// NETWORK 11
DS_HMI.b1001_02_AutoPreparationCompletedFlag := (DS_HMI.b1000_02_AutoPreparationOnOffPB AND bInternalInput_b000_05_ThermalOilTempCtrlReadySignal AND bInternalInput_b000_08_TopDistillatorTempCtrlReadySignal OR DS_HMI.b1001_02_AutoPreparationCompletedFlag) AND DS_HMI.b1000_00_AutoModeOnOffPB AND DS_HMI.b1000_03_AutoModeStartStopPB;

// NETWORK 12
DS_HMI.b1001_10_AutoProgressFlag := DS_HMI.b1001_02_AutoPreparationCompletedFlag;
END_ACTION

ACTION AutoHCTopUp_LD:
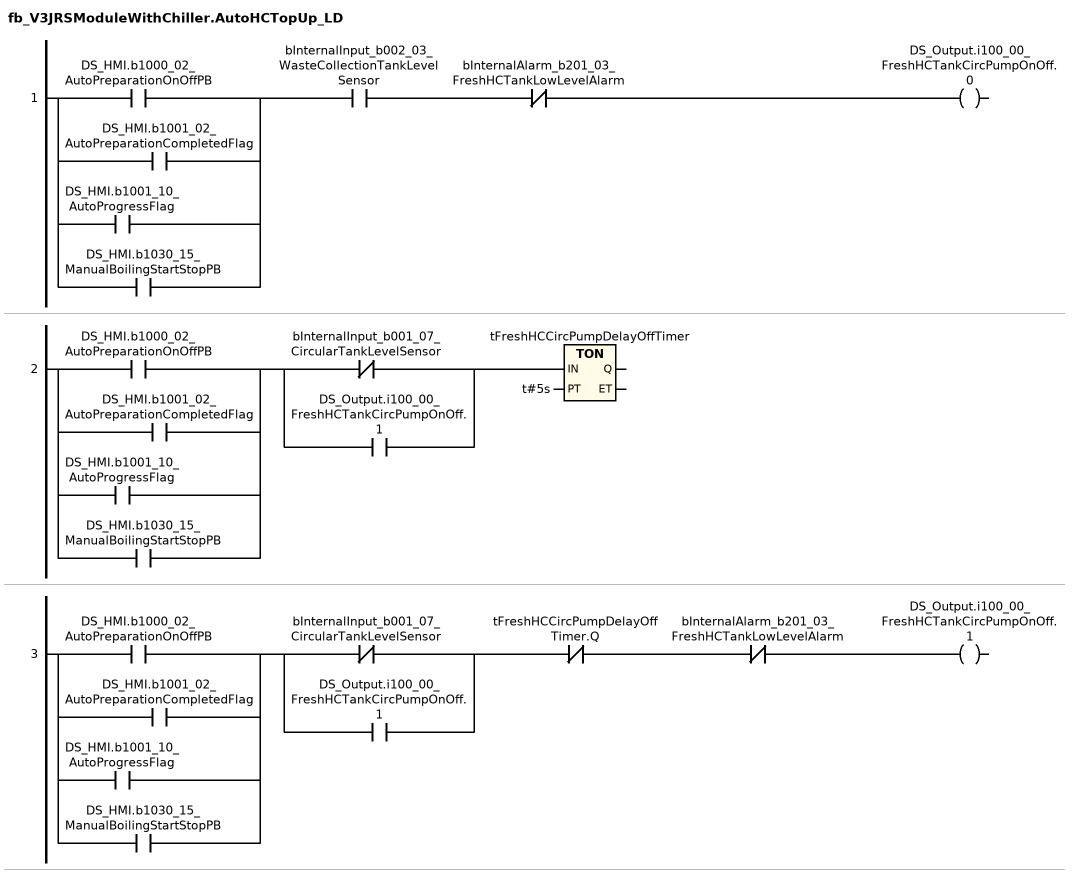
// NETWORK 1
DS_Output.i100_00_FreshHCTankCircPumpOnOff.0 := (DS_HMI.b1000_02_AutoPreparationOnOffPB OR DS_HMI.b1001_02_AutoPreparationCompletedFlag OR DS_HMI.b1001_10_AutoProgressFlag OR DS_HMI.b1030_15_ManualBoilingStartStopPB) AND bInternalInput_b002_03_WasteCollectionTankLevelSensor AND NOT bInternalAlarm_b201_03_FreshHCTankLowLevelAlarm;

// NETWORK 2
tFreshHCCircPumpDelayOffTimer(IN := (DS_HMI.b1000_02_AutoPreparationOnOffPB OR DS_HMI.b1001_02_AutoPreparationCompletedFlag OR DS_HMI.b1001_10_AutoProgressFlag OR DS_HMI.b1030_15_ManualBoilingStartStopPB) AND (NOT bInternalInput_b001_07_CircularTankLevelSensor OR DS_Output.i100_00_FreshHCTankCircPumpOnOff.1), PT := t#5s); // TON

// NETWORK 3
DS_Output.i100_00_FreshHCTankCircPumpOnOff.1 := ((DS_HMI.b1000_02_AutoPreparationOnOffPB OR DS_HMI.b1001_02_AutoPreparationCompletedFlag OR DS_HMI.b1001_10_AutoProgressFlag OR DS_HMI.b1030_15_ManualBoilingStartStopPB) AND (NOT bInternalInput_b001_07_CircularTankLevelSensor OR DS_Output.i100_00_FreshHCTankCircPumpOnOff.1)) AND NOT tFreshHCCircPumpDelayOffTimer.Q AND NOT bInternalAlarm_b201_03_FreshHCTankLowLevelAlarm;
END_ACTION

ACTION BuzzerCtrl_ST:
IF ARiBuzzerOut[1] <>0
AND ARiBuzzerOut[2] <> 0
AND ARiBuzzerOut[3] <> 0
AND ARiBuzzerOut[4] <> 0
THEN
DS_Output.i100_04_Buzzer.0 := TRUE;
ELSE
DS_Output.i100_04_Buzzer.0 := FALSE;
END_IF
END_ACTION

ACTION ChillerCtrl_LD:
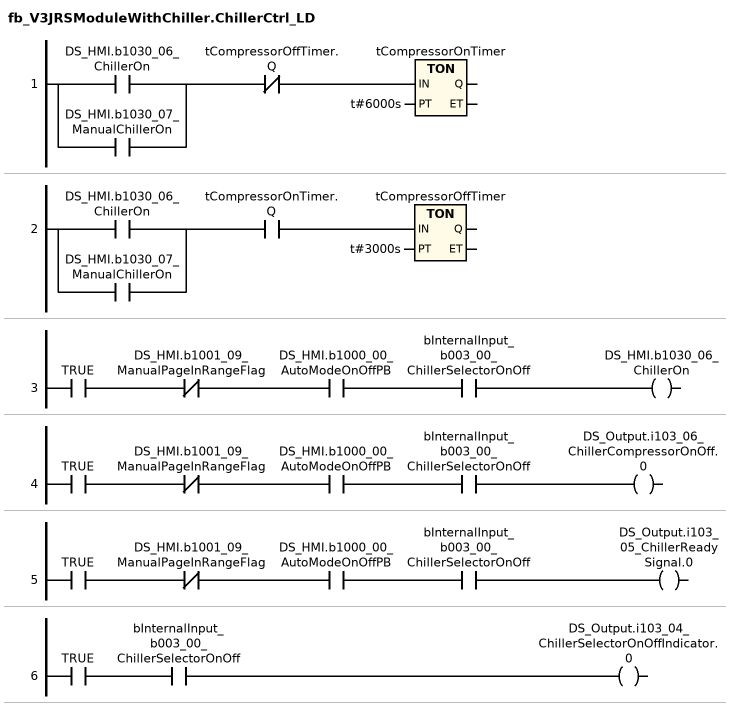
// NETWORK 1
tCompressorOnTimer(IN := (DS_HMI.b1030_06_ChillerOn OR DS_HMI.b1030_07_ManualChillerOn) AND NOT tCompressorOffTimer.Q, PT := t#6000s); // TON

// NETWORK 2
tCompressorOffTimer(IN := (DS_HMI.b1030_06_ChillerOn OR DS_HMI.b1030_07_ManualChillerOn) AND tCompressorOnTimer.Q, PT := t#3000s); // TON

// NETWORK 3
DS_HMI.b1030_06_ChillerOn := TRUE AND NOT DS_HMI.b1001_09_ManualPageInRangeFlag AND DS_HMI.b1000_00_AutoModeOnOffPB AND bInternalInput_b003_00_ChillerSelectorOnOff;

// NETWORK 4
DS_Output.i103_06_ChillerCompressorOnOff.0 := TRUE AND NOT DS_HMI.b1001_09_ManualPageInRangeFlag AND DS_HMI.b1000_00_AutoModeOnOffPB AND bInternalInput_b003_00_ChillerSelectorOnOff;

// NETWORK 5
DS_Output.i103_05_ChillerReadySignal.0 := TRUE AND NOT DS_HMI.b1001_09_ManualPageInRangeFlag AND DS_HMI.b1000_00_AutoModeOnOffPB AND bInternalInput_b003_00_ChillerSelectorOnOff;

// NETWORK 6
DS_Output.i103_04_ChillerSelectorOnOffIndicator.0 := TRUE AND bInternalInput_b003_00_ChillerSelectorOnOff;
END_ACTION

ACTION FixOutput_LD:
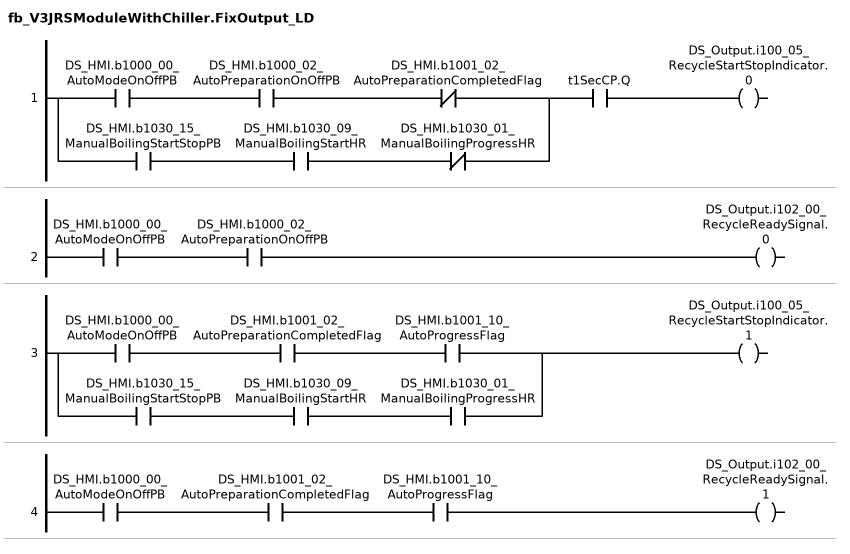
// NETWORK 1
DS_Output.i100_05_RecycleStartStopIndicator.0 := (DS_HMI.b1000_00_AutoModeOnOffPB AND DS_HMI.b1000_02_AutoPreparationOnOffPB AND NOT DS_HMI.b1001_02_AutoPreparationCompletedFlag OR DS_HMI.b1030_15_ManualBoilingStartStopPB AND DS_HMI.b1030_09_ManualBoilingStartHR AND NOT DS_HMI.b1030_01_ManualBoilingProgressHR) AND t1SecCP.Q;

// NETWORK 2
DS_Output.i102_00_RecycleReadySignal.0 := DS_HMI.b1000_00_AutoModeOnOffPB AND DS_HMI.b1000_02_AutoPreparationOnOffPB;

// NETWORK 3
DS_Output.i100_05_RecycleStartStopIndicator.1 := DS_HMI.b1000_00_AutoModeOnOffPB AND DS_HMI.b1001_02_AutoPreparationCompletedFlag AND DS_HMI.b1001_10_AutoProgressFlag OR DS_HMI.b1030_15_ManualBoilingStartStopPB AND DS_HMI.b1030_09_ManualBoilingStartHR AND DS_HMI.b1030_01_ManualBoilingProgressHR;

// NETWORK 4
DS_Output.i102_00_RecycleReadySignal.1 := DS_HMI.b1000_00_AutoModeOnOffPB AND DS_HMI.b1001_02_AutoPreparationCompletedFlag AND DS_HMI.b1001_10_AutoProgressFlag;
END_ACTION

ACTION HighLowLimitCtrl_ST:
(*Low Limit Ctrl*)
IF DS_HMI.iD490_ManualBoilCycleSV < 1 THEN
DS_HMI.iD490_ManualBoilCycleSV := 1;
END_IF

IF DS_HMI.iD200_AutoBoilProcessTimeSV_Min < 30 THEN
DS_HMI.iD200_AutoBoilProcessTimeSV_Min := 30;
END_IF

IF DS_HMI.iD201_AutoBoilDownTimeSV_Min < 5 THEN
DS_HMI.iD201_AutoBoilDownTimeSV_Min := 5;
END_IF

IF DS_HMI.iD202_AutoBoilDistillatorDrainTimeSV_Sec < 5 THEN
DS_HMI.iD202_AutoBoilDistillatorDrainTimeSV_Sec := 5;
END_IF

IF DS_HMI.iD203_AutoBoilSludgeDrainTimeSV_Sec < 5 THEN
DS_HMI.iD203_AutoBoilSludgeDrainTimeSV_Sec := 5;
END_IF

IF DS_HMI.iD210_ManualBoilDownTimeSV_Min < 5 THEN
DS_HMI.iD210_ManualBoilDownTimeSV_Min := 5;
END_IF

IF DS_HMI.iD211_ManualBoilSludgeCoolingTimeSV_Min < 1 THEN
DS_HMI.iD211_ManualBoilSludgeCoolingTimeSV_Min := 1;
END_IF

IF DS_HMI.iD212_ManualBoilSludgeDrainSV_Sec < 5 THEN
DS_HMI.iD212_ManualBoilSludgeDrainSV_Sec := 5;
END_IF




(*High LImit Ctrl*)
IF DS_HMI.iD490_ManualBoilCycleSV > 99 THEN
DS_HMI.iD490_ManualBoilCycleSV := 99;
END_IF

IF DS_HMI.iD200_AutoBoilProcessTimeSV_Min > 9999 THEN
DS_HMI.iD200_AutoBoilProcessTimeSV_Min := 9999;
END_IF

IF DS_HMI.iD201_AutoBoilDownTimeSV_Min > 9999 THEN
DS_HMI.iD201_AutoBoilDownTimeSV_Min := 9999;
END_IF

IF DS_HMI.iD202_AutoBoilDistillatorDrainTimeSV_Sec > 300 THEN
DS_HMI.iD202_AutoBoilDistillatorDrainTimeSV_Sec := 300;
END_IF

IF DS_HMI.iD203_AutoBoilSludgeDrainTimeSV_Sec > 300 THEN
DS_HMI.iD203_AutoBoilSludgeDrainTimeSV_Sec := 300;
END_IF

IF DS_HMI.iD210_ManualBoilDownTimeSV_Min > 99 THEN
DS_HMI.iD210_ManualBoilDownTimeSV_Min := 99;
END_IF

IF DS_HMI.iD211_ManualBoilSludgeCoolingTimeSV_Min > 9999 THEN
DS_HMI.iD211_ManualBoilSludgeCoolingTimeSV_Min := 9999;
END_IF

IF DS_HMI.iD212_ManualBoilSludgeDrainSV_Sec > 300 THEN
DS_HMI.iD212_ManualBoilSludgeDrainSV_Sec := 300;
END_IF
END_ACTION

ACTION JRSMachineServiceCtrl_LD:
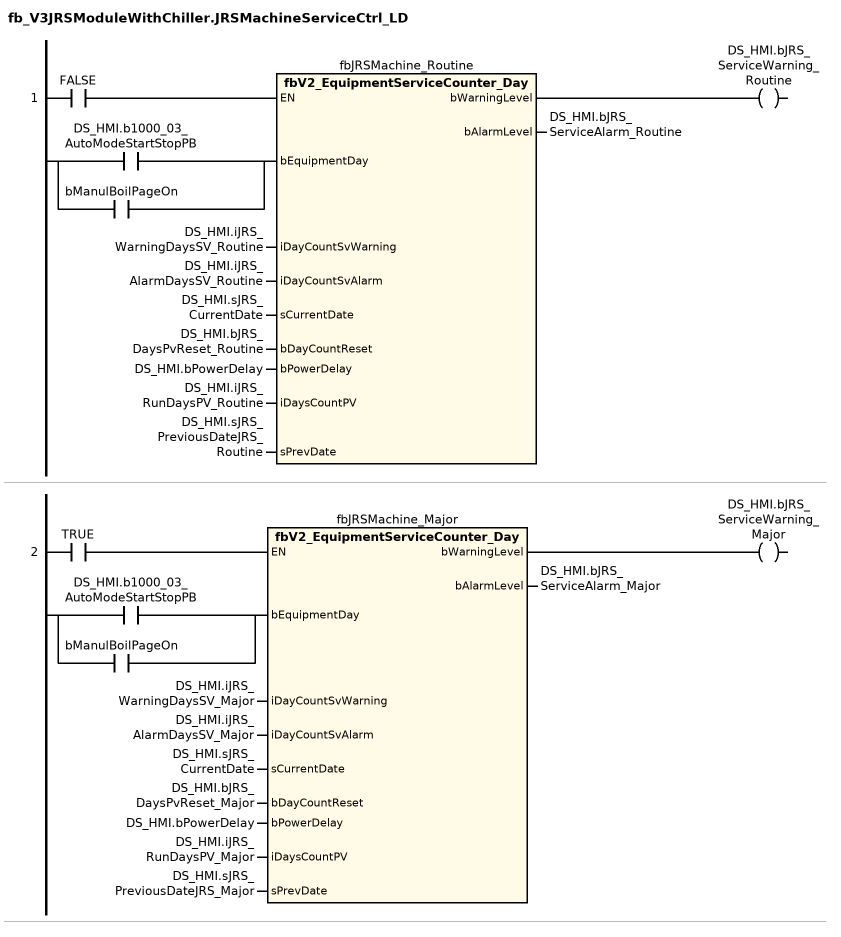
// NETWORK 1
IF FALSE THEN
    fbJRSMachine_Routine(
        bEquipmentDay := DS_HMI.b1000_03_AutoModeStartStopPB OR bManulBoilPageOn,
        iDayCountSvWarning := DS_HMI.iJRS_WarningDaysSV_Routine,
        iDayCountSvAlarm := DS_HMI.iJRS_AlarmDaysSV_Routine,
        sCurrentDate := DS_HMI.sJRS_CurrentDate,
        bDayCountReset := DS_HMI.bJRS_DaysPvReset_Routine,
        bPowerDelay := DS_HMI.bPowerDelay,
        iDaysCountPV := DS_HMI.iJRS_RunDaysPV_Routine,
        sPrevDate := DS_HMI.sJRS_PreviousDateJRS_Routine,
        bAlarmLevel => DS_HMI.bJRS_ServiceAlarm_Routine); // fbV2_EquipmentServiceCounter_Day
END_IF
DS_HMI.bJRS_ServiceWarning_Routine := fbJRSMachine_Routine.bWarningLevel;

// NETWORK 2
fbJRSMachine_Major(
    bEquipmentDay := DS_HMI.b1000_03_AutoModeStartStopPB OR bManulBoilPageOn,
    iDayCountSvWarning := DS_HMI.iJRS_WarningDaysSV_Major,
    iDayCountSvAlarm := DS_HMI.iJRS_AlarmDaysSV_Major,
    sCurrentDate := DS_HMI.sJRS_CurrentDate,
    bDayCountReset := DS_HMI.bJRS_DaysPvReset_Major,
    bPowerDelay := DS_HMI.bPowerDelay,
    iDaysCountPV := DS_HMI.iJRS_RunDaysPV_Major,
    sPrevDate := DS_HMI.sJRS_PreviousDateJRS_Major,
    bAlarmLevel => DS_HMI.bJRS_ServiceAlarm_Major); // fbV2_EquipmentServiceCounter_Day
DS_HMI.bJRS_ServiceWarning_Major := fbJRSMachine_Major.bWarningLevel;
END_ACTION

ACTION ManualBoilingCtrl_LD:
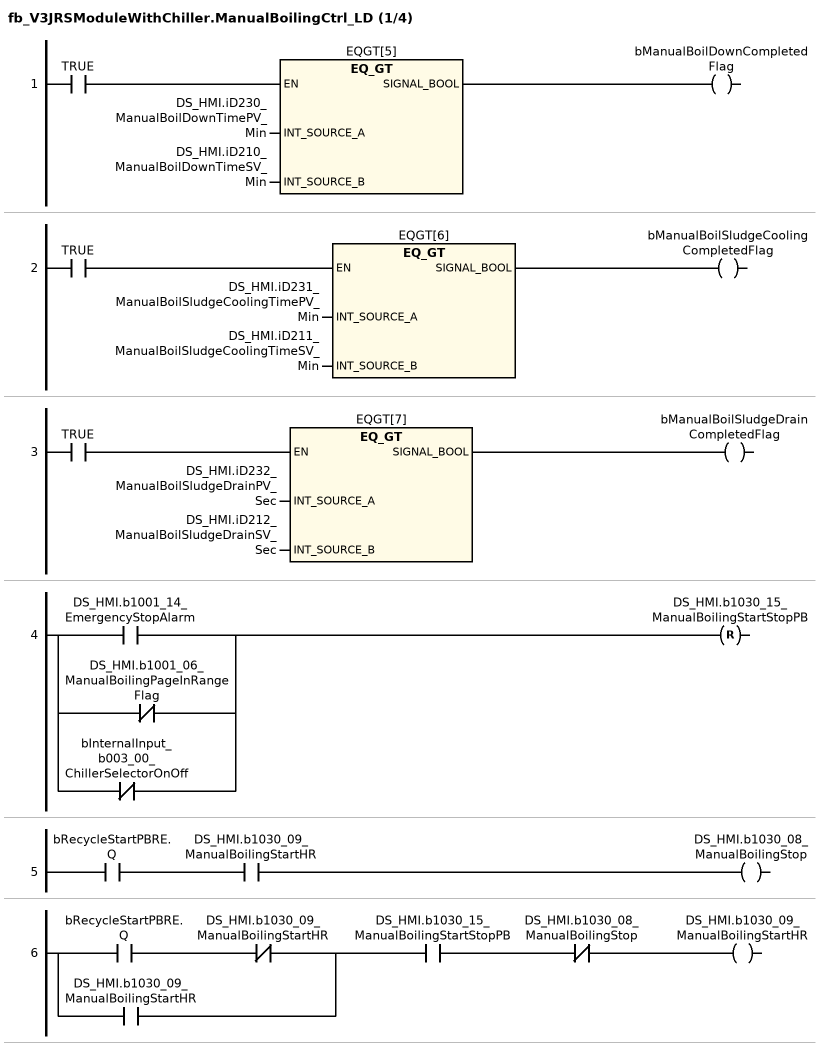
// NETWORK 1
EQGT[5](INT_SOURCE_A := DS_HMI.iD230_ManualBoilDownTimePV_Min, INT_SOURCE_B := DS_HMI.iD210_ManualBoilDownTimeSV_Min); // EQ_GT
bManualBoilDownCompletedFlag := EQGT[5].SIGNAL_BOOL;

// NETWORK 2
EQGT[6](INT_SOURCE_A := DS_HMI.iD231_ManualBoilSludgeCoolingTimePV_Min, INT_SOURCE_B := DS_HMI.iD211_ManualBoilSludgeCoolingTimeSV_Min); // EQ_GT
bManualBoilSludgeCoolingCompletedFlag := EQGT[6].SIGNAL_BOOL;

// NETWORK 3
EQGT[7](INT_SOURCE_A := DS_HMI.iD232_ManualBoilSludgeDrainPV_Sec, INT_SOURCE_B := DS_HMI.iD212_ManualBoilSludgeDrainSV_Sec); // EQ_GT
bManualBoilSludgeDrainCompletedFlag := EQGT[7].SIGNAL_BOOL;

// NETWORK 4
DS_HMI.b1030_15_ManualBoilingStartStopPB R= DS_HMI.b1001_14_EmergencyStopAlarm OR NOT DS_HMI.b1001_06_ManualBoilingPageInRangeFlag OR NOT bInternalInput_b003_00_ChillerSelectorOnOff;

// NETWORK 5
DS_HMI.b1030_08_ManualBoilingStop := bRecycleStartPBRE.Q AND DS_HMI.b1030_09_ManualBoilingStartHR;

// NETWORK 6
DS_HMI.b1030_09_ManualBoilingStartHR := (bRecycleStartPBRE.Q AND NOT DS_HMI.b1030_09_ManualBoilingStartHR OR DS_HMI.b1030_09_ManualBoilingStartHR) AND DS_HMI.b1030_15_ManualBoilingStartStopPB AND NOT DS_HMI.b1030_08_ManualBoilingStop;

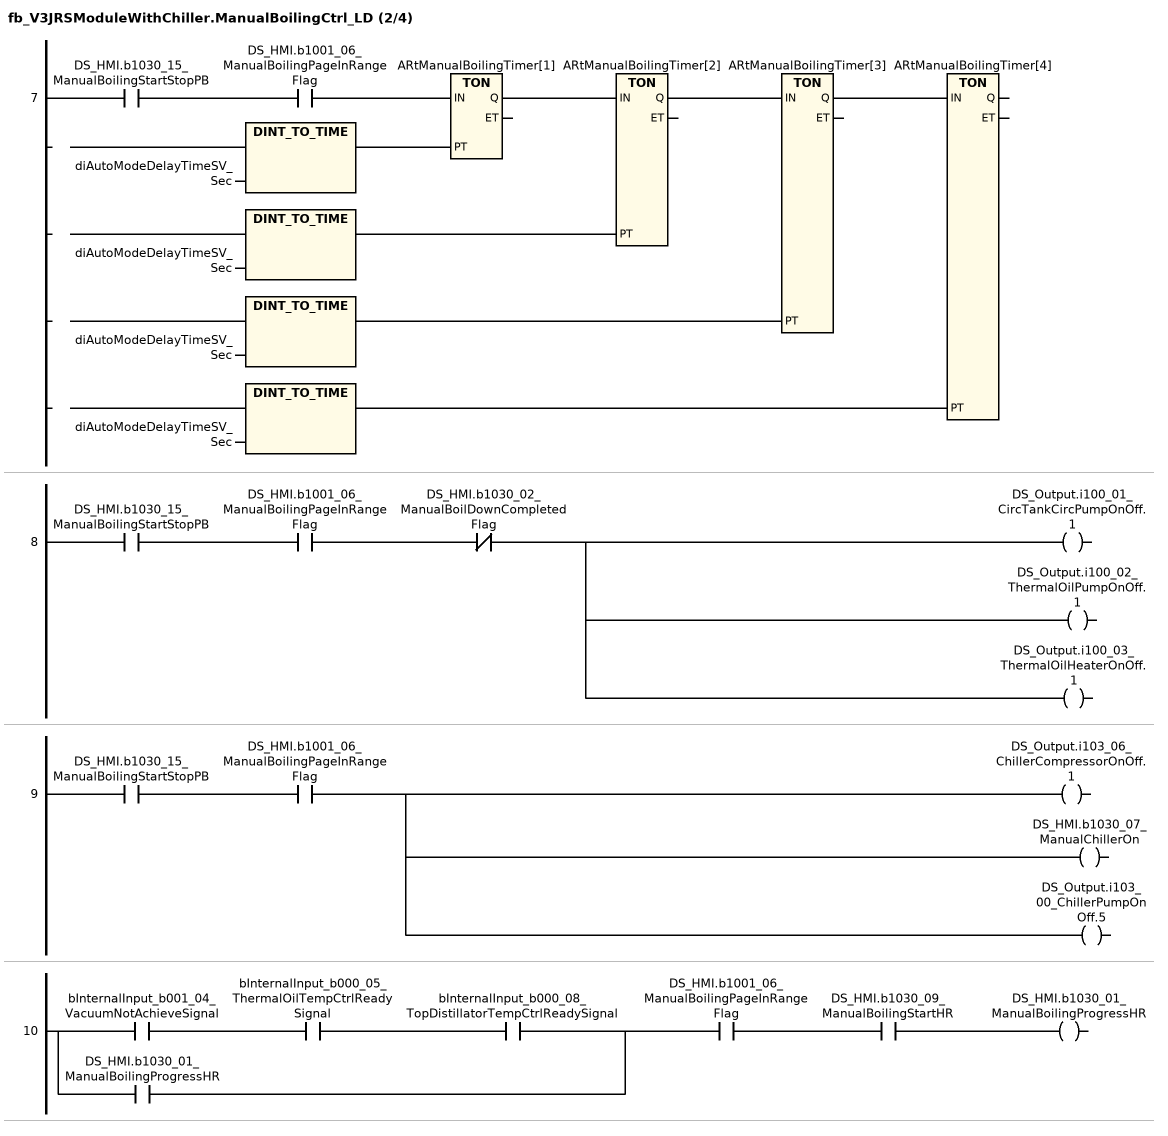
// NETWORK 7
ARtManualBoilingTimer[1](IN := DS_HMI.b1030_15_ManualBoilingStartStopPB AND DS_HMI.b1001_06_ManualBoilingPageInRangeFlag, PT := DINT_TO_TIME(diAutoModeDelayTimeSV_Sec)); // TON
ARtManualBoilingTimer[2](IN := ARtManualBoilingTimer[1].Q, PT := DINT_TO_TIME(diAutoModeDelayTimeSV_Sec)); // TON
ARtManualBoilingTimer[3](IN := ARtManualBoilingTimer[2].Q, PT := DINT_TO_TIME(diAutoModeDelayTimeSV_Sec)); // TON
ARtManualBoilingTimer[4](IN := ARtManualBoilingTimer[3].Q, PT := DINT_TO_TIME(diAutoModeDelayTimeSV_Sec)); // TON

// NETWORK 8
_w5 := DS_HMI.b1030_15_ManualBoilingStartStopPB AND DS_HMI.b1001_06_ManualBoilingPageInRangeFlag AND NOT DS_HMI.b1030_02_ManualBoilDownCompletedFlag;
DS_Output.i100_01_CircTankCircPumpOnOff.1 := _w5;
DS_Output.i100_02_ThermalOilPumpOnOff.1 := _w5;
DS_Output.i100_03_ThermalOilHeaterOnOff.1 := _w5;

// NETWORK 9
_w6 := DS_HMI.b1030_15_ManualBoilingStartStopPB AND DS_HMI.b1001_06_ManualBoilingPageInRangeFlag;
DS_Output.i103_06_ChillerCompressorOnOff.1 := _w6;
DS_HMI.b1030_07_ManualChillerOn := _w6;
DS_Output.i103_00_ChillerPumpOnOff.5 := _w6;

// NETWORK 10
DS_HMI.b1030_01_ManualBoilingProgressHR := (bInternalInput_b001_04_VacuumNotAchieveSignal AND bInternalInput_b000_05_ThermalOilTempCtrlReadySignal AND bInternalInput_b000_08_TopDistillatorTempCtrlReadySignal OR DS_HMI.b1030_01_ManualBoilingProgressHR) AND DS_HMI.b1001_06_ManualBoilingPageInRangeFlag AND DS_HMI.b1030_09_ManualBoilingStartHR;

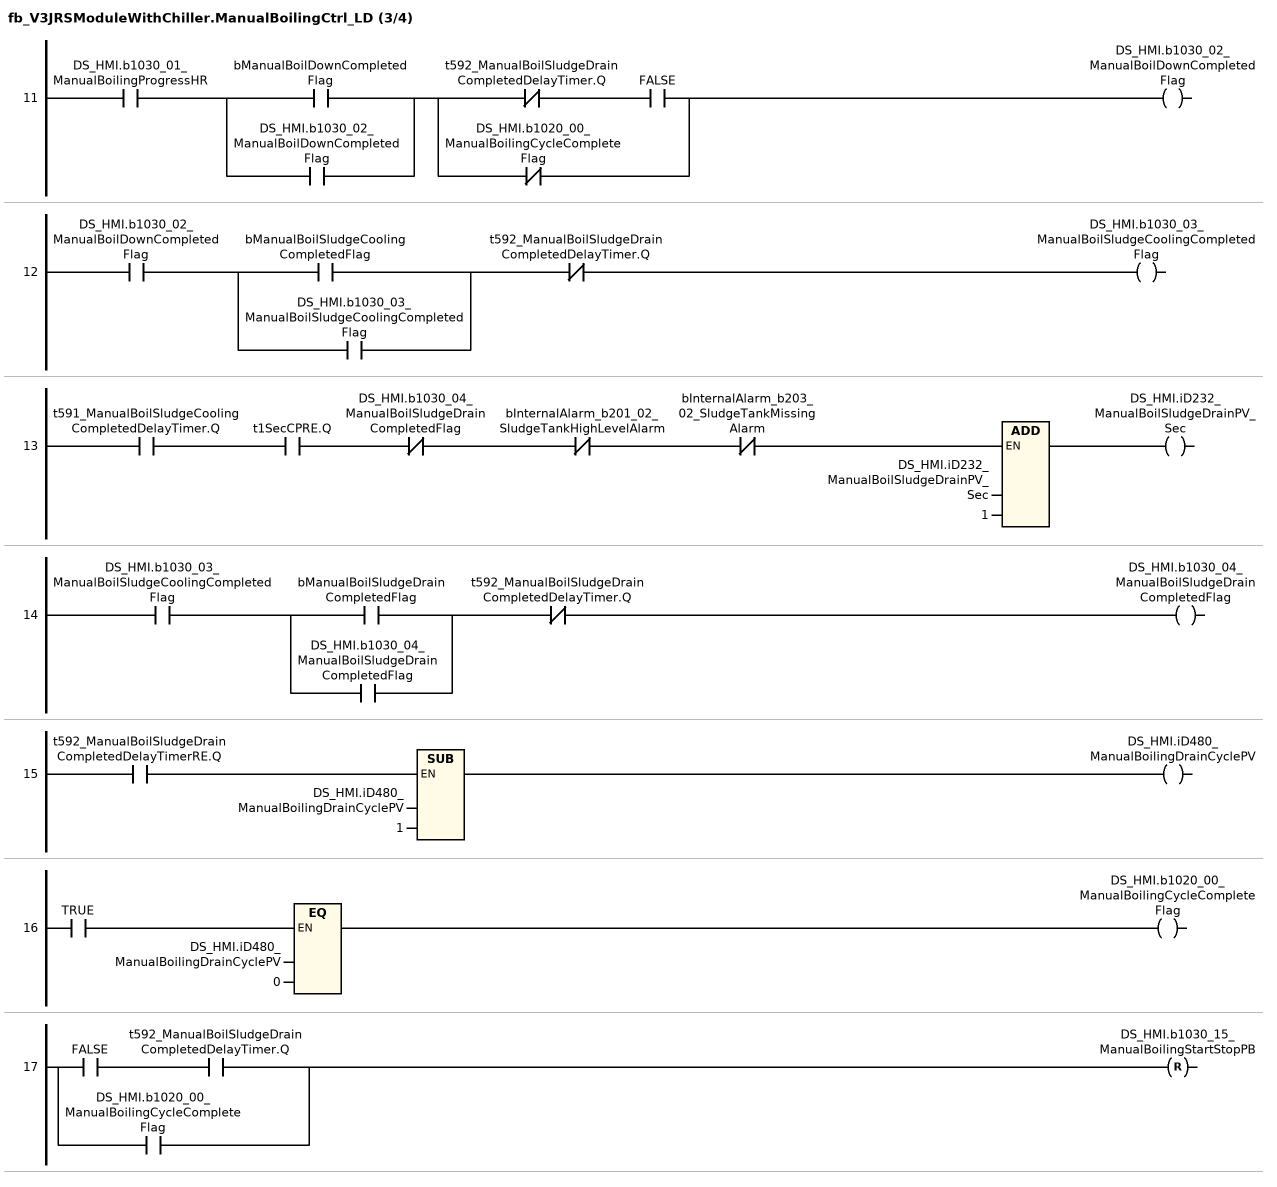
// NETWORK 11
DS_HMI.b1030_02_ManualBoilDownCompletedFlag := DS_HMI.b1030_01_ManualBoilingProgressHR AND (bManualBoilDownCompletedFlag OR DS_HMI.b1030_02_ManualBoilDownCompletedFlag) AND (NOT t592_ManualBoilSludgeDrainCompletedDelayTimer.Q AND FALSE OR NOT DS_HMI.b1020_00_ManualBoilingCycleCompleteFlag);

// NETWORK 12
DS_HMI.b1030_03_ManualBoilSludgeCoolingCompletedFlag := (DS_HMI.b1030_02_ManualBoilDownCompletedFlag AND (bManualBoilSludgeCoolingCompletedFlag OR DS_HMI.b1030_03_ManualBoilSludgeCoolingCompletedFlag)) AND NOT t592_ManualBoilSludgeDrainCompletedDelayTimer.Q;

// NETWORK 13
IF t591_ManualBoilSludgeCoolingCompletedDelayTimer.Q AND t1SecCPRE.Q AND NOT DS_HMI.b1030_04_ManualBoilSludgeDrainCompletedFlag AND NOT bInternalAlarm_b201_02_SludgeTankHighLevelAlarm AND NOT bInternalAlarm_b203_02_SludgeTankMissingAlarm THEN
    _w7 := DS_HMI.iD232_ManualBoilSludgeDrainPV_Sec + 1;
END_IF
DS_HMI.iD232_ManualBoilSludgeDrainPV_Sec := _w7;

// NETWORK 14
DS_HMI.b1030_04_ManualBoilSludgeDrainCompletedFlag := (DS_HMI.b1030_03_ManualBoilSludgeCoolingCompletedFlag AND (bManualBoilSludgeDrainCompletedFlag OR DS_HMI.b1030_04_ManualBoilSludgeDrainCompletedFlag)) AND NOT t592_ManualBoilSludgeDrainCompletedDelayTimer.Q;

// NETWORK 15
IF t592_ManualBoilSludgeDrainCompletedDelayTimerRE.Q THEN _w8 := DS_HMI.iD480_ManualBoilingDrainCyclePV - 1; END_IF
DS_HMI.iD480_ManualBoilingDrainCyclePV := _w8;

// NETWORK 16
DS_HMI.b1020_00_ManualBoilingCycleCompleteFlag := DS_HMI.iD480_ManualBoilingDrainCyclePV = 0;

// NETWORK 17
DS_HMI.b1030_15_ManualBoilingStartStopPB R= FALSE AND t592_ManualBoilSludgeDrainCompletedDelayTimer.Q OR DS_HMI.b1020_00_ManualBoilingCycleCompleteFlag;

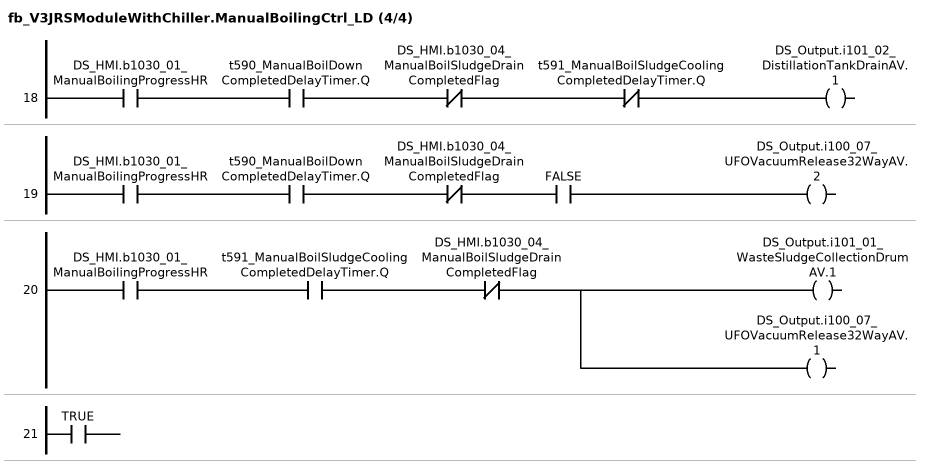
// NETWORK 18
DS_Output.i101_02_DistillationTankDrainAV.1 := DS_HMI.b1030_01_ManualBoilingProgressHR AND t590_ManualBoilDownCompletedDelayTimer.Q AND NOT DS_HMI.b1030_04_ManualBoilSludgeDrainCompletedFlag AND NOT t591_ManualBoilSludgeCoolingCompletedDelayTimer.Q;

// NETWORK 19
DS_Output.i100_07_UFOVacuumRelease32WayAV.2 := DS_HMI.b1030_01_ManualBoilingProgressHR AND t590_ManualBoilDownCompletedDelayTimer.Q AND NOT DS_HMI.b1030_04_ManualBoilSludgeDrainCompletedFlag AND FALSE;

// NETWORK 20
_w9 := DS_HMI.b1030_01_ManualBoilingProgressHR AND t591_ManualBoilSludgeCoolingCompletedDelayTimer.Q AND NOT DS_HMI.b1030_04_ManualBoilSludgeDrainCompletedFlag;
DS_Output.i101_01_WasteSludgeCollectionDrumAV.1 := _w9;
DS_Output.i100_07_UFOVacuumRelease32WayAV.1 := _w9;

// NETWORK 21
END_ACTION

ACTION ManualBoilingCtrl_ST:
	(*Timer*)
	t590_ManualBoilDownCompletedDelayTimer(IN:=DS_HMI.b1030_02_ManualBoilDownCompletedFlag , PT:=t#1s , Q=> , ET=> );
	t591_ManualBoilSludgeCoolingCompletedDelayTimer(IN:=DS_HMI.b1030_03_ManualBoilSludgeCoolingCompletedFlag , PT:=t#1s , Q=> , ET=> );
	t592_ManualBoilSludgeDrainCompletedDelayTimer(IN:=DS_HMI.b1030_04_ManualBoilSludgeDrainCompletedFlag , PT:=t#1s , Q=> , ET=> );

	(*R_TRIG*)
	t592_ManualBoilSludgeDrainCompletedDelayTimerRE(CLK:=t592_ManualBoilSludgeDrainCompletedDelayTimer.Q , Q=> );
	bManualBoilSludgeDrainCompletedRE(CLK:=DS_HMI.b1030_04_ManualBoilSludgeDrainCompletedFlag , Q=> );


	(*ManualBoiling Boil Process Time Counting*)
	IF DS_HMI.b1030_01_ManualBoilingProgressHR
	AND t1SecCPRE.Q
	THEN

		IF NOT DS_HMI.b1030_02_ManualBoilDownCompletedFlag THEN

			DS_HMI.iD235_ManualBoilDownTimePV_Sec := DS_HMI.iD235_ManualBoilDownTimePV_Sec + 1;
	
			IF DS_HMI.iD235_ManualBoilDownTimePV_Sec > 59 THEN
				DS_HMI.iD230_ManualBoilDownTimePV_Min := DS_HMI.iD230_ManualBoilDownTimePV_Min + 1;
				DS_HMI.iD235_ManualBoilDownTimePV_Sec := 0;
			END_IF

		END_IF

	END_IF

	(*ManualBoiling Boil Down Time Counting*)

	IF t590_ManualBoilDownCompletedDelayTimer.Q
	AND t1SecCPRE.Q
	THEN

		IF NOT DS_HMI.b1030_03_ManualBoilSludgeCoolingCompletedFlag THEN

			DS_HMI.iD236_ManualBoilSludgeCoolingTimePV_Sec := DS_HMI.iD236_ManualBoilSludgeCoolingTimePV_Sec + 1;

			IF DS_HMI.iD236_ManualBoilSludgeCoolingTimePV_Sec > 59 THEN
				DS_HMI.iD231_ManualBoilSludgeCoolingTimePV_Min := DS_HMI.iD231_ManualBoilSludgeCoolingTimePV_Min + 1;
				DS_HMI.iD236_ManualBoilSludgeCoolingTimePV_Sec := 0;
			END_IF

		END_IF

	END_IF

	(*Manual Boiling Reset*)
	IF NOT DS_HMI.b1030_15_ManualBoilingStartStopPB THEN
		DS_HMI.iD230_ManualBoilDownTimePV_Min						:= 0;
		DS_HMI.iD231_ManualBoilSludgeCoolingTimePV_Min				:= 0;
		DS_HMI.iD232_ManualBoilSludgeDrainPV_Sec					:= 0;
		DS_HMI.iD480_ManualBoilingDrainCyclePV						:= DS_HMI.iD490_ManualBoilCycleSV;

	END_IF



	IF bManualBoilSludgeDrainCompletedRE.Q OR  DS_HMI.b1020_00_ManualBoilingCycleCompleteFlag THEN
	
		DS_HMI.iD230_ManualBoilDownTimePV_Min						:= 0;
		DS_HMI.iD231_ManualBoilSludgeCoolingTimePV_Min				:= 0;
		DS_HMI.iD232_ManualBoilSludgeDrainPV_Sec					:= 0;
		DS_HMI.iD235_ManualBoilDownTimePV_Sec						:= 0;
		DS_HMI.iD236_ManualBoilSludgeCoolingTimePV_Sec				:= 0;

	END_IF
END_ACTION

ACTION ManualCtrl_ST:
	(*Manual Page In Range*)
	IF (	DS_HMI.iD0_HMICurrentPage > 19 		AND 	DS_HMI.iD0_HMICurrentPage < 41)
	OR	DS_HMI.iD0_HMICurrentPage = 2
	OR	DS_HMI.iD0_HMICurrentPage = 61
	OR	DS_HMI.iD0_HMICurrentPage = 63
	OR	DS_HMI.iD0_HMICurrentPage = 100
	OR	DS_HMI.iD0_HMICurrentPage = 101
	OR	DS_HMI.iD0_HMICurrentPage = 103 	THEN
		DS_HMI.b1001_09_ManualPageInRangeFlag := TRUE;
	ELSE
		DS_HMI.b1001_09_ManualPageInRangeFlag := FALSE;
	END_IF


	(*Manual Boiling Page In Range*)
	IF (	DS_HMI.iD0_HMICurrentPage > 99 		AND 	DS_HMI.iD0_HMICurrentPage < 102)
	OR	DS_HMI.iD0_HMICurrentPage = 22 		THEN
		DS_HMI.b1001_06_ManualBoilingPageInRangeFlag := TRUE;
	ELSE
		DS_HMI.b1001_06_ManualBoilingPageInRangeFlag := FALSE;
	END_IF



	IF NOT DS_HMI.b1001_09_ManualPageInRangeFlag OR DS_HMI.b1001_14_EmergencyStopAlarm THEN
		DS_Output.i100_00_FreshHCTankCircPumpOnOff.15			:= FALSE;
		DS_Output.i100_01_CircTankCircPumpOnOff.15				:= FALSE;
		DS_Output.i100_02_ThermalOilPumpOnOff.15				:= FALSE;
		DS_Output.i100_03_ThermalOilHeaterOnOff.15				:= FALSE;
		DS_Output.i100_04_Buzzer.15								:= FALSE;
		DS_Output.i100_05_RecycleStartStopIndicator.15				:= FALSE;
		DS_Output.i100_06_Reserved.15							:= FALSE;
		DS_Output.i100_07_UFOVacuumRelease32WayAV.15		:= FALSE;

		DS_Output.i101_00_CondenserTankVacuumReleaseAV.15	:= FALSE;
		DS_Output.i101_01_WasteSludgeCollectionDrumAV.15		:= FALSE;
		DS_Output.i101_02_DistillationTankDrainAV.15				:= FALSE;
		DS_Output.i101_03_EconomizerAV.15						:= FALSE;
		DS_Output.i101_04_Reserved.15							:= FALSE;
		DS_Output.i101_05_Reserved.15							:= FALSE;
		DS_Output.i101_06_VaporGenerationAV.15					:= FALSE;
		DS_Output.i101_07_VacuumSharingAV.15					:= FALSE;

		DS_Output.i102_00_RecycleReadySignal.15					:= FALSE;
		DS_Output.i102_01_VaporNotAvailableForRequestSignal.15	:= FALSE;
		DS_Output.i102_02_ToMainMachineSignal3.15				:= FALSE;
		DS_Output.i102_03_ToMainMachineSignal4.15				:= FALSE;
		DS_Output.i102_04_ToMainMachineSignal5.15				:= FALSE;
		DS_Output.i102_05_Reserved.15							:= FALSE;
		DS_Output.i102_06_Reserved.15							:= FALSE;
		DS_Output.i102_07_Reserved.15							:= FALSE;

		DS_Output.i103_00_ChillerPumpOnOff.15					:= FALSE;
		DS_Output.i103_01_Reserved.15							:= FALSE;
		DS_Output.i103_02_Reserved.15							:= FALSE;
		DS_Output.i103_03_Reserved.15							:= FALSE;
		DS_Output.i103_04_ChillerSelectorOnOffIndicator.15			:= FALSE;
		DS_Output.i103_05_ChillerReadySignal.15					:= FALSE;
		DS_Output.i103_06_ChillerCompressorOnOff.15				:= FALSE;
		DS_Output.i103_07_Reserved.15							:= FALSE;
	END_IF

	IF NOT bInternalInput_b003_00_ChillerSelectorOnOff THEN
		DS_Output.i103_06_ChillerCompressorOnOff.15				:= FALSE;
	END_IF
END_ACTION

ACTION MessageDisplayCtrl_ST:
	IF  NOT DS_HMI.b1001_15_AlarmOccur THEN

		IF NOT 		DS_HMI.b1000_00_AutoModeOnOffPB THEN

			DS_HMI.iD100_MessageDisplay := 0;
			DS_HMI.sD100_MessageDisplay := 'Machine Idle';

(*		ELSIF 		DS_HMI.b1000_00_AutoModeOnOffPB
		AND 		DS_HMI.b1000_01_AutoOriginOnOffPB
		AND NOT 	DS_HMI.b1001_01_AutoOriginCompletedFlag THEN

			DS_HMI.iD100_MessageDisplay := 1;
			DS_HMI.sD100_MessageDisplay := 'Auto Origin In Progress...';
*)
		ELSIF 		DS_HMI.b1000_00_AutoModeOnOffPB
		AND 		DS_HMI.b1000_02_AutoPreparationOnOffPB
		AND NOT 	DS_HMI.b1001_02_AutoPreparationCompletedFlag THEN

			DS_HMI.iD100_MessageDisplay := 2;
			DS_HMI.sD100_MessageDisplay := 'Auto Preparation In Progress...';

		ELSIF 		DS_HMI.b1000_00_AutoModeOnOffPB
(*		AND 		DS_HMI.b1001_01_AutoOriginCompletedFlag*)
		AND 		DS_HMI.b1000_02_AutoPreparationOnOffPB
		AND 		DS_HMI.b1001_02_AutoPreparationCompletedFlag THEN

			DS_HMI.iD100_MessageDisplay := 3;
			DS_HMI.sD100_MessageDisplay := 'Machine Ready, Press "Start" for Operation';

		ELSIF 		DS_HMI.b1000_00_AutoModeOnOffPB
(*		AND 		DS_HMI.b1001_01_AutoOriginCompletedFlag*)
		AND 		DS_HMI.b1001_02_AutoPreparationCompletedFlag
		AND 		DS_HMI.b1001_10_AutoProgressFlag
		AND NOT 	DS_HMI.b1000_05_AutoCycleStopPB THEN

			DS_HMI.iD100_MessageDisplay := 4;
			DS_HMI.sD100_MessageDisplay := 'Machine Operation...';

		ELSIF 		DS_HMI.b1000_00_AutoModeOnOffPB
(*		AND 		DS_HMI.b1001_01_AutoOriginCompletedFlag*)
		AND 		DS_HMI.b1001_02_AutoPreparationCompletedFlag
		AND 		DS_HMI.b1001_10_AutoProgressFlag
		AND 		DS_HMI.b1000_05_AutoCycleStopPB THEN

			DS_HMI.iD100_MessageDisplay := 5;
			DS_HMI.sD100_MessageDisplay := 'Auto Cycle Stop...';

		END_IF

	ELSE
		DS_HMI.iD100_MessageDisplay := 6;
			DS_HMI.sD100_MessageDisplay := 'Alarm Occured, Please check Alarm Page for more detail';

	END_IF
END_ACTION

ACTION Other_LD:
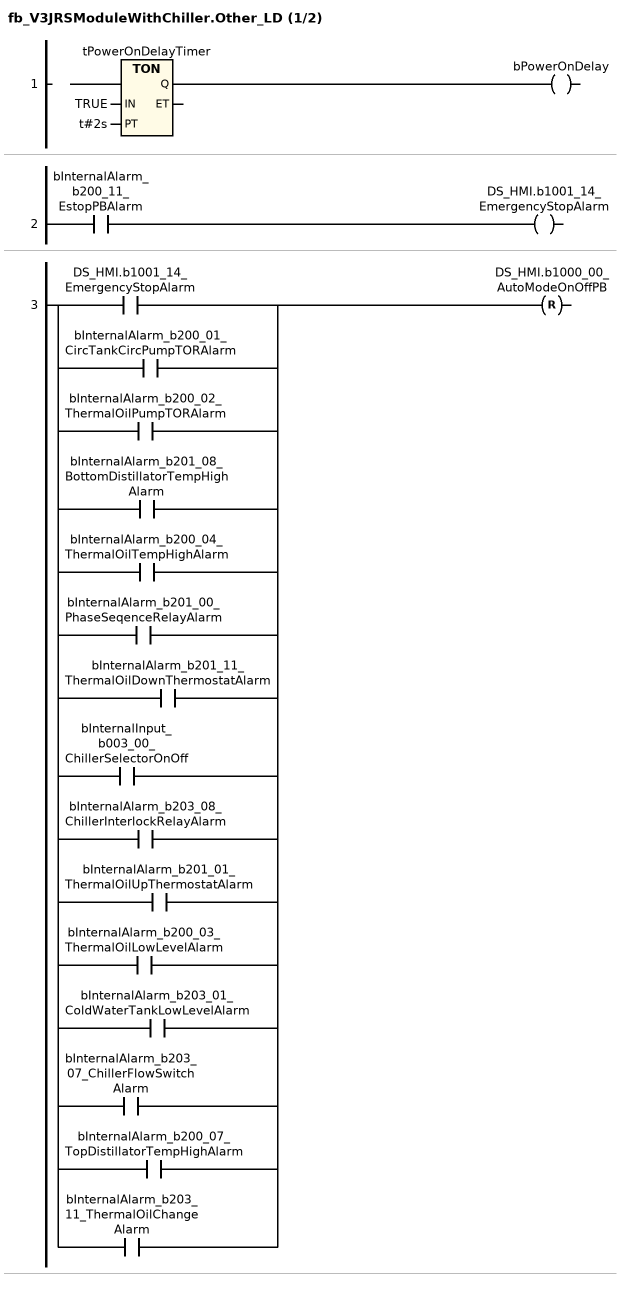
// NETWORK 1
tPowerOnDelayTimer(IN := TRUE, PT := t#2s); // TON
bPowerOnDelay := tPowerOnDelayTimer.Q;

// NETWORK 2
DS_HMI.b1001_14_EmergencyStopAlarm := bInternalAlarm_b200_11_EstopPBAlarm;

// NETWORK 3
DS_HMI.b1000_00_AutoModeOnOffPB R= DS_HMI.b1001_14_EmergencyStopAlarm OR bInternalAlarm_b200_01_CircTankCircPumpTORAlarm OR bInternalAlarm_b200_02_ThermalOilPumpTORAlarm OR bInternalAlarm_b201_08_BottomDistillatorTempHighAlarm OR bInternalAlarm_b200_04_ThermalOilTempHighAlarm OR bInternalAlarm_b201_00_PhaseSeqenceRelayAlarm OR bInternalAlarm_b201_11_ThermalOilDownThermostatAlarm OR bInternalInput_b003_00_ChillerSelectorOnOff OR bInternalAlarm_b203_08_ChillerInterlockRelayAlarm OR bInternalAlarm_b201_01_ThermalOilUpThermostatAlarm OR bInternalAlarm_b200_03_ThermalOilLowLevelAlarm OR bInternalAlarm_b203_01_ColdWaterTankLowLevelAlarm OR bInternalAlarm_b203_07_ChillerFlowSwitchAlarm OR bInternalAlarm_b200_07_TopDistillatorTempHighAlarm OR bInternalAlarm_b203_11_ThermalOilChangeAlarm;

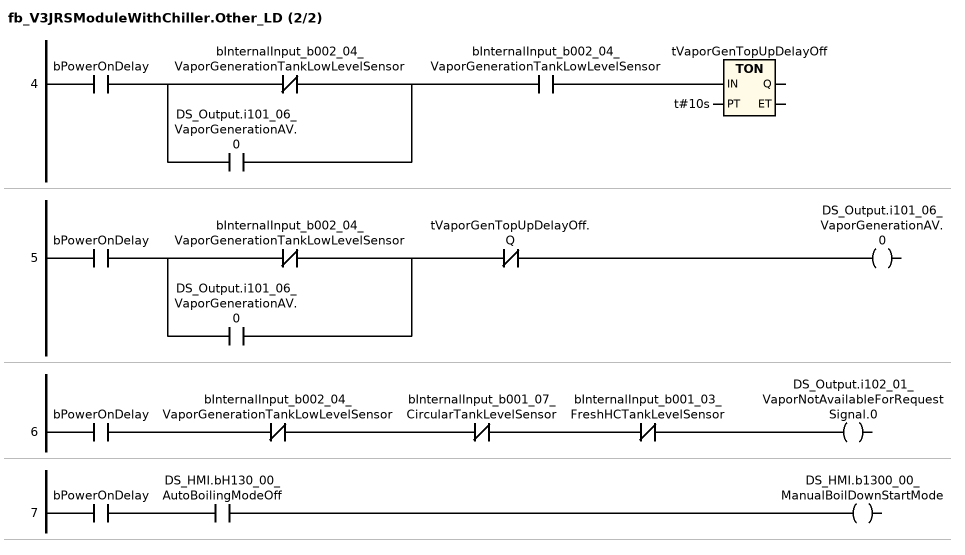
// NETWORK 4
tVaporGenTopUpDelayOff(IN := (bPowerOnDelay AND (NOT bInternalInput_b002_04_VaporGenerationTankLowLevelSensor OR DS_Output.i101_06_VaporGenerationAV.0)) AND bInternalInput_b002_04_VaporGenerationTankLowLevelSensor, PT := t#10s); // TON

// NETWORK 5
DS_Output.i101_06_VaporGenerationAV.0 := (bPowerOnDelay AND (NOT bInternalInput_b002_04_VaporGenerationTankLowLevelSensor OR DS_Output.i101_06_VaporGenerationAV.0)) AND NOT tVaporGenTopUpDelayOff.Q;

// NETWORK 6
DS_Output.i102_01_VaporNotAvailableForRequestSignal.0 := bPowerOnDelay AND NOT bInternalInput_b002_04_VaporGenerationTankLowLevelSensor AND NOT bInternalInput_b001_07_CircularTankLevelSensor AND NOT bInternalInput_b001_03_FreshHCTankLevelSensor;

// NETWORK 7
DS_HMI.b1300_00_ManualBoilDownStartMode := bPowerOnDelay AND DS_HMI.bH130_00_AutoBoilingModeOff;
END_ACTION

ACTION Other_ST:
	(*Map Alarm into Word so that can generate Alarm Occur Bit*)
	AriAlarmFlag[1].0 := bInternalAlarm_b200_00_FreshHCTankCircPumpTORAlarm ;
	AriAlarmFlag[1].1 := bInternalAlarm_b200_01_CircTankCircPumpTORAlarm ;
	AriAlarmFlag[1].2 := bInternalAlarm_b200_02_ThermalOilPumpTORAlarm ;
	AriAlarmFlag[1].3 := bInternalAlarm_b200_03_ThermalOilLowLevelAlarm ;
	AriAlarmFlag[1].4 := bInternalAlarm_b200_04_ThermalOilTempHighAlarm ;
	AriAlarmFlag[1].5 := bInternalAlarm_b200_05_ThermalOilTempNotReadyAlarm ;
	AriAlarmFlag[1].6 := bInternalAlarm_b200_06_ThermalOilHeaterOnOffAlarm ;
	AriAlarmFlag[1].7 := bInternalAlarm_b200_07_TopDistillatorTempHighAlarm ;
	AriAlarmFlag[1].8 := bInternalAlarm_b200_08_TopDistillatorTempNotReadyAlarm ;
	AriAlarmFlag[1].9 := bInternalAlarm_b200_09_TopDistillatorHeaterOnOffAlarm ;
	AriAlarmFlag[1].10 := bInternalAlarm_b200_10_RecycleStartStopPBAlarm ;
	AriAlarmFlag[1].11 := bInternalAlarm_b200_11_EstopPBAlarm ;
	
	AriAlarmFlag[2].0 := bInternalAlarm_b201_00_PhaseSeqenceRelayAlarm ;
	AriAlarmFlag[2].1 := bInternalAlarm_b201_01_ThermalOilUpThermostatAlarm ;
	AriAlarmFlag[2].2 := bInternalAlarm_b201_02_SludgeTankHighLevelAlarm ;
	AriAlarmFlag[2].3 := bInternalAlarm_b201_03_FreshHCTankLowLevelAlarm ;
	AriAlarmFlag[2].4 := bInternalAlarm_b201_04_VacuumNotAchieveAlarm ;
	AriAlarmFlag[2].5 := bInternalAlarm_b201_05_IncomingCDALowPressureAlarm ;
	AriAlarmFlag[2].6 := bInternalAlarm_b201_06_CoolingWaterLowFlowAlarm ;
	AriAlarmFlag[2].7 := bInternalAlarm_b201_07_CircularTankLowLevelAlarm ;
	AriAlarmFlag[2].8 := bInternalAlarm_b201_08_BottomDistillatorTempHighAlarm ;
	AriAlarmFlag[2].9 := bInternalAlarm_b201_09_BottomDistillatorTempNotReadyAlarm ;
	AriAlarmFlag[2].10 := bInternalAlarm_b201_10_BottomDistillatorHeaterOnOffAlarm ;
	AriAlarmFlag[2].11 := bInternalAlarm_b201_11_ThermalOilDownThermostatAlarm ;
	AriAlarmFlag[2].12 := bInternalAlarm_b201_12_ThermalOilMidThermostatAlarm ;

	AriAlarmFlag[3].0 := bInternalAlarm_b202_00_VaporGenerationTempHighAlarm ;
	AriAlarmFlag[3].1 := bInternalAlarm_b202_01_VaporGenerationTempNotReadyAlarm ;
	AriAlarmFlag[3].2 := bInternalAlarm_b202_02_VaporGenerationHeaterOnOffAlarm ;
	AriAlarmFlag[3].3 := bInternalAlarm_b202_03_WasteCollectionTankLowLevelAlarm ;
	AriAlarmFlag[3].4 := bInternalAlarm_b202_04_VaporGenerationTankLowLevelAlarm ;
	AriAlarmFlag[3].5 := bInternalAlarm_b202_05_HCPurgingAV3_1Alarm ;
	AriAlarmFlag[3].6 := bInternalAlarm_b202_06_MainMachineWasteTankLowLevelAlarm ;
	AriAlarmFlag[3].7 := bInternalAlarm_b202_07_MainMachineWasteTankHighLevelAlarm ;
	AriAlarmFlag[3].8 := bInternalAlarm_b202_08_ReservedAlarm ;
	AriAlarmFlag[3].9 := bInternalAlarm_b202_09_ReservedAlarm ;
	AriAlarmFlag[3].10 := bInternalAlarm_b202_10_ReservedAlarm ;
	AriAlarmFlag[3].11 := bInternalAlarm_b202_11_ReservedAlarm ;
	
	AriAlarmFlag[4].0 := bInternalAlarm_b203_00_ChillerSelectorOnOffAlarm ;
	AriAlarmFlag[4].1 := bInternalAlarm_b203_01_ColdWaterTankLowLevelAlarm ;
	AriAlarmFlag[4].2 := bInternalAlarm_b203_02_SludgeTankMissingAlarm ;
	AriAlarmFlag[4].3 := bInternalAlarm_b203_03_ColdWaterTankTempHighAlarm ;
	AriAlarmFlag[4].4 := bInternalAlarm_b203_04_ColdWaterTankTempNotReadyAlarm ;
	AriAlarmFlag[4].5 := bInternalAlarm_b203_05_ColdWaterTankHeaterOnOffAlarm ;
	AriAlarmFlag[4].6 := bInternalAlarm_b203_06_ChillerPumpTORAlarm ;
	AriAlarmFlag[4].7 := bInternalAlarm_b203_07_ChillerFlowSwitchAlarm ;
	AriAlarmFlag[4].8 := bInternalAlarm_b203_08_ChillerInterlockRelayAlarm ;
	AriAlarmFlag[4].9 := bInternalAlarm_b203_09_ReservedAlarm ;
	AriAlarmFlag[4].10 := bInternalAlarm_b203_10_ThermalOilChangeWarning ;
	AriAlarmFlag[4].11 := bInternalAlarm_b203_11_ThermalOilChangeAlarm ;
	
	
	IF AriAlarmFlag[1] <> 0
	OR AriAlarmFlag[2] <> 0
	OR AriAlarmFlag[3] <> 0
	OR AriAlarmFlag[4] <> 0
	THEN
	DS_HMI.b1001_15_AlarmOccur := TRUE;
	ELSE
	DS_HMI.b1001_15_AlarmOccur := FALSE;
	END_IF
END_ACTION

ACTION OutputCtrl_LD:
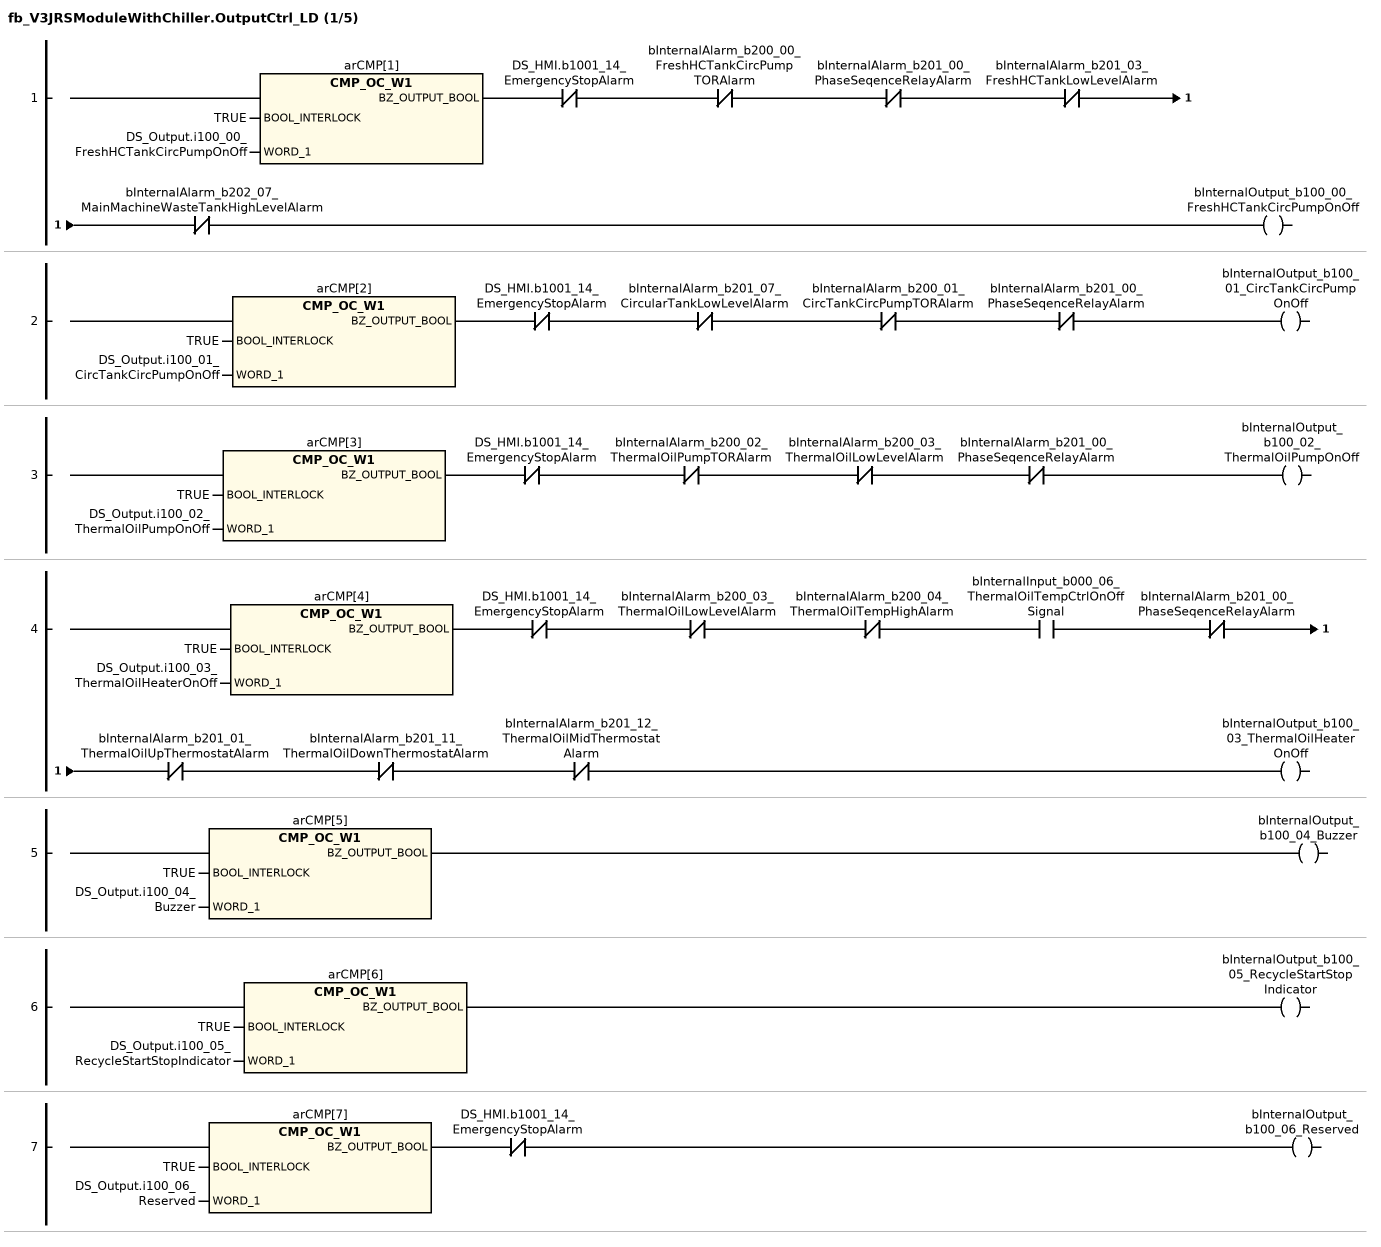
// NETWORK 1
arCMP[1](BOOL_INTERLOCK := TRUE, WORD_1 := DS_Output.i100_00_FreshHCTankCircPumpOnOff); // CMP_OC_W1
bInternalOutput_b100_00_FreshHCTankCircPumpOnOff := arCMP[1].BZ_OUTPUT_BOOL AND NOT DS_HMI.b1001_14_EmergencyStopAlarm AND NOT bInternalAlarm_b200_00_FreshHCTankCircPumpTORAlarm AND NOT bInternalAlarm_b201_00_PhaseSeqenceRelayAlarm AND NOT bInternalAlarm_b201_03_FreshHCTankLowLevelAlarm AND NOT bInternalAlarm_b202_07_MainMachineWasteTankHighLevelAlarm;

// NETWORK 2
arCMP[2](BOOL_INTERLOCK := TRUE, WORD_1 := DS_Output.i100_01_CircTankCircPumpOnOff); // CMP_OC_W1
bInternalOutput_b100_01_CircTankCircPumpOnOff := arCMP[2].BZ_OUTPUT_BOOL AND NOT DS_HMI.b1001_14_EmergencyStopAlarm AND NOT bInternalAlarm_b201_07_CircularTankLowLevelAlarm AND NOT bInternalAlarm_b200_01_CircTankCircPumpTORAlarm AND NOT bInternalAlarm_b201_00_PhaseSeqenceRelayAlarm;

// NETWORK 3
arCMP[3](BOOL_INTERLOCK := TRUE, WORD_1 := DS_Output.i100_02_ThermalOilPumpOnOff); // CMP_OC_W1
bInternalOutput_b100_02_ThermalOilPumpOnOff := arCMP[3].BZ_OUTPUT_BOOL AND NOT DS_HMI.b1001_14_EmergencyStopAlarm AND NOT bInternalAlarm_b200_02_ThermalOilPumpTORAlarm AND NOT bInternalAlarm_b200_03_ThermalOilLowLevelAlarm AND NOT bInternalAlarm_b201_00_PhaseSeqenceRelayAlarm;

// NETWORK 4
arCMP[4](BOOL_INTERLOCK := TRUE, WORD_1 := DS_Output.i100_03_ThermalOilHeaterOnOff); // CMP_OC_W1
bInternalOutput_b100_03_ThermalOilHeaterOnOff := arCMP[4].BZ_OUTPUT_BOOL AND NOT DS_HMI.b1001_14_EmergencyStopAlarm AND NOT bInternalAlarm_b200_03_ThermalOilLowLevelAlarm AND NOT bInternalAlarm_b200_04_ThermalOilTempHighAlarm AND bInternalInput_b000_06_ThermalOilTempCtrlOnOffSignal AND NOT bInternalAlarm_b201_00_PhaseSeqenceRelayAlarm AND NOT bInternalAlarm_b201_01_ThermalOilUpThermostatAlarm AND NOT bInternalAlarm_b201_11_ThermalOilDownThermostatAlarm AND NOT bInternalAlarm_b201_12_ThermalOilMidThermostatAlarm;

// NETWORK 5
arCMP[5](BOOL_INTERLOCK := TRUE, WORD_1 := DS_Output.i100_04_Buzzer); // CMP_OC_W1
bInternalOutput_b100_04_Buzzer := arCMP[5].BZ_OUTPUT_BOOL;

// NETWORK 6
arCMP[6](BOOL_INTERLOCK := TRUE, WORD_1 := DS_Output.i100_05_RecycleStartStopIndicator); // CMP_OC_W1
bInternalOutput_b100_05_RecycleStartStopIndicator := arCMP[6].BZ_OUTPUT_BOOL;

// NETWORK 7
arCMP[7](BOOL_INTERLOCK := TRUE, WORD_1 := DS_Output.i100_06_Reserved); // CMP_OC_W1
bInternalOutput_b100_06_Reserved := arCMP[7].BZ_OUTPUT_BOOL AND NOT DS_HMI.b1001_14_EmergencyStopAlarm;

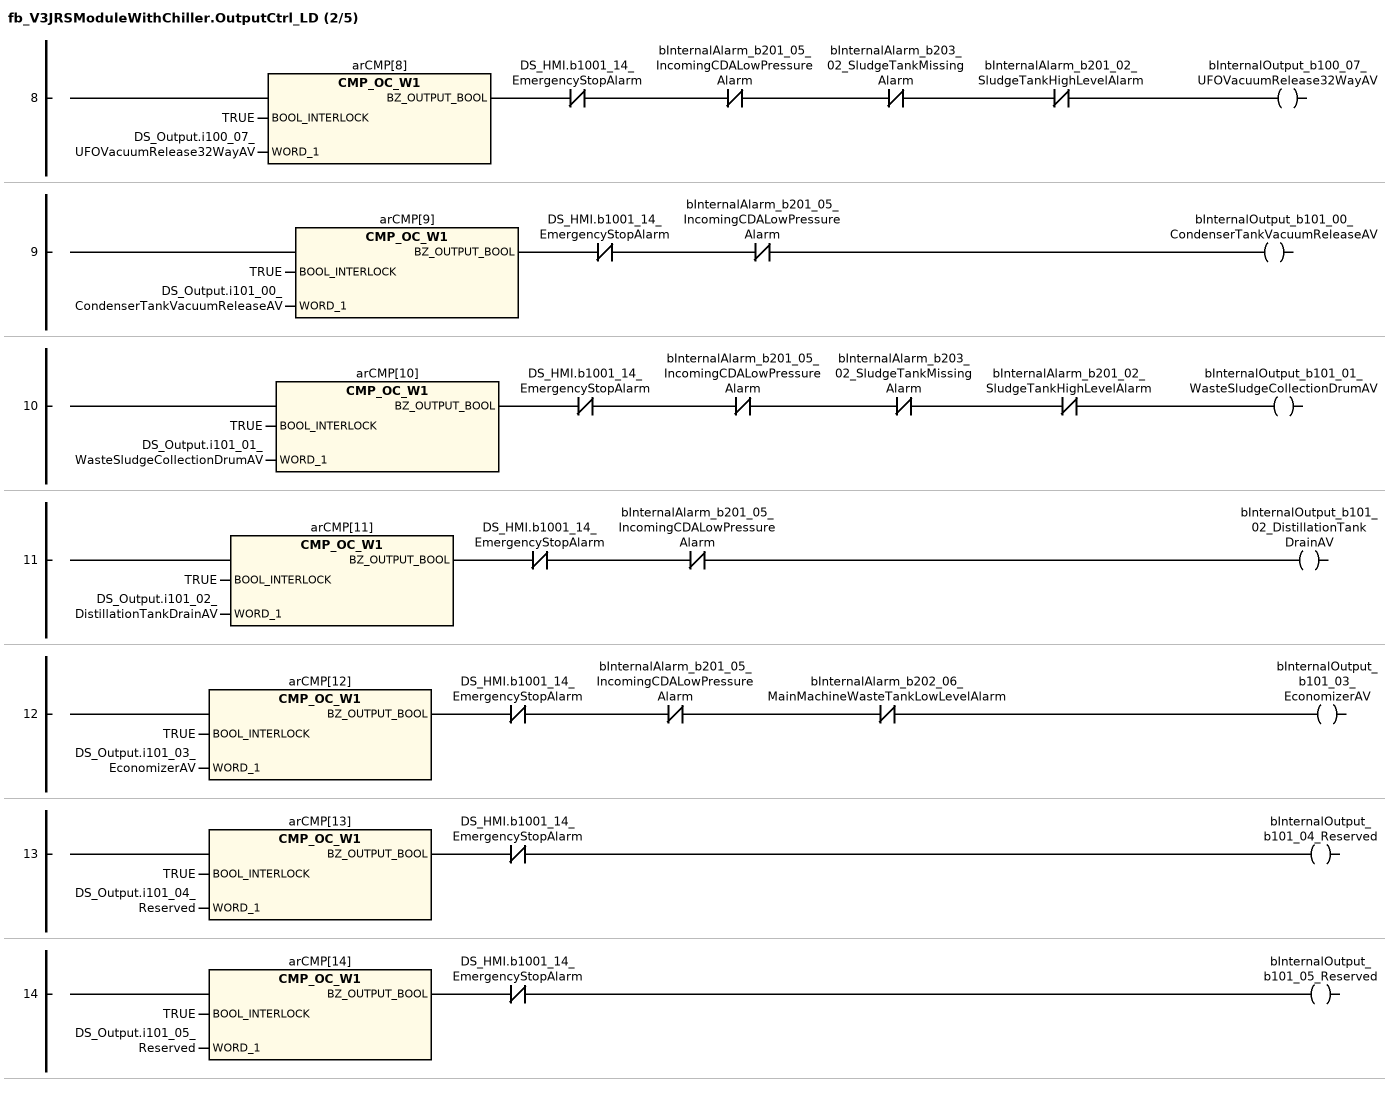
// NETWORK 8
arCMP[8](BOOL_INTERLOCK := TRUE, WORD_1 := DS_Output.i100_07_UFOVacuumRelease32WayAV); // CMP_OC_W1
bInternalOutput_b100_07_UFOVacuumRelease32WayAV := arCMP[8].BZ_OUTPUT_BOOL AND NOT DS_HMI.b1001_14_EmergencyStopAlarm AND NOT bInternalAlarm_b201_05_IncomingCDALowPressureAlarm AND NOT bInternalAlarm_b203_02_SludgeTankMissingAlarm AND NOT bInternalAlarm_b201_02_SludgeTankHighLevelAlarm;

// NETWORK 9
arCMP[9](BOOL_INTERLOCK := TRUE, WORD_1 := DS_Output.i101_00_CondenserTankVacuumReleaseAV); // CMP_OC_W1
bInternalOutput_b101_00_CondenserTankVacuumReleaseAV := arCMP[9].BZ_OUTPUT_BOOL AND NOT DS_HMI.b1001_14_EmergencyStopAlarm AND NOT bInternalAlarm_b201_05_IncomingCDALowPressureAlarm;

// NETWORK 10
arCMP[10](BOOL_INTERLOCK := TRUE, WORD_1 := DS_Output.i101_01_WasteSludgeCollectionDrumAV); // CMP_OC_W1
bInternalOutput_b101_01_WasteSludgeCollectionDrumAV := arCMP[10].BZ_OUTPUT_BOOL AND NOT DS_HMI.b1001_14_EmergencyStopAlarm AND NOT bInternalAlarm_b201_05_IncomingCDALowPressureAlarm AND NOT bInternalAlarm_b203_02_SludgeTankMissingAlarm AND NOT bInternalAlarm_b201_02_SludgeTankHighLevelAlarm;

// NETWORK 11
arCMP[11](BOOL_INTERLOCK := TRUE, WORD_1 := DS_Output.i101_02_DistillationTankDrainAV); // CMP_OC_W1
bInternalOutput_b101_02_DistillationTankDrainAV := arCMP[11].BZ_OUTPUT_BOOL AND NOT DS_HMI.b1001_14_EmergencyStopAlarm AND NOT bInternalAlarm_b201_05_IncomingCDALowPressureAlarm;

// NETWORK 12
arCMP[12](BOOL_INTERLOCK := TRUE, WORD_1 := DS_Output.i101_03_EconomizerAV); // CMP_OC_W1
bInternalOutput_b101_03_EconomizerAV := arCMP[12].BZ_OUTPUT_BOOL AND NOT DS_HMI.b1001_14_EmergencyStopAlarm AND NOT bInternalAlarm_b201_05_IncomingCDALowPressureAlarm AND NOT bInternalAlarm_b202_06_MainMachineWasteTankLowLevelAlarm;

// NETWORK 13
arCMP[13](BOOL_INTERLOCK := TRUE, WORD_1 := DS_Output.i101_04_Reserved); // CMP_OC_W1
bInternalOutput_b101_04_Reserved := arCMP[13].BZ_OUTPUT_BOOL AND NOT DS_HMI.b1001_14_EmergencyStopAlarm;

// NETWORK 14
arCMP[14](BOOL_INTERLOCK := TRUE, WORD_1 := DS_Output.i101_05_Reserved); // CMP_OC_W1
bInternalOutput_b101_05_Reserved := arCMP[14].BZ_OUTPUT_BOOL AND NOT DS_HMI.b1001_14_EmergencyStopAlarm;

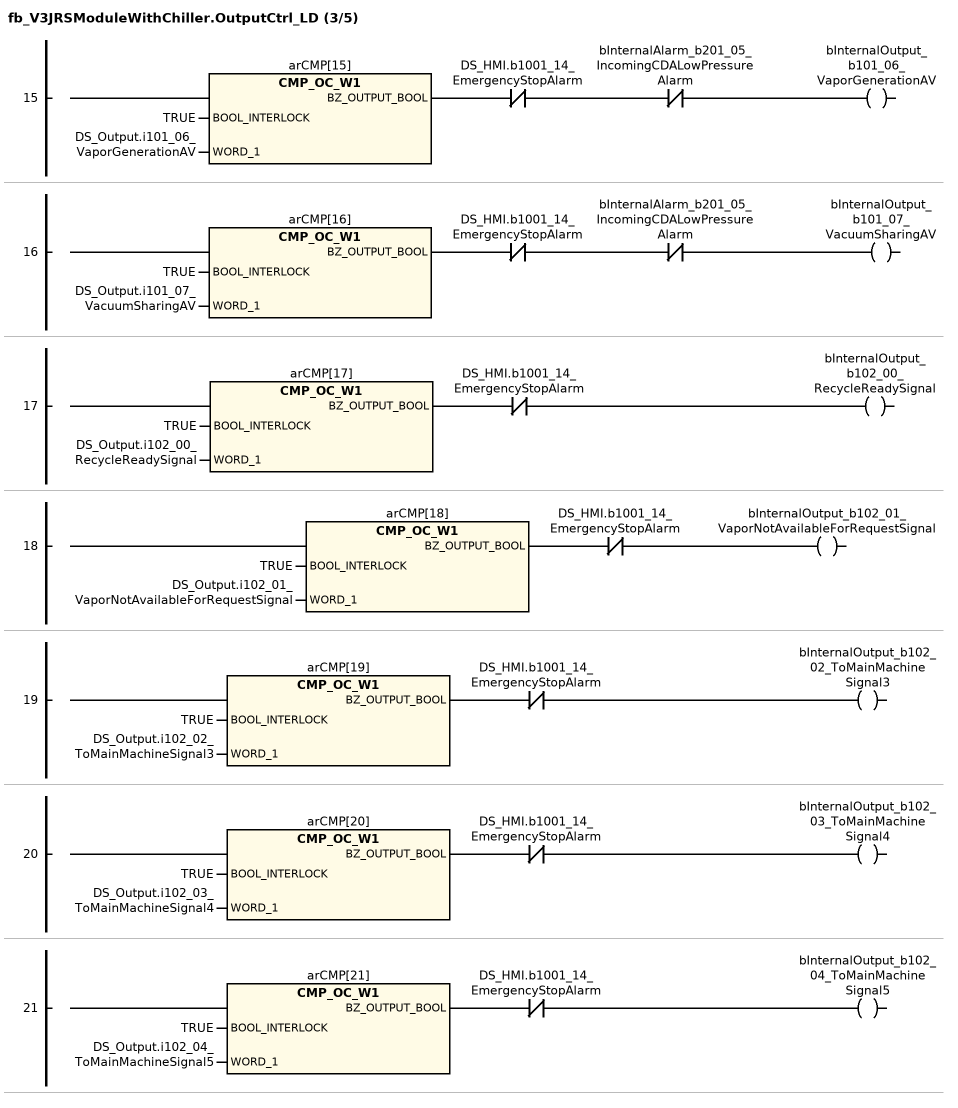
// NETWORK 15
arCMP[15](BOOL_INTERLOCK := TRUE, WORD_1 := DS_Output.i101_06_VaporGenerationAV); // CMP_OC_W1
bInternalOutput_b101_06_VaporGenerationAV := arCMP[15].BZ_OUTPUT_BOOL AND NOT DS_HMI.b1001_14_EmergencyStopAlarm AND NOT bInternalAlarm_b201_05_IncomingCDALowPressureAlarm;

// NETWORK 16
arCMP[16](BOOL_INTERLOCK := TRUE, WORD_1 := DS_Output.i101_07_VacuumSharingAV); // CMP_OC_W1
bInternalOutput_b101_07_VacuumSharingAV := arCMP[16].BZ_OUTPUT_BOOL AND NOT DS_HMI.b1001_14_EmergencyStopAlarm AND NOT bInternalAlarm_b201_05_IncomingCDALowPressureAlarm;

// NETWORK 17
arCMP[17](BOOL_INTERLOCK := TRUE, WORD_1 := DS_Output.i102_00_RecycleReadySignal); // CMP_OC_W1
bInternalOutput_b102_00_RecycleReadySignal := arCMP[17].BZ_OUTPUT_BOOL AND NOT DS_HMI.b1001_14_EmergencyStopAlarm;

// NETWORK 18
arCMP[18](BOOL_INTERLOCK := TRUE, WORD_1 := DS_Output.i102_01_VaporNotAvailableForRequestSignal); // CMP_OC_W1
bInternalOutput_b102_01_VaporNotAvailableForRequestSignal := arCMP[18].BZ_OUTPUT_BOOL AND NOT DS_HMI.b1001_14_EmergencyStopAlarm;

// NETWORK 19
arCMP[19](BOOL_INTERLOCK := TRUE, WORD_1 := DS_Output.i102_02_ToMainMachineSignal3); // CMP_OC_W1
bInternalOutput_b102_02_ToMainMachineSignal3 := arCMP[19].BZ_OUTPUT_BOOL AND NOT DS_HMI.b1001_14_EmergencyStopAlarm;

// NETWORK 20
arCMP[20](BOOL_INTERLOCK := TRUE, WORD_1 := DS_Output.i102_03_ToMainMachineSignal4); // CMP_OC_W1
bInternalOutput_b102_03_ToMainMachineSignal4 := arCMP[20].BZ_OUTPUT_BOOL AND NOT DS_HMI.b1001_14_EmergencyStopAlarm;

// NETWORK 21
arCMP[21](BOOL_INTERLOCK := TRUE, WORD_1 := DS_Output.i102_04_ToMainMachineSignal5); // CMP_OC_W1
bInternalOutput_b102_04_ToMainMachineSignal5 := arCMP[21].BZ_OUTPUT_BOOL AND NOT DS_HMI.b1001_14_EmergencyStopAlarm;

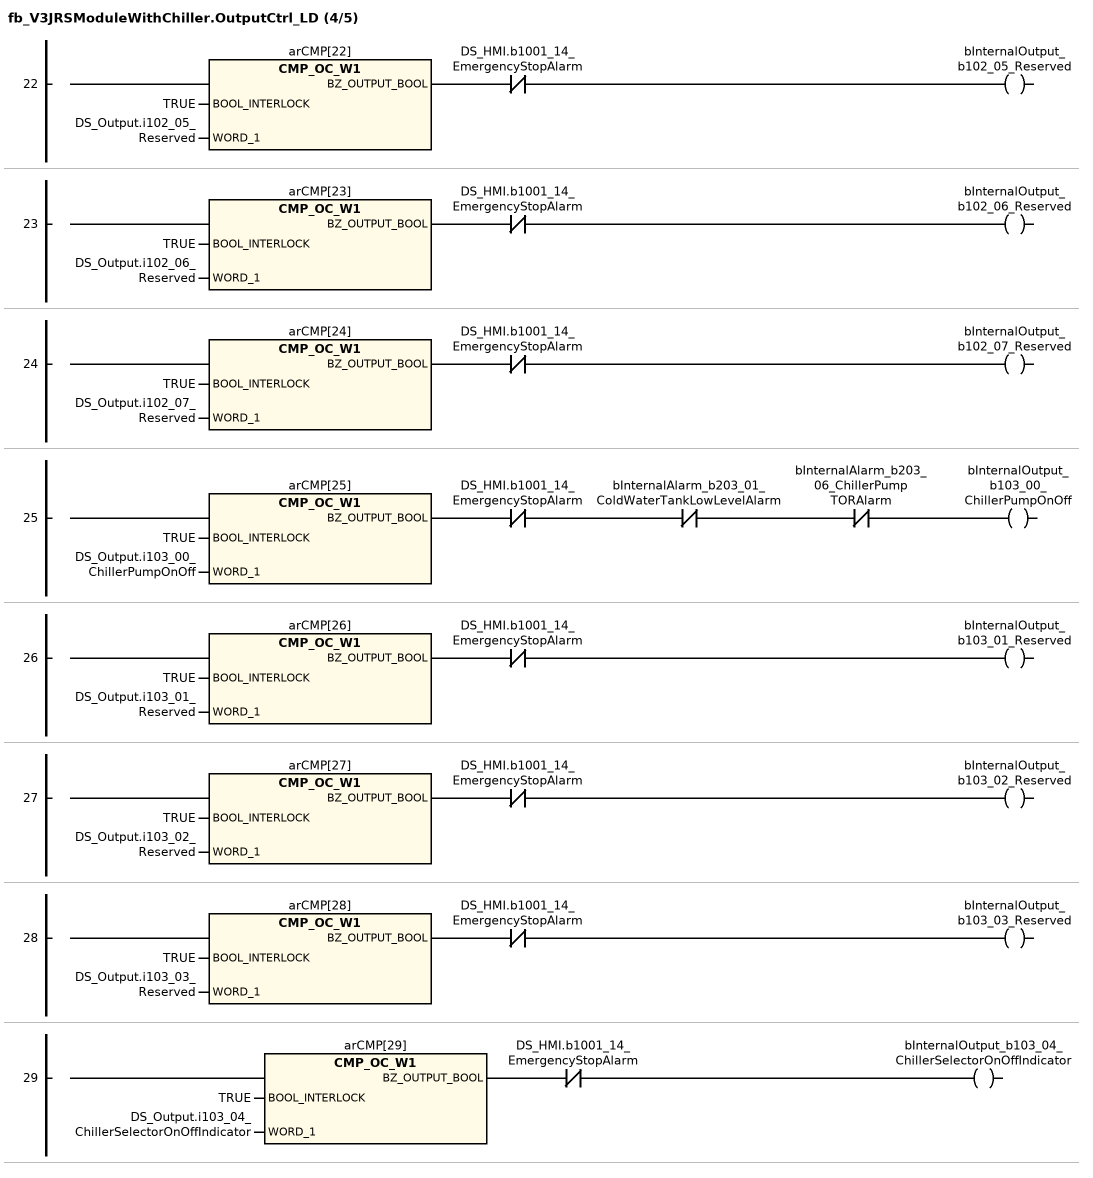
// NETWORK 22
arCMP[22](BOOL_INTERLOCK := TRUE, WORD_1 := DS_Output.i102_05_Reserved); // CMP_OC_W1
bInternalOutput_b102_05_Reserved := arCMP[22].BZ_OUTPUT_BOOL AND NOT DS_HMI.b1001_14_EmergencyStopAlarm;

// NETWORK 23
arCMP[23](BOOL_INTERLOCK := TRUE, WORD_1 := DS_Output.i102_06_Reserved); // CMP_OC_W1
bInternalOutput_b102_06_Reserved := arCMP[23].BZ_OUTPUT_BOOL AND NOT DS_HMI.b1001_14_EmergencyStopAlarm;

// NETWORK 24
arCMP[24](BOOL_INTERLOCK := TRUE, WORD_1 := DS_Output.i102_07_Reserved); // CMP_OC_W1
bInternalOutput_b102_07_Reserved := arCMP[24].BZ_OUTPUT_BOOL AND NOT DS_HMI.b1001_14_EmergencyStopAlarm;

// NETWORK 25
arCMP[25](BOOL_INTERLOCK := TRUE, WORD_1 := DS_Output.i103_00_ChillerPumpOnOff); // CMP_OC_W1
bInternalOutput_b103_00_ChillerPumpOnOff := arCMP[25].BZ_OUTPUT_BOOL AND NOT DS_HMI.b1001_14_EmergencyStopAlarm AND NOT bInternalAlarm_b203_01_ColdWaterTankLowLevelAlarm AND NOT bInternalAlarm_b203_06_ChillerPumpTORAlarm;

// NETWORK 26
arCMP[26](BOOL_INTERLOCK := TRUE, WORD_1 := DS_Output.i103_01_Reserved); // CMP_OC_W1
bInternalOutput_b103_01_Reserved := arCMP[26].BZ_OUTPUT_BOOL AND NOT DS_HMI.b1001_14_EmergencyStopAlarm;

// NETWORK 27
arCMP[27](BOOL_INTERLOCK := TRUE, WORD_1 := DS_Output.i103_02_Reserved); // CMP_OC_W1
bInternalOutput_b103_02_Reserved := arCMP[27].BZ_OUTPUT_BOOL AND NOT DS_HMI.b1001_14_EmergencyStopAlarm;

// NETWORK 28
arCMP[28](BOOL_INTERLOCK := TRUE, WORD_1 := DS_Output.i103_03_Reserved); // CMP_OC_W1
bInternalOutput_b103_03_Reserved := arCMP[28].BZ_OUTPUT_BOOL AND NOT DS_HMI.b1001_14_EmergencyStopAlarm;

// NETWORK 29
arCMP[29](BOOL_INTERLOCK := TRUE, WORD_1 := DS_Output.i103_04_ChillerSelectorOnOffIndicator); // CMP_OC_W1
bInternalOutput_b103_04_ChillerSelectorOnOffIndicator := arCMP[29].BZ_OUTPUT_BOOL AND NOT DS_HMI.b1001_14_EmergencyStopAlarm;

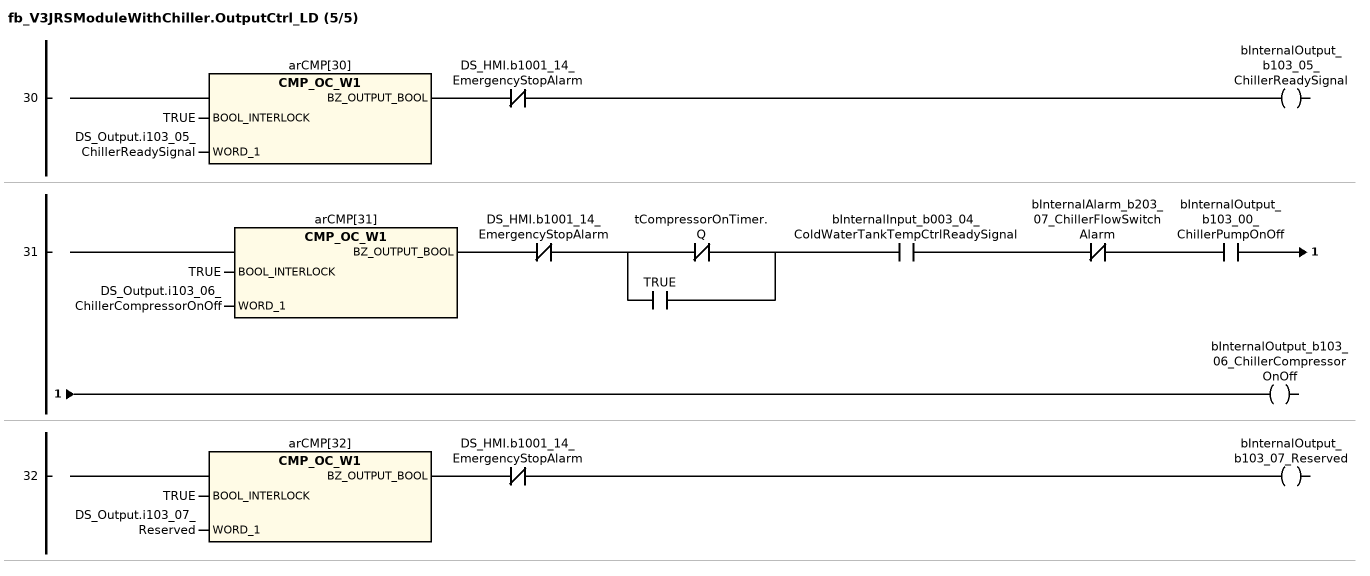
// NETWORK 30
arCMP[30](BOOL_INTERLOCK := TRUE, WORD_1 := DS_Output.i103_05_ChillerReadySignal); // CMP_OC_W1
bInternalOutput_b103_05_ChillerReadySignal := arCMP[30].BZ_OUTPUT_BOOL AND NOT DS_HMI.b1001_14_EmergencyStopAlarm;

// NETWORK 31
arCMP[31](BOOL_INTERLOCK := TRUE, WORD_1 := DS_Output.i103_06_ChillerCompressorOnOff); // CMP_OC_W1
bInternalOutput_b103_06_ChillerCompressorOnOff := (arCMP[31].BZ_OUTPUT_BOOL AND NOT DS_HMI.b1001_14_EmergencyStopAlarm AND (NOT tCompressorOnTimer.Q OR TRUE)) AND bInternalInput_b003_04_ColdWaterTankTempCtrlReadySignal AND NOT bInternalAlarm_b203_07_ChillerFlowSwitchAlarm AND bInternalOutput_b103_00_ChillerPumpOnOff;

// NETWORK 32
arCMP[32](BOOL_INTERLOCK := TRUE, WORD_1 := DS_Output.i103_07_Reserved); // CMP_OC_W1
bInternalOutput_b103_07_Reserved := arCMP[32].BZ_OUTPUT_BOOL AND NOT DS_HMI.b1001_14_EmergencyStopAlarm;
END_ACTION

ACTION SystemRestore_LD:
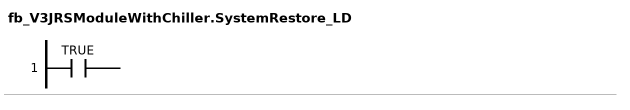
// NETWORK 1
END_ACTION

ACTION ThermalOilChangeHRMeter_ST:
	(*ThermalOilChange Hour Meter Counting*)
	IF bInternalOutput_b100_02_ThermalOilPumpOnOff AND t1SecCPRE.Q THEN

		DS_HMI.iD242_ThermalOilChangeHMeterPV_Sec := DS_HMI.iD242_ThermalOilChangeHMeterPV_Sec +1;
	
		IF DS_HMI.iD242_ThermalOilChangeHMeterPV_Sec > 59 THEN
			DS_HMI.iD241_ThermalOilChangeHMeterPV_Min := DS_HMI.iD241_ThermalOilChangeHMeterPV_Min +1;
			DS_HMI.iD242_ThermalOilChangeHMeterPV_Sec := 0;
		END_IF
	
		IF DS_HMI.iD241_ThermalOilChangeHMeterPV_Min > 59 THEN
			DS_HMI.iD240_ThermalOilChangeHMeterPV_Hour := DS_HMI.iD240_ThermalOilChangeHMeterPV_Hour +1;
			DS_HMI.iD241_ThermalOilChangeHMeterPV_Min := 0;
		END_IF

	END_IF
	

	(*ThermalOilChange Hour Meter Warning and Alarm*)
	IF DS_HMI.iD240_ThermalOilChangeHMeterPV_Hour >= DS_HMI.iD251_ThermalOilChangeAlarmSV_Hour THEN
	DS_HMI.b1040_00_ThermalOilChangeHMeterAlarm := TRUE;
	ELSE
	DS_HMI.b1040_00_ThermalOilChangeHMeterAlarm := FALSE;
	END_IF

	IF DS_HMI.iD240_ThermalOilChangeHMeterPV_Hour >= DS_HMI.iD250_ThermalOilChangeWarningSV_Hour THEN
	DS_HMI.b1040_02_ThermalOiChangeWarning := TRUE;
	ELSE
	DS_HMI.b1040_02_ThermalOiChangeWarning := FALSE;
	END_IF

	(*ThermalOilChange Hour Meter Reset*)
	tThermalOilChangeResetPBTimer(IN:=DS_HMI.b1040_01_ThermalOilChangeHMeterResetPB , PT:=t#3s , Q=> , ET=> );
	IF tThermalOilChangeResetPBTimer.Q THEN

		DS_HMI.iD242_ThermalOilChangeHMeterPV_Sec	:= 0;
		DS_HMI.iD241_ThermalOilChangeHMeterPV_Min	:= 0;
		DS_HMI.iD240_ThermalOilChangeHMeterPV_Hour	:= 0;
	END_IF
END_ACTION

ACTION Z_BuiltInTempCtrl_LD:
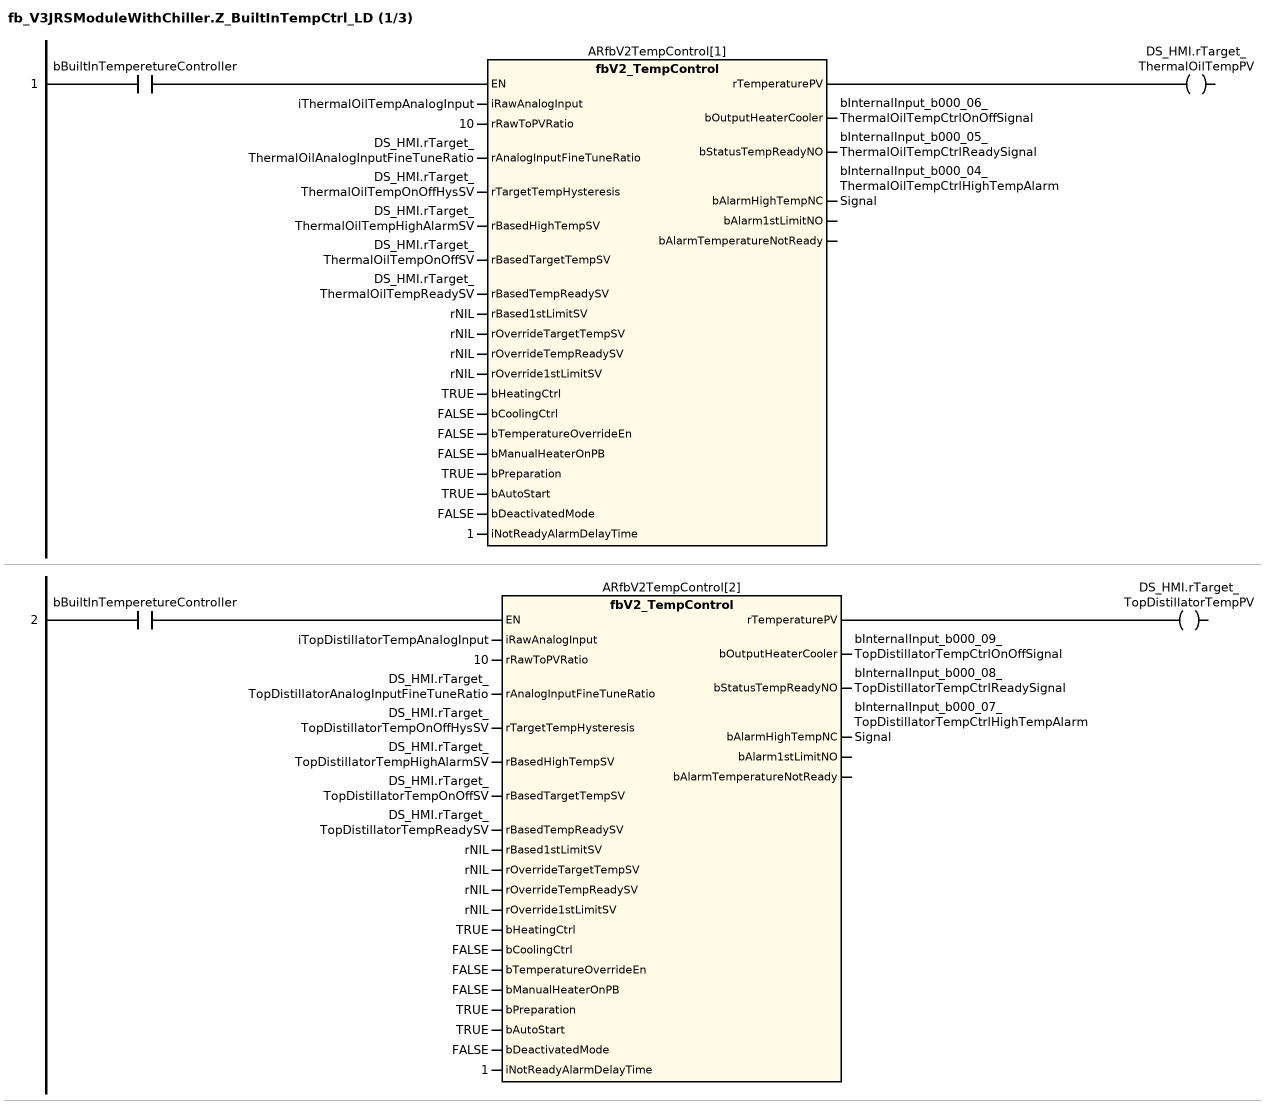
// NETWORK 1
IF bBuiltInTemperetureController THEN
    ARfbV2TempControl[1](
        iRawAnalogInput := iThermalOilTempAnalogInput,
        rRawToPVRatio := 10,
        rAnalogInputFineTuneRatio := DS_HMI.rTarget_ThermalOilAnalogInputFineTuneRatio,
        rTargetTempHysteresis := DS_HMI.rTarget_ThermalOilTempOnOffHysSV,
        rBasedHighTempSV := DS_HMI.rTarget_ThermalOilTempHighAlarmSV,
        rBasedTargetTempSV := DS_HMI.rTarget_ThermalOilTempOnOffSV,
        rBasedTempReadySV := DS_HMI.rTarget_ThermalOilTempReadySV,
        rBased1stLimitSV := rNIL,
        rOverrideTargetTempSV := rNIL,
        rOverrideTempReadySV := rNIL,
        rOverride1stLimitSV := rNIL,
        bHeatingCtrl := TRUE,
        bCoolingCtrl := FALSE,
        bTemperatureOverrideEn := FALSE,
        bManualHeaterOnPB := FALSE,
        bPreparation := TRUE,
        bAutoStart := TRUE,
        bDeactivatedMode := FALSE,
        iNotReadyAlarmDelayTime := 1,
        bOutputHeaterCooler => bInternalInput_b000_06_ThermalOilTempCtrlOnOffSignal,
        bStatusTempReadyNO => bInternalInput_b000_05_ThermalOilTempCtrlReadySignal,
        bAlarmHighTempNC => bInternalInput_b000_04_ThermalOilTempCtrlHighTempAlarmSignal); // fbV2_TempControl
END_IF
DS_HMI.rTarget_ThermalOilTempPV := ARfbV2TempControl[1].rTemperaturePV;

// NETWORK 2
IF bBuiltInTemperetureController THEN
    ARfbV2TempControl[2](
        iRawAnalogInput := iTopDistillatorTempAnalogInput,
        rRawToPVRatio := 10,
        rAnalogInputFineTuneRatio := DS_HMI.rTarget_TopDistillatorAnalogInputFineTuneRatio,
        rTargetTempHysteresis := DS_HMI.rTarget_TopDistillatorTempOnOffHysSV,
        rBasedHighTempSV := DS_HMI.rTarget_TopDistillatorTempHighAlarmSV,
        rBasedTargetTempSV := DS_HMI.rTarget_TopDistillatorTempOnOffSV,
        rBasedTempReadySV := DS_HMI.rTarget_TopDistillatorTempReadySV,
        rBased1stLimitSV := rNIL,
        rOverrideTargetTempSV := rNIL,
        rOverrideTempReadySV := rNIL,
        rOverride1stLimitSV := rNIL,
        bHeatingCtrl := TRUE,
        bCoolingCtrl := FALSE,
        bTemperatureOverrideEn := FALSE,
        bManualHeaterOnPB := FALSE,
        bPreparation := TRUE,
        bAutoStart := TRUE,
        bDeactivatedMode := FALSE,
        iNotReadyAlarmDelayTime := 1,
        bOutputHeaterCooler => bInternalInput_b000_09_TopDistillatorTempCtrlOnOffSignal,
        bStatusTempReadyNO => bInternalInput_b000_08_TopDistillatorTempCtrlReadySignal,
        bAlarmHighTempNC => bInternalInput_b000_07_TopDistillatorTempCtrlHighTempAlarmSignal); // fbV2_TempControl
END_IF
DS_HMI.rTarget_TopDistillatorTempPV := ARfbV2TempControl[2].rTemperaturePV;

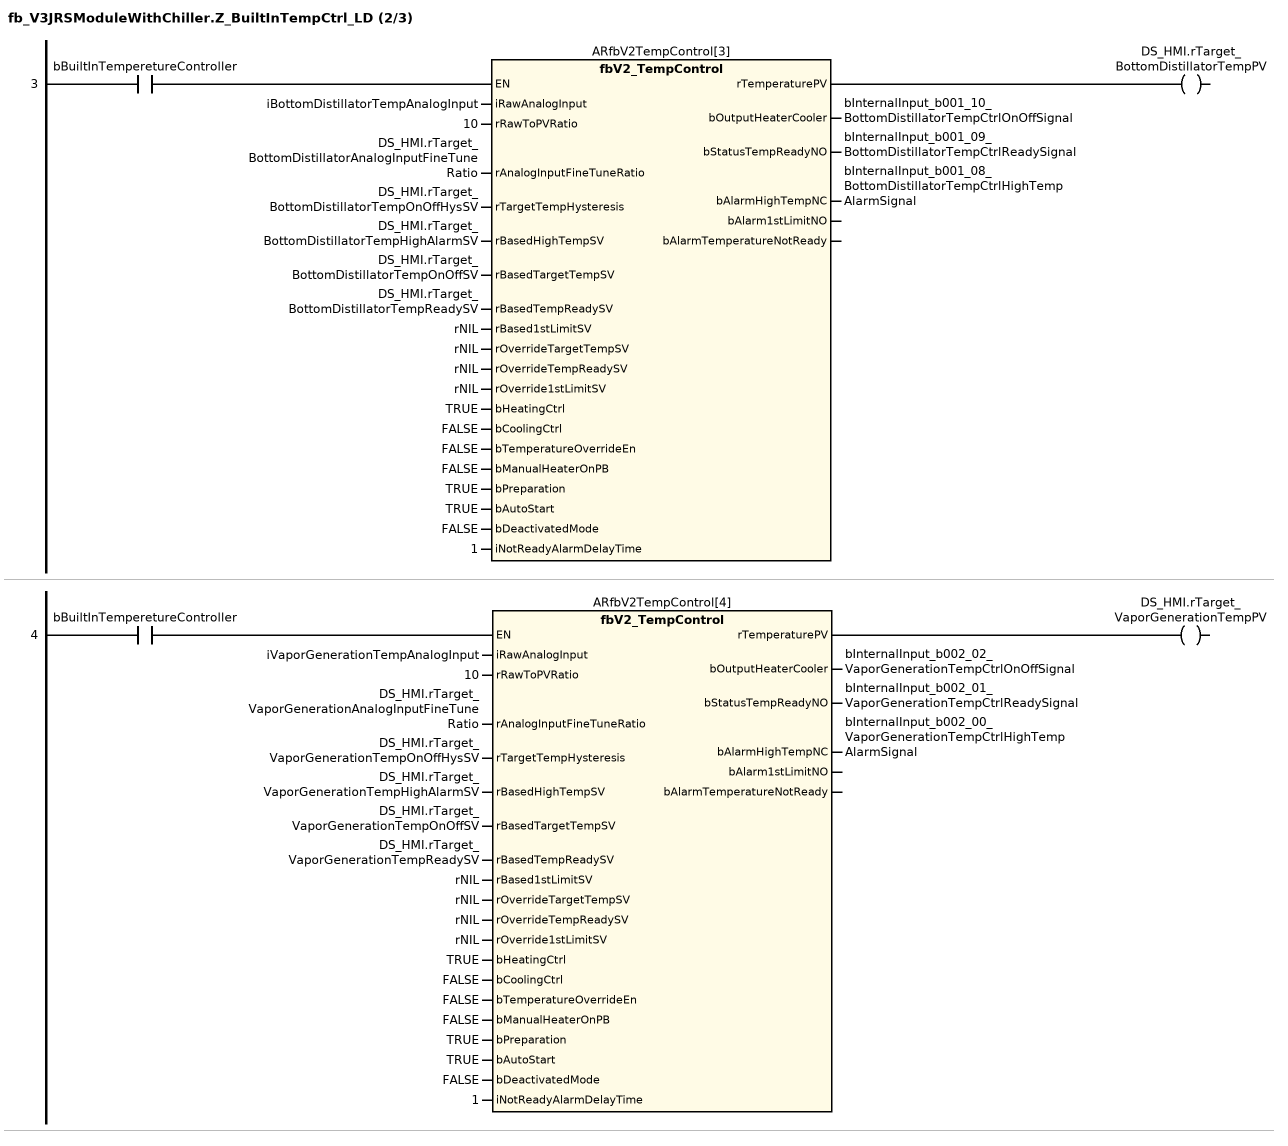
// NETWORK 3
IF bBuiltInTemperetureController THEN
    ARfbV2TempControl[3](
        iRawAnalogInput := iBottomDistillatorTempAnalogInput,
        rRawToPVRatio := 10,
        rAnalogInputFineTuneRatio := DS_HMI.rTarget_BottomDistillatorAnalogInputFineTuneRatio,
        rTargetTempHysteresis := DS_HMI.rTarget_BottomDistillatorTempOnOffHysSV,
        rBasedHighTempSV := DS_HMI.rTarget_BottomDistillatorTempHighAlarmSV,
        rBasedTargetTempSV := DS_HMI.rTarget_BottomDistillatorTempOnOffSV,
        rBasedTempReadySV := DS_HMI.rTarget_BottomDistillatorTempReadySV,
        rBased1stLimitSV := rNIL,
        rOverrideTargetTempSV := rNIL,
        rOverrideTempReadySV := rNIL,
        rOverride1stLimitSV := rNIL,
        bHeatingCtrl := TRUE,
        bCoolingCtrl := FALSE,
        bTemperatureOverrideEn := FALSE,
        bManualHeaterOnPB := FALSE,
        bPreparation := TRUE,
        bAutoStart := TRUE,
        bDeactivatedMode := FALSE,
        iNotReadyAlarmDelayTime := 1,
        bOutputHeaterCooler => bInternalInput_b001_10_BottomDistillatorTempCtrlOnOffSignal,
        bStatusTempReadyNO => bInternalInput_b001_09_BottomDistillatorTempCtrlReadySignal,
        bAlarmHighTempNC => bInternalInput_b001_08_BottomDistillatorTempCtrlHighTempAlarmSignal); // fbV2_TempControl
END_IF
DS_HMI.rTarget_BottomDistillatorTempPV := ARfbV2TempControl[3].rTemperaturePV;

// NETWORK 4
IF bBuiltInTemperetureController THEN
    ARfbV2TempControl[4](
        iRawAnalogInput := iVaporGenerationTempAnalogInput,
        rRawToPVRatio := 10,
        rAnalogInputFineTuneRatio := DS_HMI.rTarget_VaporGenerationAnalogInputFineTuneRatio,
        rTargetTempHysteresis := DS_HMI.rTarget_VaporGenerationTempOnOffHysSV,
        rBasedHighTempSV := DS_HMI.rTarget_VaporGenerationTempHighAlarmSV,
        rBasedTargetTempSV := DS_HMI.rTarget_VaporGenerationTempOnOffSV,
        rBasedTempReadySV := DS_HMI.rTarget_VaporGenerationTempReadySV,
        rBased1stLimitSV := rNIL,
        rOverrideTargetTempSV := rNIL,
        rOverrideTempReadySV := rNIL,
        rOverride1stLimitSV := rNIL,
        bHeatingCtrl := TRUE,
        bCoolingCtrl := FALSE,
        bTemperatureOverrideEn := FALSE,
        bManualHeaterOnPB := FALSE,
        bPreparation := TRUE,
        bAutoStart := TRUE,
        bDeactivatedMode := FALSE,
        iNotReadyAlarmDelayTime := 1,
        bOutputHeaterCooler => bInternalInput_b002_02_VaporGenerationTempCtrlOnOffSignal,
        bStatusTempReadyNO => bInternalInput_b002_01_VaporGenerationTempCtrlReadySignal,
        bAlarmHighTempNC => bInternalInput_b002_00_VaporGenerationTempCtrlHighTempAlarmSignal); // fbV2_TempControl
END_IF
DS_HMI.rTarget_VaporGenerationTempPV := ARfbV2TempControl[4].rTemperaturePV;

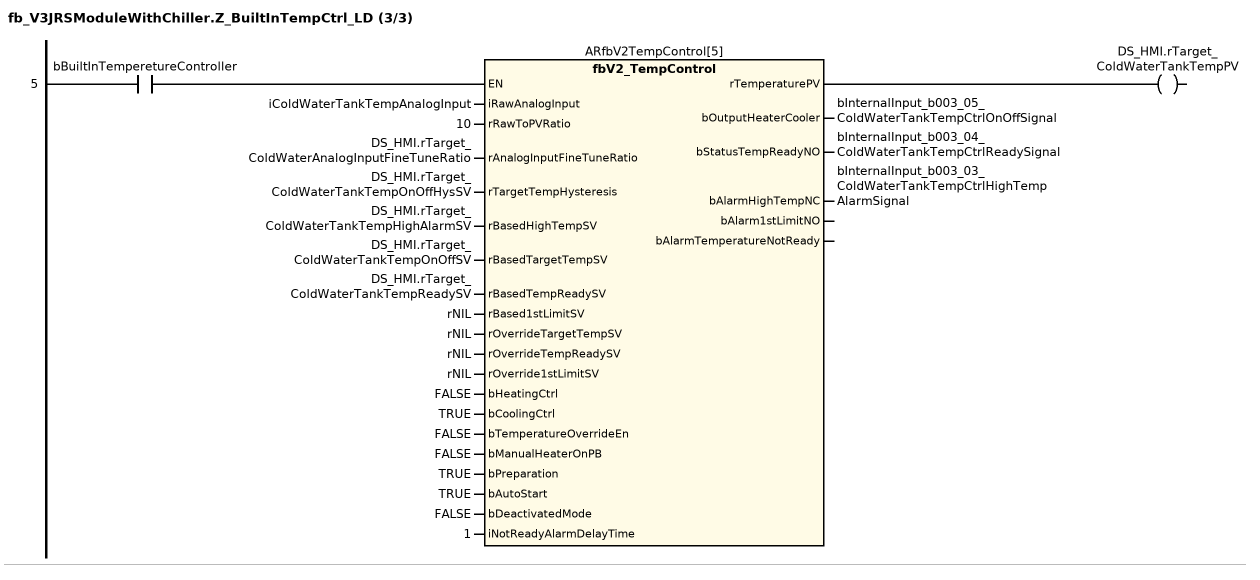
// NETWORK 5
IF bBuiltInTemperetureController THEN
    ARfbV2TempControl[5](
        iRawAnalogInput := iColdWaterTankTempAnalogInput,
        rRawToPVRatio := 10,
        rAnalogInputFineTuneRatio := DS_HMI.rTarget_ColdWaterAnalogInputFineTuneRatio,
        rTargetTempHysteresis := DS_HMI.rTarget_ColdWaterTankTempOnOffHysSV,
        rBasedHighTempSV := DS_HMI.rTarget_ColdWaterTankTempHighAlarmSV,
        rBasedTargetTempSV := DS_HMI.rTarget_ColdWaterTankTempOnOffSV,
        rBasedTempReadySV := DS_HMI.rTarget_ColdWaterTankTempReadySV,
        rBased1stLimitSV := rNIL,
        rOverrideTargetTempSV := rNIL,
        rOverrideTempReadySV := rNIL,
        rOverride1stLimitSV := rNIL,
        bHeatingCtrl := FALSE,
        bCoolingCtrl := TRUE,
        bTemperatureOverrideEn := FALSE,
        bManualHeaterOnPB := FALSE,
        bPreparation := TRUE,
        bAutoStart := TRUE,
        bDeactivatedMode := FALSE,
        iNotReadyAlarmDelayTime := 1,
        bOutputHeaterCooler => bInternalInput_b003_05_ColdWaterTankTempCtrlOnOffSignal,
        bStatusTempReadyNO => bInternalInput_b003_04_ColdWaterTankTempCtrlReadySignal,
        bAlarmHighTempNC => bInternalInput_b003_03_ColdWaterTankTempCtrlHighTempAlarmSignal); // fbV2_TempControl
END_IF
DS_HMI.rTarget_ColdWaterTankTempPV := ARfbV2TempControl[5].rTemperaturePV;
END_ACTION

ACTION Z_BuiltInTempCtrl_ST:
	IF NOT bBuiltInTemperetureController THEN
	bInternalInput_b000_04_ThermalOilTempCtrlHighTempAlarmSignal 		:= 	DS_Input.b000_04_ThermalOilTempCtrlHighTempAlarmSignal;
	bInternalInput_b000_05_ThermalOilTempCtrlReadySignal			 	:= 	DS_Input.b000_05_ThermalOilTempCtrlReadySignal;
	bInternalInput_b000_06_ThermalOilTempCtrlOnOffSignal  				:= 	DS_Input.b000_06_ThermalOilTempCtrlOnOffSignal ;
	bInternalInput_b000_07_TopDistillatorTempCtrlHighTempAlarmSignal 		:= 	DS_Input.b000_07_TopDistillatorTempCtrlHighTempAlarmSignal;
	bInternalInput_b000_08_TopDistillatorTempCtrlReadySignal 				:= 	DS_Input.b000_08_TopDistillatorTempCtrlReadySignal;
	bInternalInput_b000_09_TopDistillatorTempCtrlOnOffSignal  				:= 	DS_Input.b000_09_TopDistillatorTempCtrlOnOffSignal ;
	bInternalInput_b001_08_BottomDistillatorTempCtrlHighTempAlarmSignal 	:= 	DS_Input.b001_08_BottomDistillatorTempCtrlHighTempAlarmSignal;
	bInternalInput_b001_09_BottomDistillatorTempCtrlReadySignal 			:= 	DS_Input.b001_09_BottomDistillatorTempCtrlReadySignal;
	bInternalInput_b001_10_BottomDistillatorTempCtrlOnOffSignal  			:= 	DS_Input.b001_10_BottomDistillatorTempCtrlOnOffSignal ;
	bInternalInput_b002_00_VaporGenerationTempCtrlHighTempAlarmSignal 	:= 	DS_Input.b002_00_VaporGenerationTempCtrlHighTempAlarmSignal;
	bInternalInput_b002_01_VaporGenerationTempCtrlReadySignal 			:= 	DS_Input.b002_01_VaporGenerationTempCtrlReadySignal;
	bInternalInput_b002_02_VaporGenerationTempCtrlOnOffSignal 			:= 	DS_Input.b002_02_VaporGenerationTempCtrlOnOffSignal;
	bInternalInput_b003_03_ColdWaterTankTempCtrlHighTempAlarmSignal 	:= 	DS_Input.b003_03_ColdWaterTankTempCtrlHighTempAlarmSignal;
	bInternalInput_b003_04_ColdWaterTankTempCtrlReadySignal 			:= 	DS_Input.b003_04_ColdWaterTankTempCtrlReadySignal;
	bInternalInput_b003_05_ColdWaterTankTempCtrlOnOffSignal 			:= 	DS_Input.b003_05_ColdWaterTankTempCtrlOnOffSignal;

	ELSE

	Z_BuiltInTempCtrl_LD();
	END_IF

(*
	iThermalOilTempAnalogInput;			AT %I* : INT;
	iTopDistillatorTempAnalogInput;			AT %I* : INT;
	iBottomDistillatorTempAnalogInput;		AT %I* : INT;
	iVaporGenerationTempAnalogInput;		AT %I* : INT;
	iColdWaterTankTempAnalogInput; 		AT %I* : INT;


*)
END_ACTION

ACTION Z_BuiltInVacuumCtrl_LD:
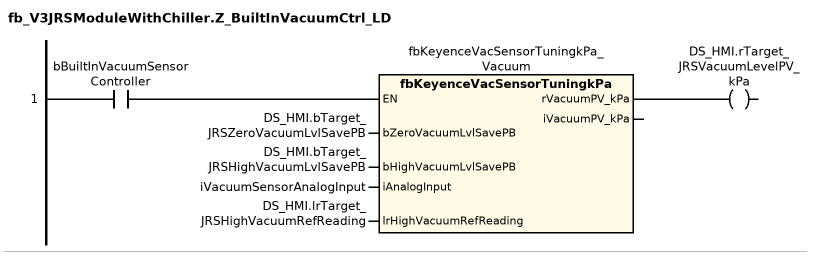
// NETWORK 1
IF bBuiltInVacuumSensorController THEN
    fbKeyenceVacSensorTuningkPa_Vacuum(
        bZeroVacuumLvlSavePB := DS_HMI.bTarget_JRSZeroVacuumLvlSavePB,
        bHighVacuumLvlSavePB := DS_HMI.bTarget_JRSHighVacuumLvlSavePB,
        iAnalogInput := iVacuumSensorAnalogInput,
        lrHighVacuumRefReading := DS_HMI.lrTarget_JRSHighVacuumRefReading); // fbKeyenceVacSensorTuningkPa
END_IF
DS_HMI.rTarget_JRSVacuumLevelPV_kPa := fbKeyenceVacSensorTuningkPa_Vacuum.rVacuumPV_kPa;
END_ACTION

ACTION Z_BuiltInVacuumCtrl_ST:
	IF NOT bBuiltInVacuumSensorController THEN

		bInternalInput_b001_04_VacuumNotAchieveSignal 		:= 	DS_Input.b001_04_VacuumNotAchieveSignal;

	ELSE

		Z_BuiltInVacuumCtrl_LD();

		bVacuumAchieveFlag := FALSE;

		(*Compare and trigger output*)
		IF bBuiltInVacuumNegativeSignal THEN

			IF DS_HMI.rTarget_JRSVacuumLevelPV_kPa <= DS_HMI.rTarget_JRSVacuumLevelSV_kPa THEN
				bVacuumAchieveFlag := TRUE;
			END_IF

		ELSE

			IF DS_HMI.rTarget_JRSVacuumLevelPV_kPa >= DS_HMI.rTarget_JRSVacuumLevelSV_kPa THEN
				bVacuumAchieveFlag := TRUE;
			END_IF

		END_IF

		bInternalInput_b001_04_VacuumNotAchieveSignal := NOT bVacuumAchieveFlag;


	END_IF
END_ACTION

ACTION Z_Mapping:
		(*Mapping - Alarm*)
		DS_Alarm.b200_00_FreshHCTankCircPumpTORAlarm  := bInternalAlarm_b200_00_FreshHCTankCircPumpTORAlarm ;
		DS_Alarm.b200_01_CircTankCircPumpTORAlarm  := bInternalAlarm_b200_01_CircTankCircPumpTORAlarm ;
		DS_Alarm.b200_02_ThermalOilPumpTORAlarm  := bInternalAlarm_b200_02_ThermalOilPumpTORAlarm ;
		DS_Alarm.b200_03_ThermalOilLowLevelAlarm  := bInternalAlarm_b200_03_ThermalOilLowLevelAlarm ;
		DS_Alarm.b200_04_ThermalOilTempHighAlarm  := bInternalAlarm_b200_04_ThermalOilTempHighAlarm ;
		DS_Alarm.b200_05_ThermalOilTempNotReadyAlarm  := bInternalAlarm_b200_05_ThermalOilTempNotReadyAlarm ;
		DS_Alarm.b200_06_ThermalOilHeaterOnOffAlarm  := bInternalAlarm_b200_06_ThermalOilHeaterOnOffAlarm ;
		DS_Alarm.b200_07_TopDistillatorTempHighAlarm  := bInternalAlarm_b200_07_TopDistillatorTempHighAlarm ;
		DS_Alarm.b200_08_TopDistillatorTempNotReadyAlarm  := bInternalAlarm_b200_08_TopDistillatorTempNotReadyAlarm ;
		DS_Alarm.b200_09_TopDistillatorHeaterOnOffAlarm  := bInternalAlarm_b200_09_TopDistillatorHeaterOnOffAlarm ;
		DS_Alarm.b200_10_RecycleStartStopPBAlarm  := bInternalAlarm_b200_10_RecycleStartStopPBAlarm ;
		DS_Alarm.b200_11_EstopPBAlarm  := bInternalAlarm_b200_11_EstopPBAlarm ;

		DS_Alarm.b201_00_PhaseSeqenceRelayAlarm  := bInternalAlarm_b201_00_PhaseSeqenceRelayAlarm ;
		DS_Alarm.b201_01_ThermalOilUpThermostatAlarm  := bInternalAlarm_b201_01_ThermalOilUpThermostatAlarm ;
		DS_Alarm.b201_02_SludgeTankHighLevelAlarm  := bInternalAlarm_b201_02_SludgeTankHighLevelAlarm ;
		DS_Alarm.b201_03_FreshHCTankLowLevelAlarm  := bInternalAlarm_b201_03_FreshHCTankLowLevelAlarm ;
		DS_Alarm.b201_04_VacuumNotAchieveAlarm  := bInternalAlarm_b201_04_VacuumNotAchieveAlarm ;
		DS_Alarm.b201_05_IncomingCDALowPressureAlarm  := bInternalAlarm_b201_05_IncomingCDALowPressureAlarm ;
		DS_Alarm.b201_06_CoolingWaterLowFlowAlarm  := bInternalAlarm_b201_06_CoolingWaterLowFlowAlarm ;
		DS_Alarm.b201_07_CircularTankLowLevelAlarm  := bInternalAlarm_b201_07_CircularTankLowLevelAlarm ;
		DS_Alarm.b201_08_BottomDistillatorTempHighAlarm  := bInternalAlarm_b201_08_BottomDistillatorTempHighAlarm ;
		DS_Alarm.b201_09_BottomDistillatorTempNotReadyAlarm  := bInternalAlarm_b201_09_BottomDistillatorTempNotReadyAlarm ;
		DS_Alarm.b201_10_BottomDistillatorHeaterOnOffAlarm  := bInternalAlarm_b201_10_BottomDistillatorHeaterOnOffAlarm ;
		DS_Alarm.b201_11_ThermalOilDownThermostatAlarm  := bInternalAlarm_b201_11_ThermalOilDownThermostatAlarm ;
		DS_Alarm.b201_12_ThermalOilMidThermostatAlarm  := bInternalAlarm_b201_12_ThermalOilMidThermostatAlarm ;

		DS_Alarm.b202_00_VaporGenerationTempHighAlarm  := bInternalAlarm_b202_00_VaporGenerationTempHighAlarm ;
		DS_Alarm.b202_01_VaporGenerationTempNotReadyAlarm  := bInternalAlarm_b202_01_VaporGenerationTempNotReadyAlarm ;
		DS_Alarm.b202_02_VaporGenerationHeaterOnOffAlarm  := bInternalAlarm_b202_02_VaporGenerationHeaterOnOffAlarm ;
		DS_Alarm.b202_03_WasteCollectionTankLowLevelAlarm  := bInternalAlarm_b202_03_WasteCollectionTankLowLevelAlarm ;
		DS_Alarm.b202_04_VaporGenerationTankLowLevelAlarm  := bInternalAlarm_b202_04_VaporGenerationTankLowLevelAlarm ;
		DS_Alarm.b202_05_HCPurgingAV3_1Alarm  := bInternalAlarm_b202_05_HCPurgingAV3_1Alarm ;
		DS_Alarm.b202_06_MainMachineWasteTankLowLevelAlarm  := bInternalAlarm_b202_06_MainMachineWasteTankLowLevelAlarm ;
		DS_Alarm.b202_07_MainMachineWasteTankHighLevelAlarm  := bInternalAlarm_b202_07_MainMachineWasteTankHighLevelAlarm ;
		DS_Alarm.b202_08_ReservedAlarm  := bInternalAlarm_b202_08_ReservedAlarm ;
		DS_Alarm.b202_09_ReservedAlarm  := bInternalAlarm_b202_09_ReservedAlarm ;
		DS_Alarm.b202_10_ReservedAlarm  := bInternalAlarm_b202_10_ReservedAlarm ;
		DS_Alarm.b202_11_ReservedAlarm  := bInternalAlarm_b202_11_ReservedAlarm ;
		
		DS_Alarm.b203_00_ChillerSelectorOnOffAlarm  := bInternalAlarm_b203_00_ChillerSelectorOnOffAlarm ;
		DS_Alarm.b203_01_ColdWaterTankLowLevelAlarm  := bInternalAlarm_b203_01_ColdWaterTankLowLevelAlarm ;
		DS_Alarm.b203_02_SludgeTankMissingAlarm  := bInternalAlarm_b203_02_SludgeTankMissingAlarm ;
		DS_Alarm.b203_03_ColdWaterTankTempHighAlarm  := bInternalAlarm_b203_03_ColdWaterTankTempHighAlarm ;
		DS_Alarm.b203_04_ColdWaterTankTempNotReadyAlarm  := bInternalAlarm_b203_04_ColdWaterTankTempNotReadyAlarm ;
		DS_Alarm.b203_05_ColdWaterTankHeaterOnOffAlarm  := bInternalAlarm_b203_05_ColdWaterTankHeaterOnOffAlarm ;
		DS_Alarm.b203_06_ChillerPumpTORAlarm  := bInternalAlarm_b203_06_ChillerPumpTORAlarm ;
		DS_Alarm.b203_07_ChillerFlowSwitchAlarm  := bInternalAlarm_b203_07_ChillerFlowSwitchAlarm ;
		DS_Alarm.b203_08_ChillerInterlockRelayAlarm  := bInternalAlarm_b203_08_ChillerInterlockRelayAlarm ;
		DS_Alarm.b203_09_ReservedAlarm  := bInternalAlarm_b203_09_ReservedAlarm ;
		DS_Alarm.b203_10_ThermalOilChangeWarning  := bInternalAlarm_b203_10_ThermalOilChangeWarning ;
		DS_Alarm.b203_11_ThermalOilChangeAlarm  := bInternalAlarm_b203_11_ThermalOilChangeAlarm ;
		
		
		(*Mapping - Input*)	
		bInternalInput_b000_00_FreshHCTankCircPumpTOR  := DS_Input.b000_00_FreshHCTankCircPumpTOR ;
		bInternalInput_b000_01_CircTankCircPumpTOR  := DS_Input.b000_01_CircTankCircPumpTOR ;
		bInternalInput_b000_02_ThermalOilPumpTOR := DS_Input.b000_02_ThermalOilPumpTOR;
		bInternalInput_b000_03_ThermalOilLevelSensor := DS_Input.b000_03_ThermalOilLevelSensor;
(*		bInternalInput_b000_04_ThermalOilTempCtrlHighTempAlarmSignal := DS_Input.b000_04_ThermalOilTempCtrlHighTempAlarmSignal;
		bInternalInput_b000_05_ThermalOilTempCtrlReadySignal := DS_Input.b000_05_ThermalOilTempCtrlReadySignal;
		bInternalInput_b000_06_ThermalOilTempCtrlOnOffSignal  := DS_Input.b000_06_ThermalOilTempCtrlOnOffSignal ;
		bInternalInput_b000_07_TopDistillatorTempCtrlHighTempAlarmSignal := DS_Input.b000_07_TopDistillatorTempCtrlHighTempAlarmSignal;
		bInternalInput_b000_08_TopDistillatorTempCtrlReadySignal := DS_Input.b000_08_TopDistillatorTempCtrlReadySignal;
		bInternalInput_b000_09_TopDistillatorTempCtrlOnOffSignal  := DS_Input.b000_09_TopDistillatorTempCtrlOnOffSignal ;
*)		bInternalInput_b000_10_RecycleStartStopPB := DS_Input.b000_10_RecycleStartStopPB;
		bInternalInput_b000_11_EStopPB := DS_Input.b000_11_EStopPB;


		bInternalInput_b001_00_PhaseSequenceRelayAlarm := DS_Input.b001_00_PhaseSequenceRelayAlarm;
		bInternalInput_b001_01_ThermalOilUpThermostat  := DS_Input.b001_01_ThermalOilUpThermostat ;
		bInternalInput_b001_02_SludgeTankLevelSensor := DS_Input.b001_02_SludgeTankLevelSensor;
		bInternalInput_b001_03_FreshHCTankLevelSensor := DS_Input.b001_03_FreshHCTankLevelSensor;
(*		bInternalInput_b001_04_VacuumNotAchieveSignal := DS_Input.b001_04_VacuumNotAchieveSignal;
*)		bInternalInput_b001_05_IncomingCDAPressureSwitch := DS_Input.b001_05_IncomingCDAPressureSwitch;
		bInternalInput_b001_06_CoolingWaterFlowSwitch := DS_Input.b001_06_CoolingWaterFlowSwitch;
		bInternalInput_b001_07_CircularTankLevelSensor := DS_Input.b001_07_CircularTankLevelSensor;
(*		bInternalInput_b001_08_BottomDistillatorTempCtrlHighTempAlarmSignal := DS_Input.b001_08_BottomDistillatorTempCtrlHighTempAlarmSignal;
		bInternalInput_b001_09_BottomDistillatorTempCtrlReadySignal := DS_Input.b001_09_BottomDistillatorTempCtrlReadySignal;
		bInternalInput_b001_10_BottomDistillatorTempCtrlOnOffSignal  := DS_Input.b001_10_BottomDistillatorTempCtrlOnOffSignal ;
*)		bInternalInput_b001_11_ThermalOilDownThermostat := DS_Input.b001_11_ThermalOilDownThermostat;
		bInternalInput_b001_12_ThermalOilMidThermostat := DS_Input.b001_12_ThermalOilMidThermostat;

(*		bInternalInput_b002_00_VaporGenerationTempCtrlHighTempAlarmSignal := DS_Input.b002_00_VaporGenerationTempCtrlHighTempAlarmSignal;
		bInternalInput_b002_01_VaporGenerationTempCtrlReadySignal := DS_Input.b002_01_VaporGenerationTempCtrlReadySignal;
		bInternalInput_b002_02_VaporGenerationTempCtrlOnOffSignal := DS_Input.b002_02_VaporGenerationTempCtrlOnOffSignal;
*)		bInternalInput_b002_03_WasteCollectionTankLevelSensor := DS_Input.b002_03_WasteCollectionTankLevelSensor;
		bInternalInput_b002_04_VaporGenerationTankLowLevelSensor := DS_Input.b002_04_VaporGenerationTankLowLevelSensor;
		bInternalInput_b002_05_HCPurgingAV := DS_Input.b002_05_HCPurgingAV;
		bInternalInput_b002_06_MainMachineWasteCollectTankLowLevelSignal := DS_Input.b002_06_MainMachineWasteCollectTankLowLevelSignal;
		bInternalInput_b002_07_MainMachineWasteCollectTankHighLevelSignal := DS_Input.b002_07_MainMachineWasteCollectTankHighLevelSignal;
		bInternalInput_b002_08_FromMainMachineSignal3 := DS_Input.b002_08_FromMainMachineSignal3;
		bInternalInput_b002_09_FromMainMachineSignal4 := DS_Input.b002_09_FromMainMachineSignal4;
		bInternalInput_b002_10_FromMainMachineSignal5 := DS_Input.b002_10_FromMainMachineSignal5;
		bInternalInput_b002_11_ReservedAlarmSignal := DS_Input.b002_11_ReservedAlarmSignal;


		bInternalInput_b003_00_ChillerSelectorOnOff := DS_Input.b003_00_ChillerSelectorOnOff;
		bInternalInput_b003_01_ColdWaterTankLowLevelSensor := DS_Input.b003_01_ColdWaterTankLowLevelSensor;
		bInternalInput_b003_02_SludgeTankPresentSensor := DS_Input.b003_02_SludgeTankPresentSensor;
(*		bInternalInput_b003_03_ColdWaterTankTempCtrlHighTempAlarmSignal := DS_Input.b003_03_ColdWaterTankTempCtrlHighTempAlarmSignal;
		bInternalInput_b003_04_ColdWaterTankTempCtrlReadySignal := DS_Input.b003_04_ColdWaterTankTempCtrlReadySignal;
		bInternalInput_b003_05_ColdWaterTankTempCtrlOnOffSignal := DS_Input.b003_05_ColdWaterTankTempCtrlOnOffSignal;
*)		bInternalInput_b003_06_ChillerPumpTOR := DS_Input.b003_06_ChillerPumpTOR;
		bInternalInput_b003_07_ChillerFlowSwitch := DS_Input.b003_07_ChillerFlowSwitch;
		bInternalInput_b003_08_ChillerInterlockRelay := DS_Input.b003_08_ChillerInterlockRelay;
		bInternalInput_b003_09_ReservedAlarmSignal := DS_Input.b003_09_ReservedAlarmSignal;
		bInternalInput_b003_10_ReservedAlarmSignal := DS_Input.b003_10_ReservedAlarmSignal;
		bInternalInput_b003_11_ReservedAlarmSignal := DS_Input.b003_11_ReservedAlarmSignal;
		
		(*Mapping - Output*)
		DS_Output.b100_00_FreshHCTankCircPumpOnOff  := bInternalOutput_b100_00_FreshHCTankCircPumpOnOff ;
		DS_Output.b100_01_CircTankCircPumpOnOff := bInternalOutput_b100_01_CircTankCircPumpOnOff;
		DS_Output.b100_02_ThermalOilPumpOnOff := bInternalOutput_b100_02_ThermalOilPumpOnOff;
		DS_Output.b100_03_ThermalOilHeaterOnOff := bInternalOutput_b100_03_ThermalOilHeaterOnOff;
		DS_Output.b100_04_Buzzer := bInternalOutput_b100_04_Buzzer;
		DS_Output.b100_05_RecycleStartStopIndicator := bInternalOutput_b100_05_RecycleStartStopIndicator;
		DS_Output.b100_06_Reserved := bInternalOutput_b100_06_Reserved;
		DS_Output.b100_07_UFOVacuumRelease32WayAV := bInternalOutput_b100_07_UFOVacuumRelease32WayAV;
		
		
		DS_Output.b101_00_CondenserTankVacuumReleaseAV := bInternalOutput_b101_00_CondenserTankVacuumReleaseAV;
		DS_Output.b101_01_WasteSludgeCollectionDrumAV  := bInternalOutput_b101_01_WasteSludgeCollectionDrumAV ;
		DS_Output.b101_02_DistillationTankDrainAV := bInternalOutput_b101_02_DistillationTankDrainAV;
		DS_Output.b101_03_EconomizerAV := bInternalOutput_b101_03_EconomizerAV;
		DS_Output.b101_04_Reserved := bInternalOutput_b101_04_Reserved;
		DS_Output.b101_05_Reserved := bInternalOutput_b101_05_Reserved;
		DS_Output.b101_06_VaporGenerationAV := bInternalOutput_b101_06_VaporGenerationAV;
		DS_Output.b101_07_VacuumSharingAV := bInternalOutput_b101_07_VacuumSharingAV;

		
		DS_Output.b102_00_RecycleReadySignal := bInternalOutput_b102_00_RecycleReadySignal;
		DS_Output.b102_01_VaporNotAvailableForRequestSignal := bInternalOutput_b102_01_VaporNotAvailableForRequestSignal;
		DS_Output.b102_02_ToMainMachineSignal3 := bInternalOutput_b102_02_ToMainMachineSignal3;
		DS_Output.b102_03_ToMainMachineSignal4 := bInternalOutput_b102_03_ToMainMachineSignal4;
		DS_Output.b102_04_ToMainMachineSignal5 := bInternalOutput_b102_04_ToMainMachineSignal5;
		DS_Output.b102_05_Reserved := bInternalOutput_b102_05_Reserved;
		DS_Output.b102_06_Reserved := bInternalOutput_b102_06_Reserved;
		DS_Output.b102_07_Reserved := bInternalOutput_b102_07_Reserved;
		
		
		DS_Output.b103_00_ChillerPumpOnOff := bInternalOutput_b103_00_ChillerPumpOnOff;
		DS_Output.b103_01_Reserved := bInternalOutput_b103_01_Reserved;
		DS_Output.b103_02_Reserved := bInternalOutput_b103_02_Reserved;
		DS_Output.b103_03_Reserved := bInternalOutput_b103_03_Reserved;
		DS_Output.b103_04_ChillerSelectorOnOffIndicator := bInternalOutput_b103_04_ChillerSelectorOnOffIndicator;
		DS_Output.b103_05_ChillerReadySignal := bInternalOutput_b103_05_ChillerReadySignal;
		DS_Output.b103_06_ChillerCompressorOnOff := bInternalOutput_b103_06_ChillerCompressorOnOff;
		DS_Output.b103_07_Reserved := bInternalOutput_b103_07_Reserved;
END_ACTION

END_FUNCTION_BLOCK

// ---- FBs/B_JKS_OldFB/Timer/TIMER_ALARM.TcPOU
FUNCTION_BLOCK TIMER_ALARM
VAR_INPUT
	BOOL_SIGNAL_IN: BOOL;
	BOOL_ALMRST_PB: BOOL;
	BOOL_BZRST_PB: BOOL;
	INT_PV: INT;

END_VAR

VAR_OUTPUT
	ALM_MSG_BOOL: BOOL;
	BZ_OUT_BOOL: BOOL;
	EV_INT: INT;
END_VAR

VAR
	T1: TON;
	M0: BOOL;
	M1: BOOL;
	D200: TIME;
	D202: INT;
END_VAR

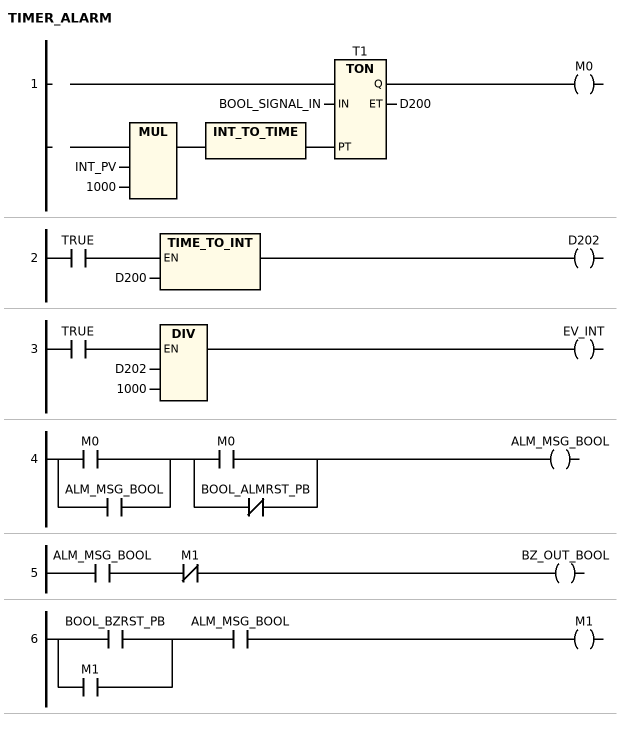
// NETWORK 1
T1(IN := BOOL_SIGNAL_IN, PT := INT_TO_TIME(INT_PV * 1000), ET => D200); // TON
M0 := T1.Q;

// NETWORK 2
D202 := TIME_TO_INT(D200);

// NETWORK 3
EV_INT := D202 / 1000;

// NETWORK 4
ALM_MSG_BOOL := (M0 OR ALM_MSG_BOOL) AND (M0 OR NOT BOOL_ALMRST_PB);

// NETWORK 5
BZ_OUT_BOOL := ALM_MSG_BOOL AND NOT M1;

// NETWORK 6
M1 := (BOOL_BZRST_PB OR M1) AND ALM_MSG_BOOL;

END_FUNCTION_BLOCK

// ---- FBs/B_JKS_OldFB/Compare/EQ_GT.TcPOU
FUNCTION_BLOCK EQ_GT
VAR_INPUT
	INT_SOURCE_A: INT;
	INT_SOURCE_B: INT;
END_VAR
VAR_OUTPUT
	SIGNAL_BOOL: BOOL;
END_VAR
VAR
	M0: BOOL;
	M1: BOOL;
END_VAR

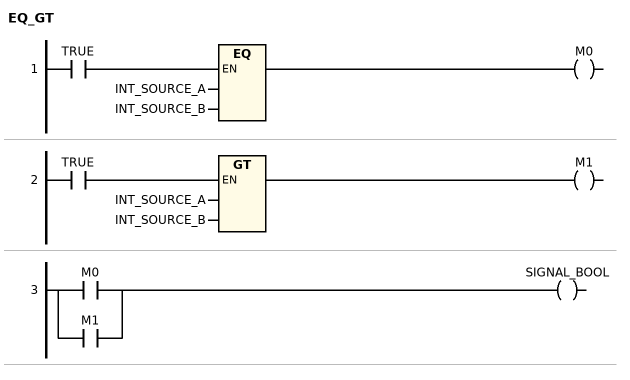
// NETWORK 1
M0 := INT_SOURCE_A = INT_SOURCE_B;

// NETWORK 2
M1 := INT_SOURCE_A > INT_SOURCE_B;

// NETWORK 3
SIGNAL_BOOL := M0 OR M1;

END_FUNCTION_BLOCK

// ---- FBs/B_JKS_NewFB/FBP-ProcessOptimisation/fbMasterTimeBlockG2.TcPOU
FUNCTION_BLOCK fbMasterTimeBlockG2

VAR_INPUT
	bStartEN : BOOL;
	bScanEN: BOOL;
	bWriteEN : BOOL;
	bCallRTB_CallOK : BOOL; (*From fbFBPTimeTrackerG2*)
	bMTBResetEN : BOOL;
	ARiArmID: ARRAY [1..iArmQty] OF INT;
	ARbAlternateStnEn : ARRAY [1..iAlternateSetQty] OF BOOL;
	AR2siAlternateStn : ARRAY [1..iAlternateSetQty, 1..iAlternateStnQty] OF INT;

	iScanCompleteDelayOnTime_ms: INT;
	iWriteRetryQty: INT;
	iWriteRetryDelayTimeSec : INT;
	iLoadingCallArmTime : INT;

END_VAR


VAR_OUTPUT

	bScanCompletedFlag: BOOL;
	bWriteDoneFlag : BOOL;
	bMTBResetDoneFlag : BOOL;

	bWriteArmDataError : BOOL;
	bWriteStnDataError : BOOL;
	bNoAvailableSlotError : BOOL;
	bArmIDAndStnIDNotFound : BOOL;

	iNextTransferScanCounter: INT;
	iNextNotAvailableScanCounter: INT;

	ARbArmProgress:ARRAY [1..iArmQty] OF BOOL;
	iNextTransferTime: INT;
	iNextNotAvailableTime : INT; (*New*)

	bWriteDisable: BOOL;
	bWriteRetry : BOOL;
	bWriteExecutedError : BOOL;
END_VAR

VAR_IN_OUT
	AR2SiRecipeTimeBlockNoCallArmTime : ARRAY[1..iRecipeBlockQty, 1..3] OF INT;
	AR2SiRecipeTimeBlockWithCallArmTime : ARRAY[1..iRecipeBlockQty, 1..3] OF INT;
	AR3SiMasterTimeBlockArm : ARRAY[1..iArmQty, 1..iMasterBlockQty, 1..3] OF INT;
	AR3SiMasterTimeBlockStn : ARRAY[1..iStnQty, 1..iMasterBlockQty, 1..3] OF INT;



END_VAR


VAR

	AR2SiInternalRepTimeBlockNoCallArmTime : ARRAY[1..iRecipeBlockQty, 1..3] OF INT;
	AR2SiInternalRepTimeBlockWithCallArmTime : ARRAY[1..iRecipeBlockQty, 1..3] OF INT;


	bInternalScanEN : BOOL;
	bInternalWriteEN : BOOL;
	OnTime : TON;
	OffTime : TON;
	OnTimeRE : R_TRIG;

	AR3SiBufferTimeBlockArm : ARRAY[1..iArmQty, 1..iMasterBlockQty, 1..3] OF INT;
	AR3SiBufferTimeBlockStn : ARRAY[1..iStnQty, 1..iMasterBlockQty, 1..3] OF INT;

	iScanningCounter: INT;
	ScanStep: INT;

	MTBResetRE: R_TRIG;
	BWriteRE: R_TRIG;
	ScanRE: R_TRIG;
	bMTBResetDoneFlagRE: R_TRIG;
	bInternalReScanFlagRE: R_TRIG;
	bWriteDoneFlagRE: R_TRIG;
	bNotAvailableTimeRE: R_TRIG;


	AR3SiNABufferTimeBlockArm : ARRAY[1..iArmQty, 1..iMasterBlockQty, 1..3] OF INT;
	AR3SiNABufferTimeBlockStn : ARRAY[1..iStnQty, 1..iMasterBlockQty, 1..3] OF INT;



	bNotAvailableTimeDetected: BOOL;
	bInternalReScanFlag: BOOL;
	bOverrideWriteInterlock: BOOL;

	bWriteElapseTimeST: BOOL;
	DelayOnScanCompleteTimer: TON;


	iArmNo: INT;
	iStnNo: INT;
	bArmIDFound: BOOL;
	bStnIDFound: BOOL;
	bCrashArm : BOOL;
	bCrashStn: BOOL;

	iNextTransferTimeTemp: INT;


	iNextNotAvailableTimeTemp : INT;

	iNAArmNo: INT;
	iNAStnNo: INT;
	bNAArmIDFound: BOOL;
	bNAStnIDFound: BOOL;
	bNACrashArm: BOOL;
	bNACrashStn: BOOL;
	iFillArmNo: INT;
	iFillStnNo: INT;
	bFIllArmIDFound: BOOL;
	bFillStnIDFound: BOOL;
	bFillArmDone: BOOL;
	bFillStnDone: BOOL;


	MTBCopyMFL: INT;
	MTBCopySFL: INT;

	ScanFL: INT;
	ScanMFL: INT;
	ScanSFL: INT;
	iCheckArmIDFL: INT;
	iCheckStnIDFL: INT;
	MTBMinusTimeMFL: INT;
	MTBMinusTimeSFL: INT;

	NAScanFL: INT;
	NAScanMFL : INT;
	NAScanSFL : INT;
	iNACheckArmIDFL: INT;
	iNACheckStnIDFL: INT;
	NAMTBMinusTimeMFL: INT;
	NAMTBMinusTimeSFL: INT;

	FillMFL: INT;
	FillSFL: INT;
	iCheckFillArmIDFL: INT;
	iCheckFillStnIDFL: INT;

(*No need master clear*)
	MTBResetMFL: INT;
	MTBResetSFL: INT;

	MTBBufferMinusTimeMFL: INT;
	MTBBufferMinusTimeSFL: INT;
	iTransferMFL: INT;
	iTransferSFL : INT;
	bWriteHR: BOOL;
	bOverrideRE: R_TRIG;
	iWriteStep: INT;

	BWriteOnlyRE: R_TRIG;
	iAutoRetryDelayTimer: INT;
	iWriteRetryQtyPV: INT;
	iCheckAlternateStnEnFL: INT;
	bAlternateStnEnableFound: BOOL;
	iAlternateSetFindFL: INT;
	iAlternateQtyFindFL: INT;
	iAlternateStnFindFL: INT;
	bAltStnIDFound: BOOL;
	iAltStnTransferFL: INT;
	ARiBufferAltStn: ARRAY [1..iAlternateStnQty] OF INT;
	iClearBufferAltFL: INT;
	iScanAltStnFL: INT;
	bCrashAltStn: BOOL;
	bAltnStnNoCrashFound: BOOL;

	iCheckMTBEmptyMFL: INT;
	iCheckMTBEmptySFL: INT;
	bMTBNotEmpty: BOOL;
	bScanStep9RE: R_TRIG;
END_VAR

IF bStartEN THEN

OnTime(IN:=NOT OffTime.Q , PT:=T#500ms , Q=> , ET=> );
OffTime(IN:=OnTime.Q , PT:=T#500ms , Q=> , ET=> );
OnTimeRE(CLK:=OnTime.Q , Q=> );

END_IF

(*Check if MTB is Empty *)

bMTBNotEmpty := FALSE;
iCheckMTBEmptyMFL := 1;
iCheckMTBEmptySFL := 1;


	IF iCheckMTBEmptyMFL>0 AND iCheckMTBEmptyMFL < iStnQty+1 THEN
		FOR iCheckMTBEmptyMFL := 1 TO iStnQty DO
		iCheckMTBEmptySFL := 1;
			IF iCheckMTBEmptySFL>0 AND iCheckMTBEmptySFL < iMasterBlockQty+1 THEN
				FOR iCheckMTBEmptySFL := 1 TO iMasterBlockQty DO

					IF AR3SiMasterTimeBlockStn[iCheckMTBEmptyMFL, iCheckMTBEmptySFL, 3] <> 0 THEN
					bMTBNotEmpty := TRUE;
					END_IF

					IF iCheckMTBEmptyMFL>0 AND iCheckMTBEmptyMFL <= iArmQty AND AR3SiMasterTimeBlockArm[iCheckMTBEmptyMFL, iCheckMTBEmptySFL, 3] <> 0 THEN
					bMTBNotEmpty := TRUE;
					END_IF
	
				END_FOR
			END_IF
	
		END_FOR
	
	END_IF




(*Check if AlternateStn Enable*)
bAlternateStnEnableFound := FALSE;
iCheckAlternateStnEnFL := 1;
	FOR iCheckAlternateStnEnFL := 1 TO iAlternateSetQty DO
		IF iCheckAlternateStnEnFL >= 1 AND iCheckAlternateStnEnFL <= iAlternateSetQty THEN
			IF ARbAlternateStnEn[iCheckAlternateStnEnFL] THEN
				bAlternateStnEnableFound := TRUE;
			END_IF
		END_IF
	END_FOR


(*Interlock for bScanEN and bWriteEN*)
IF bCallRTB_CallOK AND bScanEN THEN
bInternalScanEN := TRUE;
ELSE
bInternalScanEN := FALSE;
END_IF

IF bCallRTB_CallOK AND bWriteEN THEN
bInternalWriteEN := TRUE;
ELSE
bInternalWriteEN := FALSE;
END_IF

(* Minus 1 sec - Simulate actual status in machine*)
IF OnTimeRE.Q THEN
MTBMinusTimeMFL := 1;
MTBMinusTimeSFL := 1;
END_IF
IF bStartEN THEN

		IF MTBMinusTimeMFL>0 AND MTBMinusTimeMFL < iStnQty+1 THEN
			FOR MTBMinusTimeMFL := 1 TO iStnQty DO
			MTBMinusTimeSFL := 1;

				IF MTBMinusTimeSFL>0 AND MTBMinusTimeSFL < iMasterBlockQty+1 THEN
					FOR MTBMinusTimeSFL := 1 TO iMasterBlockQty DO

						IF AR3SiMasterTimeBlockStn[MTBMinusTimeMFL, MTBMinusTimeSFL, 1] > 0 THEN
						AR3SiMasterTimeBlockStn[MTBMinusTimeMFL, MTBMinusTimeSFL, 1] := AR3SiMasterTimeBlockStn[MTBMinusTimeMFL, MTBMinusTimeSFL, 1] - 1;
						END_IF

						IF AR3SiMasterTimeBlockStn[MTBMinusTimeMFL, MTBMinusTimeSFL, 2] > 0 THEN
						AR3SiMasterTimeBlockStn[MTBMinusTimeMFL, MTBMinusTimeSFL, 2] := AR3SiMasterTimeBlockStn[MTBMinusTimeMFL, MTBMinusTimeSFL, 2] - 1;
						END_IF

						IF AR3SiMasterTimeBlockStn[MTBMinusTimeMFL, MTBMinusTimeSFL, 2] <= 0 THEN
						AR3SiMasterTimeBlockStn[MTBMinusTimeMFL, MTBMinusTimeSFL, 1] := 0;
						AR3SiMasterTimeBlockStn[MTBMinusTimeMFL, MTBMinusTimeSFL, 2] := 0;
						AR3SiMasterTimeBlockStn[MTBMinusTimeMFL, MTBMinusTimeSFL, 3] := 0;
						END_IF



						IF MTBMinusTimeMFL <= iArmQty THEN
							ARbArmProgress[MTBMinusTimeMFL] := FALSE;
							IF AR3SiMasterTimeBlockArm[MTBMinusTimeMFL, MTBMinusTimeSFL, 1] > 0 THEN
							AR3SiMasterTimeBlockArm[MTBMinusTimeMFL, MTBMinusTimeSFL, 1] := AR3SiMasterTimeBlockArm[MTBMinusTimeMFL, MTBMinusTimeSFL, 1] - 1;
							END_IF

							IF AR3SiMasterTimeBlockArm[MTBMinusTimeMFL, MTBMinusTimeSFL, 2] > 0 THEN
							AR3SiMasterTimeBlockArm[MTBMinusTimeMFL, MTBMinusTimeSFL, 2] := AR3SiMasterTimeBlockArm[MTBMinusTimeMFL, MTBMinusTimeSFL, 2] - 1;
							END_IF

							IF AR3SiMasterTimeBlockArm[MTBMinusTimeMFL, MTBMinusTimeSFL, 2] <= 0 THEN
							AR3SiMasterTimeBlockArm[MTBMinusTimeMFL, MTBMinusTimeSFL, 1] := 0;
							AR3SiMasterTimeBlockArm[MTBMinusTimeMFL, MTBMinusTimeSFL, 2] := 0;
							AR3SiMasterTimeBlockArm[MTBMinusTimeMFL, MTBMinusTimeSFL, 3] := 0;
							END_IF

						IF AR3SiMasterTimeBlockArm[MTBMinusTimeMFL, MTBMinusTimeSFL, 1] = 0 AND AR3SiMasterTimeBlockArm[MTBMinusTimeMFL, MTBMinusTimeSFL, 2] > 0 THEN
						ARbArmProgress[MTBMinusTimeMFL] := TRUE;
						END_IF



						END_IF

					END_FOR
				END_IF

			END_FOR

		END_IF


END_IF


IF bInternalScanEN THEN
iNextTransferScanCounter:= ScanFL;
iNextNotAvailableScanCounter := NAScanFL;
ELSE
iNextTransferScanCounter:= 0;
iNextNotAvailableScanCounter := 0;
END_IF


(*Master Time Block Reset Program*)
MTBResetRE(CLK:=bMTBResetEN , Q=> );
IF MTBResetRE.Q(* bMTBResetEN*) THEN

(*iWriteElapseTime := 0;*)

MTBResetMFL := 1;
MTBResetSFL := 1;


	IF MTBResetMFL>0 AND MTBResetMFL < iStnQty+1 THEN
		FOR MTBResetMFL := 1 TO iStnQty DO
		MTBResetSFL := 1;
			IF MTBResetSFL>0 AND MTBResetSFL < iMasterBlockQty+1 THEN
				FOR MTBResetSFL := 1 TO iMasterBlockQty DO
	
					AR3SiMasterTimeBlockStn[MTBResetMFL, MTBResetSFL, 1] := 0;
					AR3SiMasterTimeBlockStn[MTBResetMFL, MTBResetSFL, 2] := 0;
					AR3SiMasterTimeBlockStn[MTBResetMFL, MTBResetSFL, 3] := 0;
	
					AR3SiBufferTimeBlockStn[MTBResetMFL, MTBResetSFL, 1] := 0;
					AR3SiBufferTimeBlockStn[MTBResetMFL, MTBResetSFL, 2] := 0;
					AR3SiBufferTimeBlockStn[MTBResetMFL, MTBResetSFL, 3] := 0;
	
					AR3SiNABufferTimeBlockStn[MTBResetMFL, MTBResetSFL, 1] := 0;
					AR3SiNABufferTimeBlockStn[MTBResetMFL, MTBResetSFL, 2] := 0;
					AR3SiNABufferTimeBlockStn[MTBResetMFL, MTBResetSFL, 3] := 0;
	
					IF MTBResetMFL>0 AND MTBResetMFL <= iArmQty THEN
	
					AR3SiMasterTimeBlockArm[MTBResetMFL, MTBResetSFL, 1] := 0;
					AR3SiMasterTimeBlockArm[MTBResetMFL, MTBResetSFL, 2] := 0;
					AR3SiMasterTimeBlockArm[MTBResetMFL, MTBResetSFL, 3] := 0;

					AR3SiBufferTimeBlockArm[MTBResetMFL, MTBResetSFL, 1] := 0;
					AR3SiBufferTimeBlockArm[MTBResetMFL, MTBResetSFL, 2] := 0;
					AR3SiBufferTimeBlockArm[MTBResetMFL, MTBResetSFL, 3] := 0;
	
					AR3SiNABufferTimeBlockArm[MTBResetMFL, MTBResetSFL, 1] := 0;
					AR3SiNABufferTimeBlockArm[MTBResetMFL, MTBResetSFL, 2] := 0;
					AR3SiNABufferTimeBlockArm[MTBResetMFL, MTBResetSFL, 3] := 0;

					ARbArmProgress[MTBResetMFL] := FALSE;

					END_IF
	
				END_FOR
			END_IF
	
		END_FOR
	
	END_IF

END_IF


IF bMTBResetEN AND MTBResetMFL > iStnQty AND MTBResetSFL > iMasterBlockQty THEN
bMTBResetDoneFlag := TRUE;
END_IF

IF NOT bMTBResetEN THEN
bMTBResetDoneFlag := FALSE;
END_IF



(************************************************ScanEN**********************************************************)

IF bInternalScanEN AND NOT bWriteDoneFlag AND OnTimeRE.Q THEN
iScanningCounter := iScanningCounter +1;
END_IF


IF NOT bInternalScanEN OR bWriteDoneFlag THEN

bNotAvailableTimeDetected:=FALSE;
bWriteArmDataError:=FALSE;
bWriteStnDataError:=FALSE;
bNoAvailableSlotError:=FALSE;
bArmIDAndStnIDNotFound:=FALSE;


iScanningCounter := 0;
iNextTransferTimeTemp := 0;
iNextTransferTime := 0;
ScanMFL := 0;
ScanStep := 0;
iNextNotAvailableTimeTemp := 0;
iNextNotAvailableTime := 0;
NAScanMFL := 0;
NAScanSFL := 0;

bScanCompletedFlag := FALSE;
bInternalReScanFlag := FALSE;


END_IF


ScanRE(CLK:=bInternalScanEN AND NOT bWriteDoneFlag , Q=> );
bMTBResetDoneFlagRE(CLK:=bMTBResetDoneFlag , Q=> );
bInternalReScanFlagRE(CLK:=bInternalReScanFlag AND NOT bInternalWriteEN , Q=> );



IF ScanRE.Q OR bInternalReScanFlagRE.Q OR bMTBResetDoneFlagRE.Q THEN

bNotAvailableTimeDetected:=FALSE;
bWriteArmDataError:=FALSE;
bWriteStnDataError:=FALSE;
bNoAvailableSlotError:=FALSE;
bArmIDAndStnIDNotFound:=FALSE;


iScanningCounter := 0;
iNextTransferTimeTemp := 0;
iNextTransferTime := 0;

iNextNotAvailableTimeTemp := 0;
iNextNotAvailableTime := 0;

bScanCompletedFlag := FALSE;
bInternalReScanFlag := FALSE;


ScanStep := 1;
MTBCopyMFL := 1;
MTBCopySFL := 1;



END_IF

(**Added to solve Alternate Tank Problem***)

IF bScanEN AND NOT bWriteEN AND ScanStep <=2 THEN
AR2SiInternalRepTimeBlockNoCallArmTime		:= AR2SiRecipeTimeBlockNoCallArmTime;
AR2SiInternalRepTimeBlockWithCallArmTime		:= AR2SiRecipeTimeBlockWithCallArmTime;
END_IF





(*Add Loading call arm time - Rising Edge*)
bScanStep9RE(CLK:=ScanStep=9 , Q=> );


CASE ScanStep OF

0:;


2: (*Reset ScanMFL and ScanSFL*)
ScanMFL:=1;
ScanSFL:=1;
ScanStep := 3;





1:  (*Copy from MasterTimeBlock to BufferTimeBlock*)



IF MTBCopyMFL> 0 AND MTBCopyMFL < iStnQty+1 THEN
	FOR MTBCopyMFL := 1 TO iStnQty DO
	MTBCopySFL := 1;
		IF MTBCopySFL> 0 AND MTBCopySFL < iMasterBlockQty+1 THEN
			FOR MTBCopySFL := 1 TO iMasterBlockQty DO

				AR3SiBufferTimeBlockStn[MTBCopyMFL, MTBCopySFL, 1] := AR3SiMasterTimeBlockStn[MTBCopyMFL, MTBCopySFL, 1];
				AR3SiBufferTimeBlockStn[MTBCopyMFL, MTBCopySFL, 2] := AR3SiMasterTimeBlockStn[MTBCopyMFL, MTBCopySFL, 2];
				AR3SiBufferTimeBlockStn[MTBCopyMFL, MTBCopySFL, 3] := AR3SiMasterTimeBlockStn[MTBCopyMFL, MTBCopySFL, 3];

				AR3SiNABufferTimeBlockStn[MTBCopyMFL, MTBCopySFL, 1] := AR3SiMasterTimeBlockStn[MTBCopyMFL, MTBCopySFL, 1];
				AR3SiNABufferTimeBlockStn[MTBCopyMFL, MTBCopySFL, 2] := AR3SiMasterTimeBlockStn[MTBCopyMFL, MTBCopySFL, 2];
				AR3SiNABufferTimeBlockStn[MTBCopyMFL, MTBCopySFL, 3] := AR3SiMasterTimeBlockStn[MTBCopyMFL, MTBCopySFL, 3];

				IF MTBCopyMFL> 0 AND MTBCopyMFL <= iArmQty THEN

				AR3SiBufferTimeBlockArm[MTBCopyMFL, MTBCopySFL, 1] := AR3SiMasterTimeBlockArm[MTBCopyMFL, MTBCopySFL, 1];
				AR3SiBufferTimeBlockArm[MTBCopyMFL, MTBCopySFL, 2] := AR3SiMasterTimeBlockArm[MTBCopyMFL, MTBCopySFL, 2];
				AR3SiBufferTimeBlockArm[MTBCopyMFL, MTBCopySFL, 3] := AR3SiMasterTimeBlockArm[MTBCopyMFL, MTBCopySFL, 3];

				AR3SiNABufferTimeBlockArm[MTBCopyMFL, MTBCopySFL, 1] := AR3SiMasterTimeBlockArm[MTBCopyMFL, MTBCopySFL, 1];
				AR3SiNABufferTimeBlockArm[MTBCopyMFL, MTBCopySFL, 2] := AR3SiMasterTimeBlockArm[MTBCopyMFL, MTBCopySFL, 2];
				AR3SiNABufferTimeBlockArm[MTBCopyMFL, MTBCopySFL, 3] := AR3SiMasterTimeBlockArm[MTBCopyMFL, MTBCopySFL, 3];

				END_IF

			END_FOR
		END_IF

	END_FOR

END_IF

IF MTBCopyMFL > iStnQty AND MTBCopySFL > iMasterBlockQty THEN
ScanFL := 1;
ScanStep := 2;
END_IF


3: (*Compare BufferTimeBlock VS RecipeTimeBlock*)

	IF ScanFL < 10000+1 THEN
	ScanMFL:= 1;

		IF ScanMFL>0 AND ScanMFL < iRecipeBlockQty+1 THEN

			FOR ScanMFL := 1 TO iRecipeBlockQty DO

				IF AR2SiInternalRepTimeBlockWithCallArmTime[ScanMFL, 2] > 0 THEN

					iClearBufferAltFL := 1;
						FOR iClearBufferAltFL := 1 TO iAlternateStnQty DO
							IF iClearBufferAltFL >= 1 AND iClearBufferAltFL <= iAlternateStnQty THEN
							ARiBufferAltStn[iClearBufferAltFL] := 0;
							END_IF
						END_FOR

					iArmNo:=0;
					iStnNo:=0;
					bArmIDFound:= FALSE;
					bStnIDFound:= FALSE;
					bAltStnIDFound := FALSE;

					iCheckArmIDFL := 1;
					iCheckStnIDFL := 1;

					(*Check ArmID*)
					IF iCheckArmIDFL>0 AND iCheckArmIDFL < iArmQty+1 THEN
						FOR iCheckArmIDFL := 1 TO iArmQty DO
							IF AR2SiInternalRepTimeBlockWithCallArmTime[ScanMFL,3] = ARiArmID[iCheckArmIDFL] THEN
							iArmNo := iCheckArmIDFL;
							bArmIDFound := TRUE;
							iCheckArmIDFL := iArmQty+1;
							END_IF
						END_FOR
					END_IF
	
					(*Check StnID*)
					IF iCheckStnIDFL>0 AND iCheckStnIDFL <iStnQty+1 THEN
						FOR iCheckStnIDFL := 1 TO iStnQty DO
							IF AR2SiInternalRepTimeBlockWithCallArmTime[ScanMFL,3] = iCheckStnIDFL THEN
							iStnNo := iCheckStnIDFL;
							bStnIDFound := TRUE;
							iCheckStnIDFL := iStnQty+1;
							END_IF

					(*ADD HERE*)
							IF bStnIDFound AND bAlternateStnEnableFound THEN
							iAlternateSetFindFL := 1;
								FOR iAlternateSetFindFL := 1 TO iAlternateSetQty DO
									IF iAlternateSetFindFL >= 1 AND iAlternateSetFindFL <= iAlternateSetQty THEN
										IF ARbAlternateStnEn[iAlternateSetFindFL] THEN
										iAlternateStnFindFL := 1; (*Find Stn ID matching*)
											FOR iAlternateStnFindFL := 1 TO iAlternateStnQty DO
												IF iAlternateStnFindFL >= 1 AND iAlternateStnFindFL <= iAlternateStnQty THEN
													IF iStnNo = AR2SiAlternateStn[iAlternateSetFindFL , iAlternateStnFindFL] THEN
														bAltStnIDFound := TRUE;
														iAltStnTransferFL := 1;
															FOR iAltStnTransferFL := 1 TO iAlternateStnQty DO
																IF iAltStnTransferFL >= 1 AND iAltStnTransferFL <= iAlternateStnQty THEN
																	ARiBufferAltStn[iAltStnTransferFL] := AR2SiAlternateStn[iAlternateSetFindFL , iAltStnTransferFL];
																END_IF
															END_FOR
														iAlternateSetFindFL := iAlternateSetQty+1;
														iAlternateStnFindFL := iAlternateStnQty+1;
														iAltStnTransferFL := iAlternateStnQty+1;

													END_IF
												END_IF
											END_FOR
										END_IF
									END_IF
								END_FOR
							END_IF
						END_FOR
					END_IF



					IF (bArmIDFound OR bStnIDFound) AND NOT bAltStnIDFound THEN

					ScanSFL := 1;
					bCrashArm := FALSE;
					bCrashStn := FALSE;

						IF (bArmIDFound OR bStnIDFound) AND ScanSFL>0 AND ScanSFL < iMasterBlockQty+1 THEN
							FOR ScanSFL := 1 TO iMasterBlockQty DO
	
								(*Arm Scanning*)
								IF bArmIDFound THEN

									IF AR3SiBufferTimeBlockArm[iArmNo,ScanSFL, 2] > 0 THEN
		
										IF
										AR3SiBufferTimeBlockArm[iArmNo,ScanSFL, 1] (*MD1*) <= AR2SiInternalRepTimeBlockWithCallArmTime[ScanMFL, 1] (*RD1*)
										AND
										AR3SiBufferTimeBlockArm[iArmNo,ScanSFL, 2] (*MD2*) >= AR2SiInternalRepTimeBlockWithCallArmTime[ScanMFL, 1] (*RD1*)
										THEN
										bCrashArm:=TRUE;
										ScanSFL:=iMasterBlockQty+1;
										ScanMFL := iRecipeBlockQty+1;
										END_IF
		
										IF
										AR3SiBufferTimeBlockArm[iArmNo,ScanSFL, 1] (*MD1*) <= AR2SiInternalRepTimeBlockWithCallArmTime[ScanMFL, 2] (*RD2*)
										AND
										AR3SiBufferTimeBlockArm[iArmNo,ScanSFL, 2] (*MD2*) >= AR2SiInternalRepTimeBlockWithCallArmTime[ScanMFL, 2] (*RD2*)
										THEN
										bCrashArm:=TRUE;
										ScanSFL:=iMasterBlockQty+1;
										ScanMFL := iRecipeBlockQty+1;
										END_IF
	
										IF
										AR2SiInternalRepTimeBlockWithCallArmTime[ScanMFL, 1] (*RD1*) <= AR3SiBufferTimeBlockArm[iArmNo,ScanSFL, 1] (*MD1*)
										AND
										AR2SiInternalRepTimeBlockWithCallArmTime[ScanMFL, 2] (*RD2*) >= AR3SiBufferTimeBlockArm[iArmNo,ScanSFL, 1] (*MD1*)
										THEN
										bCrashArm:=TRUE;
										ScanSFL:=iMasterBlockQty+1;
										ScanMFL := iRecipeBlockQty+1;
										END_IF
		
										IF
										AR2SiInternalRepTimeBlockWithCallArmTime[ScanMFL, 1] (*RD1*) <= AR3SiBufferTimeBlockArm[iArmNo,ScanSFL, 2] (*MD2*)
										AND
										AR2SiInternalRepTimeBlockWithCallArmTime[ScanMFL, 2] (*RD2*) >= AR3SiBufferTimeBlockArm[iArmNo,ScanSFL, 2] (*MD2*)
										THEN
										bCrashArm:=TRUE;
										ScanSFL:=iMasterBlockQty+1;
										ScanMFL := iRecipeBlockQty+1;
										END_IF
	
	
									END_IF
		
								END_IF
		
								(*Stn Scanning without Alternate Stn*)
								IF bStnIDFound AND NOT bAltStnIDFound THEN
	
									IF AR3SiBufferTimeBlockStn[iStnNo,ScanSFL, 2] > 0 THEN
	
										IF
										AR3SiBufferTimeBlockStn[iStnNo,ScanSFL, 1] (*MD1*) <= AR2SiInternalRepTimeBlockWithCallArmTime[ScanMFL, 1] (*RD1*)
										AND
										AR3SiBufferTimeBlockStn[iStnNo,ScanSFL, 2] (*MD2*) >= AR2SiInternalRepTimeBlockWithCallArmTime[ScanMFL, 1] (*RD1*)
										THEN
										bCrashStn:=TRUE;
										ScanSFL:=iMasterBlockQty+1;
										ScanMFL := iRecipeBlockQty+1;
										END_IF
		
										IF
										AR3SiBufferTimeBlockStn[iStnNo,ScanSFL, 1] (*MD1*) <= AR2SiInternalRepTimeBlockWithCallArmTime[ScanMFL, 2] (*RD2*)
										AND
										AR3SiBufferTimeBlockStn[iStnNo,ScanSFL, 2] (*MD2*) >= AR2SiInternalRepTimeBlockWithCallArmTime[ScanMFL, 2] (*RD2*)
										THEN
										bCrashStn:=TRUE;
										ScanSFL:=iMasterBlockQty+1;
										ScanMFL := iRecipeBlockQty+1;
										END_IF
	
										IF
										AR2SiInternalRepTimeBlockWithCallArmTime[ScanMFL, 1] (*RD1*) <= AR3SiBufferTimeBlockStn[iStnNo,ScanSFL, 1] (*MD1*)
										AND
										AR2SiInternalRepTimeBlockWithCallArmTime[ScanMFL, 2] (*RD2*) >= AR3SiBufferTimeBlockStn[iStnNo,ScanSFL, 1] (*MD1*)
										THEN
										bCrashStn:=TRUE;
										ScanSFL:=iMasterBlockQty+1;
										ScanMFL := iRecipeBlockQty+1;
										END_IF

										IF
										AR2SiInternalRepTimeBlockWithCallArmTime[ScanMFL, 1] (*RD1*) <= AR3SiBufferTimeBlockStn[iStnNo,ScanSFL, 2] (*MD2*)
										AND
										AR2SiInternalRepTimeBlockWithCallArmTime[ScanMFL, 2] (*RD2*) >= AR3SiBufferTimeBlockStn[iStnNo,ScanSFL, 2] (*MD2*)
										THEN
										bCrashStn:=TRUE;
										ScanSFL:=iMasterBlockQty+1;
										ScanMFL := iRecipeBlockQty+1;
										END_IF
	
	
									END_IF
		
								END_IF

							END_FOR

						END_IF

					END_IF

					(*Stn Scanning WITH Alternate Stn*)
					IF bStnIDFound AND bAltStnIDFound THEN

					iScanAltStnFL := 1;
					bCrashArm := FALSE;
					bCrashStn := FALSE;
					bAltnStnNoCrashFound := FALSE;
						FOR iScanAltStnFL := 1 TO iAlternateStnQty DO
							IF iScanAltStnFL >= 1 AND iScanAltStnFL <= iAlternateStnQty THEN

								IF ARiBufferAltStn[iScanAltStnFL] > 0 THEN
								bCrashAltStn := FALSE;
								ScanSFL := 1;

									FOR ScanSFL := 1 TO iMasterBlockQty DO
										IF  ScanSFL>= 1 AND ScanSFL <= iMasterBlockQty AND NOT bAltnStnNoCrashFound THEN

											IF AR3SiBufferTimeBlockStn[ARiBufferAltStn[iScanAltStnFL],ScanSFL, 2] > 0 THEN

												IF
												AR3SiBufferTimeBlockStn[ARiBufferAltStn[iScanAltStnFL],ScanSFL, 1] (*MD1*) <= AR2SiInternalRepTimeBlockWithCallArmTime[ScanMFL, 1] (*RD1*)
												AND
												AR3SiBufferTimeBlockStn[ARiBufferAltStn[iScanAltStnFL],ScanSFL, 2] (*MD2*) >= AR2SiInternalRepTimeBlockWithCallArmTime[ScanMFL, 1] (*RD1*)
												THEN
												bCrashAltStn:=TRUE;
												ScanSFL:=iMasterBlockQty+1;
												END_IF

												IF
												AR3SiBufferTimeBlockStn[ARiBufferAltStn[iScanAltStnFL],ScanSFL, 1] (*MD1*) <= AR2SiInternalRepTimeBlockWithCallArmTime[ScanMFL, 2] (*RD2*)
												AND
												AR3SiBufferTimeBlockStn[ARiBufferAltStn[iScanAltStnFL],ScanSFL, 2] (*MD2*) >= AR2SiInternalRepTimeBlockWithCallArmTime[ScanMFL, 2] (*RD2*)
												THEN
												bCrashAltStn:=TRUE;
												ScanSFL:=iMasterBlockQty+1;
												END_IF

												IF
												AR2SiInternalRepTimeBlockWithCallArmTime[ScanMFL, 1] (*RD1*) <= AR3SiBufferTimeBlockStn[ARiBufferAltStn[iScanAltStnFL],ScanSFL, 1] (*MD1*)
												AND
												AR2SiInternalRepTimeBlockWithCallArmTime[ScanMFL, 2] (*RD2*) >= AR3SiBufferTimeBlockStn[ARiBufferAltStn[iScanAltStnFL],ScanSFL, 1] (*MD1*)
												THEN
												bCrashAltStn:=TRUE;
												ScanSFL:=iMasterBlockQty+1;
												END_IF

												IF
												AR2SiInternalRepTimeBlockWithCallArmTime[ScanMFL, 1] (*RD1*) <= AR3SiBufferTimeBlockStn[ARiBufferAltStn[iScanAltStnFL],ScanSFL, 2] (*MD2*)
												AND
												AR2SiInternalRepTimeBlockWithCallArmTime[ScanMFL, 2] (*RD2*) >= AR3SiBufferTimeBlockStn[ARiBufferAltStn[iScanAltStnFL],ScanSFL, 2] (*MD2*)
												THEN
												bCrashAltStn:=TRUE;
												ScanSFL:=iMasterBlockQty+1;
												END_IF
											END_IF
										END_IF
									END_FOR

									IF ScanSFL > iMasterBlockQty AND bCrashAltStn AND (ARiBufferAltStn[iScanAltStnFL+1] <=0 OR iScanAltStnFL >= iAlternateStnQty) AND NOT bAltnStnNoCrashFound THEN
									bCrashStn := TRUE;
									iScanAltStnFL := iAlternateStnQty+1;
									ScanMFL := iRecipeBlockQty+1;
									END_IF

									IF ScanSFL > iMasterBlockQty AND NOT bCrashAltStn AND NOT bAltnStnNoCrashFound THEN
									AR2SiInternalRepTimeBlockWithCallArmTime[ScanMFL, 3] := ARiBufferAltStn[iScanAltStnFL];
									AR2SiInternalRepTimeBlockNoCallArmTime[ScanMFL, 3] := ARiBufferAltStn[iScanAltStnFL];
									bAltnStnNoCrashFound := TRUE;
									bCrashAltStn:=FALSE;
									bCrashStn := FALSE;
									END_IF

								END_IF
							END_IF
						END_FOR
					END_IF



				END_IF

			END_FOR

		END_IF

	END_IF



(* CRASH Found !!!, Shift one Second and Test again*)
IF ScanMFL > iRecipeBlockQty AND ScanSFL > iMasterBlockQty AND (bCrashArm OR bCrashStn) (*AND (bStepENRE.Q OR bStepAlwaysEN)*) THEN
MTBBufferMinusTimeMFL := 1;
MTBBufferMinusTimeSFL := 1;
ScanStep := 4;
END_IF

(* No Crash Found, Can proceed to Push In Basket *)
IF ScanMFL > iRecipeBlockQty AND ScanSFL > iMasterBlockQty AND NOT bCrashArm AND NOT bCrashStn (*AND (bStepENRE.Q OR bStepAlwaysEN)*) THEN

(*		IF bMTBNotEmpty THEN
			iNextTransferTimeTemp := ScanFL+iLoadingCallArmTime; (*Result FOUND*)
		ELSE
			iNextTransferTimeTemp := ScanFL; (*Result FOUND*)
		END_IF
*)
iNextTransferTimeTemp := ScanFL; (*Result FOUND*)

iTransferMFL := 1;
iTransferSFL := 1;
ScanStep := 5;
END_IF

(* No ArmID or StnID found*)
IF ScanMFL > iRecipeBlockQty AND NOT bStnIDFound AND NOT bArmIDFound THEN
ScanStep := 23; (*ArmID and StnID not found Error*)
END_IF

(*Cannot find suitable Slot*)
IF ScanFL > 10000 AND ScanMFL > iRecipeBlockQty AND ScanSFL > iMasterBlockQty THEN
ScanStep := 24;
END_IF

4: (*Minus One Second of BufferFL and Retry*)


		IF MTBBufferMinusTimeMFL>0 AND MTBBufferMinusTimeMFL < iStnQty+1 THEN
			FOR MTBBufferMinusTimeMFL := 1 TO iStnQty DO
			MTBBufferMinusTimeSFL := 1;
				IF MTBBufferMinusTimeSFL>0 AND MTBBufferMinusTimeSFL < iMasterBlockQty+1 THEN
					FOR MTBBufferMinusTimeSFL := 1 TO iMasterBlockQty DO

						IF AR3SiBufferTimeBlockStn[MTBBufferMinusTimeMFL, MTBBufferMinusTimeSFL, 1] > 0 THEN
						AR3SiBufferTimeBlockStn[MTBBufferMinusTimeMFL, MTBBufferMinusTimeSFL, 1] := AR3SiBufferTimeBlockStn[MTBBufferMinusTimeMFL, MTBBufferMinusTimeSFL, 1] - 1;
						END_IF

						IF AR3SiBufferTimeBlockStn[MTBBufferMinusTimeMFL, MTBBufferMinusTimeSFL, 2] > 0 THEN
						AR3SiBufferTimeBlockStn[MTBBufferMinusTimeMFL, MTBBufferMinusTimeSFL, 2] := AR3SiBufferTimeBlockStn[MTBBufferMinusTimeMFL, MTBBufferMinusTimeSFL, 2] - 1;
						END_IF

						IF AR3SiBufferTimeBlockStn[MTBBufferMinusTimeMFL, MTBBufferMinusTimeSFL, 2] <= 0 THEN
						AR3SiBufferTimeBlockStn[MTBBufferMinusTimeMFL, MTBBufferMinusTimeSFL, 1] := 0;
						AR3SiBufferTimeBlockStn[MTBBufferMinusTimeMFL, MTBBufferMinusTimeSFL, 2] := 0;
						AR3SiBufferTimeBlockStn[MTBBufferMinusTimeMFL, MTBBufferMinusTimeSFL, 3] := 0;
						END_IF



						IF MTBBufferMinusTimeMFL>0 AND MTBBufferMinusTimeMFL <= iArmQty THEN

							IF AR3SiBufferTimeBlockArm[MTBBufferMinusTimeMFL, MTBBufferMinusTimeSFL, 1] > 0 THEN
							AR3SiBufferTimeBlockArm[MTBBufferMinusTimeMFL, MTBBufferMinusTimeSFL, 1] := AR3SiBufferTimeBlockArm[MTBBufferMinusTimeMFL, MTBBufferMinusTimeSFL, 1] - 1;
							END_IF

							IF AR3SiBufferTimeBlockArm[MTBBufferMinusTimeMFL, MTBBufferMinusTimeSFL, 2] > 0 THEN
							AR3SiBufferTimeBlockArm[MTBBufferMinusTimeMFL, MTBBufferMinusTimeSFL, 2] := AR3SiBufferTimeBlockArm[MTBBufferMinusTimeMFL, MTBBufferMinusTimeSFL, 2] - 1;
							END_IF

							IF AR3SiBufferTimeBlockArm[MTBBufferMinusTimeMFL, MTBBufferMinusTimeSFL, 2] <= 0 THEN
							AR3SiBufferTimeBlockArm[MTBBufferMinusTimeMFL, MTBBufferMinusTimeSFL, 1] := 0;
							AR3SiBufferTimeBlockArm[MTBBufferMinusTimeMFL, MTBBufferMinusTimeSFL, 2] := 0;
							AR3SiBufferTimeBlockArm[MTBBufferMinusTimeMFL, MTBBufferMinusTimeSFL, 3] := 0;
							END_IF


						END_IF

					END_FOR
				END_IF

			END_FOR

		END_IF


(*Return to Step 2 for retry*)

ScanFL:=ScanFL+1;
ScanStep := 2;



5: (*Copy for Buffer TimeBlock to NA TimeBlock to continue search*)

IF iTransferMFL>0 AND iTransferMFL < iStnQty+1 THEN
	FOR iTransferMFL := 1 TO iStnQty DO
	iTransferSFL := 1;
		IF iTransferSFL>0 AND iTransferSFL < iMasterBlockQty+1 THEN
			FOR iTransferSFL := 1 TO iMasterBlockQty DO

				AR3SiNABufferTimeBlockStn[iTransferMFL, iTransferSFL, 1] := AR3SiBufferTimeBlockStn[iTransferMFL, iTransferSFL, 1];
				AR3SiNABufferTimeBlockStn[iTransferMFL, iTransferSFL, 2] := AR3SiBufferTimeBlockStn[iTransferMFL, iTransferSFL, 2];
				AR3SiNABufferTimeBlockStn[iTransferMFL, iTransferSFL, 3] := AR3SiBufferTimeBlockStn[iTransferMFL, iTransferSFL, 3];

				IF iTransferMFL>0 AND iTransferMFL <= iArmQty THEN

				AR3SiNABufferTimeBlockArm[iTransferMFL, iTransferSFL, 1] := AR3SiBufferTimeBlockArm[iTransferMFL, iTransferSFL, 1];
				AR3SiNABufferTimeBlockArm[iTransferMFL, iTransferSFL, 2] := AR3SiBufferTimeBlockArm[iTransferMFL, iTransferSFL, 2];
				AR3SiNABufferTimeBlockArm[iTransferMFL, iTransferSFL, 3] := AR3SiBufferTimeBlockArm[iTransferMFL, iTransferSFL, 3];

				END_IF

			END_FOR
		END_IF

	END_FOR

END_IF

IF iTransferMFL > iStnQty AND iTransferSFL > iMasterBlockQty THEN
NAScanFL:= iNextTransferTimeTemp;
ScanStep := 6;
END_IF


6: (*Reset NAScanMFL and NAScanSFL*)
NAScanMFL:=1;
NAScanSFL:=1;
ScanStep := 7;

7: (*Compare Not Available BufferTimeBlock VS RecipeTimeBlock*)


	IF NAScanFL>0 AND NAScanFL < iNextTransferTimeTemp+100+1 THEN
	NAScanMFL:=1;

		IF NAScanMFL>0 AND NAScanMFL < iRecipeBlockQty+1 THEN

			FOR NAScanMFL := 1 TO iRecipeBlockQty DO

				IF AR2SiInternalRepTimeBlockWithCallArmTime[NAScanMFL, 2] > 0 THEN

					iNAArmNo:=0;
					iNAStnNo:=0;
					bNAArmIDFound:= FALSE;
					bNAStnIDFound:= FALSE;

					iNACheckArmIDFL := 1;
					iNACheckStnIDFL := 1;

					(*Check ArmID*)
					IF iNACheckArmIDFL>0 AND iNACheckArmIDFL < iArmQty+1 THEN
						FOR iNACheckArmIDFL := 1 TO iArmQty DO
							IF AR2SiInternalRepTimeBlockWithCallArmTime[NAScanMFL,3] = ARiArmID[iNACheckArmIDFL] THEN
							iNAArmNo := iNACheckArmIDFL;
							bNAArmIDFound := TRUE;
							iNACheckArmIDFL := iArmQty+1;
							END_IF
						END_FOR
					END_IF

					(*Check StnID*)
					IF iNACheckStnIDFL>0 AND iNACheckStnIDFL <iStnQty+1 THEN
						FOR iNACheckStnIDFL := 1 TO iStnQty DO
							IF AR2SiInternalRepTimeBlockWithCallArmTime[NAScanMFL,3] = iNACheckStnIDFL THEN
							iNAStnNo := iNACheckStnIDFL;
							bNAStnIDFound := TRUE;
							iNACheckStnIDFL := iStnQty+1;
							END_IF
						END_FOR
					END_IF

					NAScanSFL := 1;
					bNACrashArm := FALSE;
					bNACrashStn := FALSE;



					IF (bNAArmIDFound OR bNAStnIDFound) AND NAScanSFL>0 AND NAScanSFL < iMasterBlockQty+1 THEN
						FOR NAScanSFL := 1 TO iMasterBlockQty DO

							(*Arm Scanning*)
							IF bNAArmIDFound THEN

								IF AR3SiNABufferTimeBlockArm[iNAArmNo,NAScanSFL, 2] > 0 THEN

									IF
									AR3SiNABufferTimeBlockArm[iNAArmNo,NAScanSFL, 1] (*MD1*) <= AR2SiInternalRepTimeBlockWithCallArmTime[NAScanMFL, 1] (*RD1*)
									AND
									AR3SiNABufferTimeBlockArm[iNAArmNo,NAScanSFL, 2] (*MD2*) >= AR2SiInternalRepTimeBlockWithCallArmTime[NAScanMFL, 1] (*RD1*)
									THEN
									bNACrashArm:=TRUE;
									NAScanSFL:=iMasterBlockQty+1;
									NAScanMFL := iRecipeBlockQty+1;
									END_IF

									IF
									AR3SiNABufferTimeBlockArm[iNAArmNo,NAScanSFL, 1] (*MD1*) <= AR2SiInternalRepTimeBlockWithCallArmTime[NAScanMFL, 2] (*RD2*)
									AND
									AR3SiNABufferTimeBlockArm[iNAArmNo,NAScanSFL, 2] (*MD2*) >= AR2SiInternalRepTimeBlockWithCallArmTime[NAScanMFL, 2] (*RD2*)
									THEN
									bNACrashArm:=TRUE;
									NAScanSFL:=iMasterBlockQty+1;
									NAScanMFL := iRecipeBlockQty+1;
									END_IF

									IF
									AR2SiInternalRepTimeBlockWithCallArmTime[NAScanMFL, 1] (*RD1*) <= AR3SiNABufferTimeBlockArm[iNAArmNo,NAScanSFL, 1] (*MD1*)
									AND
									AR2SiInternalRepTimeBlockWithCallArmTime[NAScanMFL, 2] (*RD2*) >= AR3SiNABufferTimeBlockArm[iNAArmNo,NAScanSFL, 1] (*MD1*)
									THEN
									bNACrashArm:=TRUE;
									NAScanSFL:=iMasterBlockQty+1;
									NAScanMFL := iRecipeBlockQty+1;
									END_IF

									IF
									AR2SiInternalRepTimeBlockWithCallArmTime[NAScanMFL, 1] (*RD1*) <= AR3SiNABufferTimeBlockArm[iNAArmNo,NAScanSFL, 2] (*MD2*)
									AND
									AR2SiInternalRepTimeBlockWithCallArmTime[NAScanMFL, 2] (*RD2*) >= AR3SiNABufferTimeBlockArm[iNAArmNo,NAScanSFL, 2] (*MD2*)
									THEN
									bNACrashArm:=TRUE;
									NAScanSFL:=iMasterBlockQty+1;
									NAScanMFL := iRecipeBlockQty+1;
									END_IF

								END_IF

							END_IF

							(*Stn Scanning*)
							IF bNAStnIDFound THEN

								IF AR3SiNABufferTimeBlockStn[iNAStnNo,NAScanSFL, 2] > 0 THEN

									IF
									AR3SiNABufferTimeBlockStn[iNAStnNo,NAScanSFL, 1] (*MD1*) <= AR2SiInternalRepTimeBlockWithCallArmTime[NAScanMFL, 1] (*RD1*)
									AND
									AR3SiNABufferTimeBlockStn[iNAStnNo,NAScanSFL, 2] (*MD2*) >= AR2SiInternalRepTimeBlockWithCallArmTime[NAScanMFL, 1] (*RD1*)
									THEN
									bNACrashStn:=TRUE;
									NAScanSFL:=iMasterBlockQty+1;
									NAScanMFL := iRecipeBlockQty+1;
									END_IF

									IF
									AR3SiNABufferTimeBlockStn[iNAStnNo,NAScanSFL, 1] (*MD1*) <= AR2SiInternalRepTimeBlockWithCallArmTime[NAScanMFL, 2] (*RD2*)
									AND
									AR3SiNABufferTimeBlockStn[iNAStnNo,NAScanSFL, 2] (*MD2*) >= AR2SiInternalRepTimeBlockWithCallArmTime[NAScanMFL, 2] (*RD2*)
									THEN
									bNACrashStn:=TRUE;
									NAScanSFL:=iMasterBlockQty+1;
									NAScanMFL := iRecipeBlockQty+1;
									END_IF

									IF
									AR2SiInternalRepTimeBlockWithCallArmTime[NAScanMFL, 1] (*RD1*) <= AR3SiNABufferTimeBlockStn[iNAStnNo,NAScanSFL, 1] (*MD1*)
									AND
									AR2SiInternalRepTimeBlockWithCallArmTime[NAScanMFL, 2] (*RD2*) >= AR3SiNABufferTimeBlockStn[iNAStnNo,NAScanSFL, 1] (*MD1*)
									THEN
									bNACrashStn:=TRUE;
									NAScanSFL:=iMasterBlockQty+1;
									NAScanMFL := iRecipeBlockQty+1;
									END_IF

									IF
									AR2SiInternalRepTimeBlockWithCallArmTime[NAScanMFL, 1] (*RD1*) <= AR3SiNABufferTimeBlockStn[iNAStnNo,NAScanSFL, 2] (*MD2*)
									AND
									AR2SiInternalRepTimeBlockWithCallArmTime[NAScanMFL, 2] (*RD2*) >= AR3SiNABufferTimeBlockStn[iNAStnNo,NAScanSFL, 2] (*MD2*)
									THEN
									bNACrashStn:=TRUE;
									NAScanSFL:=iMasterBlockQty+1;
									NAScanMFL := iRecipeBlockQty+1;
									END_IF

								END_IF
	
							END_IF

						END_FOR
	
					END_IF

				END_IF

			END_FOR

		END_IF

	END_IF

(* No Crash Found, minus one second and retry*)
IF NAScanMFL > iRecipeBlockQty AND NAScanSFL > iMasterBlockQty AND NOT bNACrashArm AND NOT bNACrashStn (*AND (bStepENRE.Q OR bStepAlwaysEN)*) THEN

		IF NAScanFL < 10000 THEN
		NAMTBMinusTimeMFL := 1;
		NAMTBMinusTimeSFL := 1;
		ScanStep := 8;
		END_IF

		IF NAScanFL >= iNextTransferTimeTemp+100 THEN
		iNextNotAvailableTimeTemp := NAScanFL; (*No Crash Found after the full scan*)
		ScanStep := 9;
		END_IF

END_IF


(* CRASH Found !!!, define next not available time*)
IF NAScanMFL > iRecipeBlockQty AND NAScanSFL > iMasterBlockQty AND (bNACrashArm OR bNACrashStn) (*AND (bStepENRE.Q OR bStepAlwaysEN)*) THEN
iNextNotAvailableTimeTemp := NAScanFL; (*Result FOUND*)
ScanStep := 9;
END_IF


(* No ArmID or StnID found*)
IF NAScanMFL > iRecipeBlockQty AND NOT bStnIDFound AND NOT bArmIDFound THEN
ScanStep := 23; (*ArmID and StnID not found Error*)
END_IF

8: (* No Crash Found, minus one second and retry*)


IF NAMTBMinusTimeMFL>0 AND NAMTBMinusTimeMFL < iStnQty+1 THEN
	FOR NAMTBMinusTimeMFL := 1 TO iStnQty DO
	NAMTBMinusTimeSFL := 1;
		IF NAMTBMinusTimeSFL>0 AND NAMTBMinusTimeSFL < iMasterBlockQty+1 THEN
			FOR NAMTBMinusTimeSFL := 1 TO iMasterBlockQty DO

				IF AR3SiNABufferTimeBlockStn[NAMTBMinusTimeMFL, NAMTBMinusTimeSFL, 1] > 0 THEN
				AR3SiNABufferTimeBlockStn[NAMTBMinusTimeMFL, NAMTBMinusTimeSFL, 1] := AR3SiNABufferTimeBlockStn[NAMTBMinusTimeMFL, NAMTBMinusTimeSFL, 1] - 1;
				END_IF

				IF AR3SiNABufferTimeBlockStn[NAMTBMinusTimeMFL, NAMTBMinusTimeSFL, 2] > 0 THEN
				AR3SiNABufferTimeBlockStn[NAMTBMinusTimeMFL, NAMTBMinusTimeSFL, 2] := AR3SiNABufferTimeBlockStn[NAMTBMinusTimeMFL, NAMTBMinusTimeSFL, 2] - 1;
				END_IF

				IF AR3SiNABufferTimeBlockStn[NAMTBMinusTimeMFL, NAMTBMinusTimeSFL, 2] <= 0 THEN
				AR3SiNABufferTimeBlockStn[NAMTBMinusTimeMFL, NAMTBMinusTimeSFL, 1] := 0;
				AR3SiNABufferTimeBlockStn[NAMTBMinusTimeMFL, NAMTBMinusTimeSFL, 2] := 0;
				AR3SiNABufferTimeBlockStn[NAMTBMinusTimeMFL, NAMTBMinusTimeSFL, 3] := 0;
				END_IF



				IF NAMTBMinusTimeMFL <= iArmQty THEN

					IF AR3SiNABufferTimeBlockArm[NAMTBMinusTimeMFL, NAMTBMinusTimeSFL, 1] > 0 THEN
					AR3SiNABufferTimeBlockArm[NAMTBMinusTimeMFL, NAMTBMinusTimeSFL, 1] := AR3SiNABufferTimeBlockArm[NAMTBMinusTimeMFL, NAMTBMinusTimeSFL, 1] - 1;
					END_IF

					IF AR3SiNABufferTimeBlockArm[NAMTBMinusTimeMFL, NAMTBMinusTimeSFL, 2] > 0 THEN
					AR3SiNABufferTimeBlockArm[NAMTBMinusTimeMFL, NAMTBMinusTimeSFL, 2] := AR3SiNABufferTimeBlockArm[NAMTBMinusTimeMFL, NAMTBMinusTimeSFL, 2] - 1;
					END_IF

					IF AR3SiNABufferTimeBlockArm[NAMTBMinusTimeMFL, NAMTBMinusTimeSFL, 2] <= 0 THEN
					AR3SiNABufferTimeBlockArm[NAMTBMinusTimeMFL, NAMTBMinusTimeSFL, 1] := 0;
					AR3SiNABufferTimeBlockArm[NAMTBMinusTimeMFL, NAMTBMinusTimeSFL, 2] := 0;
					AR3SiNABufferTimeBlockArm[NAMTBMinusTimeMFL, NAMTBMinusTimeSFL, 3] := 0;
					END_IF


				END_IF

			END_FOR
		END_IF

	END_FOR

END_IF


(*Return to Step 6 for retry*)

NAScanFL:=NAScanFL+1;
ScanStep := 6;



9: (* Simulated NextTransferTime Program*)

IF bScanStep9RE.Q THEN
	IF bMTBNotEmpty THEN
		iNextTransferTimeTemp := iNextTransferTimeTemp + iLoadingCallArmTime;
		iNextNotAvailableTimeTemp := iNextNotAvailableTimeTemp + iLoadingCallArmTime;
	END_IF
END_IF


IF bInternalScanEN THEN

	IF iNextTransferTimeTemp - iScanningCounter >= 0 AND OnTimeRE.Q THEN
	iNextTransferTime := iNextTransferTimeTemp - iScanningCounter;
	END_IF

	IF iNextTransferTimeTemp - iScanningCounter < 0  THEN
	iNextTransferTime := 0;
	END_IF



	IF iNextNotAvailableTimeTemp - iScanningCounter >= 0 AND OnTimeRE.Q THEN
	iNextNotAvailableTime := iNextNotAvailableTimeTemp - iScanningCounter;
	END_IF

	IF iNextNotAvailableTimeTemp - iScanningCounter < 0  THEN
	iNextNotAvailableTime := 0;
	END_IF

	bWriteDoneFlagRE(CLK:=bWriteDoneFlag , Q=> );
(*	bNotAvailableTimeRE(CLK:=  iNextNotAvailableTimeTemp <= iScanningCounter, Q=> );*)

	IF  iNextNotAvailableTimeTemp <= iScanningCounter THEN
	bNotAvailableTimeDetected:=TRUE;
	END_IF

	IF bWriteDoneFlagRE.Q OR bNotAvailableTimeDetected (*bNotAvailableTimeRE.Q*) THEN
	bInternalReScanFlag := TRUE;
	END_IF

END_IF

23: (* No ArmID or StnID found*)
bArmIDAndStnIDNotFound:=TRUE;


24: (*Cannot find suitable Slot*)
bNoAvailableSlotError:=TRUE;

END_CASE


(*Generate Scan CompleteFlag*)

DelayOnScanCompleteTimer(IN:=bInternalScanEN AND (ScanStep = 9) , PT:=INT_TO_TIME(iScanCompleteDelayOnTime_ms) , Q=> , ET=> );
IF DelayOnScanCompleteTimer.Q THEN
bScanCompletedFlag := TRUE;
ELSE
bScanCompletedFlag := FALSE;

END_IF

(*Write Basket into Master Time Block*)


(*Trigger Write*)

BWriteOnlyRE(CLK:= bInternalWriteEN AND NOT bWriteDisable AND iWriteStep <> 0 , Q=> );
bOverrideRE(CLK:= bOverrideWriteInterlock  , Q=> );


IF (NOT bStartEN OR NOT bInternalWriteEN OR bMTBResetEN OR NOT bScanCompletedFlag OR iNextTransferTime > 0 ) AND NOT bWriteHR  THEN
iWriteStep := 0; (*Reset and trigger Write Disable*)
END_IF

IF bStartEN AND NOT bMTBResetEN AND bScanCompletedFlag  AND NOT bWriteHR AND iNextTransferTime = 0 AND (NOT BWriteOnlyRE.Q AND NOT bOverrideRE.Q) THEN
iWriteStep := 1; (*Ready to Write*)
END_IF

IF BWriteOnlyRE.Q OR bOverrideRE.Q THEN
iWriteStep := 2; (*Write Start*)
bWriteHR := TRUE;
END_IF

IF NOT bInternalWriteEN THEN
bWriteHR := FALSE;
END_IF

IF iWriteRetryQtyPV < 1 THEN
iWriteRetryQtyPV := 1;
END_IF


CASE iWriteStep OF

0: (*Reset and trigger Write Disable*)
(*iWriteElapseTime := 0;*)
bWriteElapseTimeST:=FALSE;
bWriteDoneFlag := FALSE;
bWriteHR := FALSE;
bWriteDisable := TRUE;
bWriteArmDataError := FALSE;
bWriteStnDataError := FALSE;
iAutoRetryDelayTimer := 0;
iWriteRetryQtyPV := 1;

1:
bWriteDisable := FALSE;
bWriteHR := FALSE;
iWriteRetryQtyPV := 1;

2:
IF iNextTransferTime = 0 AND iNextNotAvailableTime >0 OR bOverrideRE.Q THEN
iWriteStep:=3; (*Prepare to Write*)
ELSE
iAutoRetryDelayTimer := 0;
iWriteStep := 11; (*Error Write -> Retry*)
END_IF


3: (*Prepare to Write*)
(*iWriteElapseTime:=0;*)
bWriteElapseTimeST:=TRUE;
bWriteDoneFlag := FALSE;
bWriteDisable := FALSE;
FillMFL := 1;
iWriteStep := 4;


4:
IF FillMFL>0 AND FillMFL < iRecipeBlockQty+1 THEN

	FOR FillMFL := 1 TO iRecipeBlockQty DO

		IF AR2SiInternalRepTimeBlockNoCallArmTime[FillMFL, 2] > 0 THEN

			iFillArmNo:=0;
			iFillStnNo:=0;
			bFIllArmIDFound:= FALSE;
			bFillStnIDFound:= FALSE;

			iCheckFillArmIDFL := 1;
			iCheckFillStnIDFL := 1;

